REGION Network 28: ABFV 103 MULTIGRADE FILTER VALVE
   RUNG wire#powerrail
      Contact( "AlwaysTRUE" )
      { S7_Templates := "SrcType := Int" } GE_Contact(in1 := "MODE SELECTION DB".MGF."PROCESS BUFF", in2 := 30)
      { S7_Templates := "SrcType := Int" } LT_Contact(in1 := "MODE SELECTION DB".MGF."PROCESS BUFF", in2 := 55)
      { S7_Templates := "time_type := Time" } "IEC_Timer_0_DB_143".TOF(pt := T#3S, et =>)
      Coil( "AUTO_SUBOUTPUT DB"."ABFV 103 MULTIGRADE FILTER VALVE" )
   END_RUNG
   // the same network as SCL:
   "IEC_Timer_0_DB_143".TOF(IN := "AlwaysTRUE" AND ("MODE SELECTION DB".MGF."PROCESS BUFF" >= 30) AND ("MODE SELECTION DB".MGF."PROCESS BUFF" < 55),
                           PT := T#3S);
   "AUTO_SUBOUTPUT DB"."ABFV 103 MULTIGRADE FILTER VALVE" := "IEC_Timer_0_DB_143".Q;
END_REGION

REGION Network 29: ABFV 104 MULTIGRADE FILTER VALVE
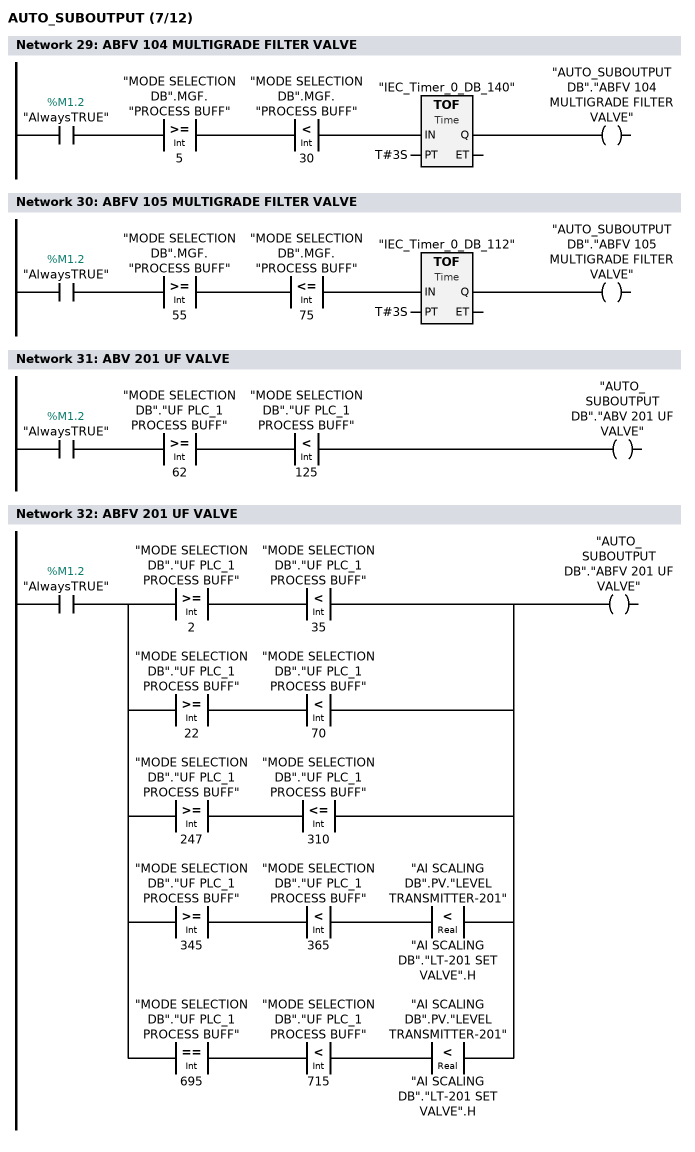
   RUNG wire#powerrail
      Contact( "AlwaysTRUE" )
      { S7_Templates := "SrcType := Int" } GE_Contact(in1 := "MODE SELECTION DB".MGF."PROCESS BUFF", in2 := 5)
      { S7_Templates := "SrcType := Int" } LT_Contact(in1 := "MODE SELECTION DB".MGF."PROCESS BUFF", in2 := 30)
      { S7_Templates := "time_type := Time" } "IEC_Timer_0_DB_140".TOF(pt := T#3S, et =>)
      Coil( "AUTO_SUBOUTPUT DB"."ABFV 104 MULTIGRADE FILTER VALVE" )
   END_RUNG
   // the same network as SCL:
   "IEC_Timer_0_DB_140".TOF(IN := "AlwaysTRUE" AND ("MODE SELECTION DB".MGF."PROCESS BUFF" >= 5) AND ("MODE SELECTION DB".MGF."PROCESS BUFF" < 30),
                           PT := T#3S);
   "AUTO_SUBOUTPUT DB"."ABFV 104 MULTIGRADE FILTER VALVE" := "IEC_Timer_0_DB_140".Q;
END_REGION

REGION Network 30: ABFV 105 MULTIGRADE FILTER VALVE
   RUNG wire#powerrail
      Contact( "AlwaysTRUE" )
      { S7_Templates := "SrcType := Int" } GE_Contact(in1 := "MODE SELECTION DB".MGF."PROCESS BUFF", in2 := 55)
      { S7_Templates := "SrcType := Int" } LE_Contact(in1 := "MODE SELECTION DB".MGF."PROCESS BUFF", in2 := 75)
      { S7_Templates := "time_type := Time" } "IEC_Timer_0_DB_112".TOF(pt := T#3S, et =>)
      Coil( "AUTO_SUBOUTPUT DB"."ABFV 105 MULTIGRADE FILTER VALVE" )
   END_RUNG
   // the same network as SCL:
   "IEC_Timer_0_DB_112".TOF(IN := "AlwaysTRUE" AND ("MODE SELECTION DB".MGF."PROCESS BUFF" >= 55) AND ("MODE SELECTION DB".MGF."PROCESS BUFF" <= 75),
                           PT := T#3S);
   "AUTO_SUBOUTPUT DB"."ABFV 105 MULTIGRADE FILTER VALVE" := "IEC_Timer_0_DB_112".Q;
END_REGION

REGION Network 31: ABV 201 UF VALVE
   RUNG wire#powerrail
      Contact( "AlwaysTRUE" )
      { S7_Templates := "SrcType := Int" } GE_Contact(in1 := "MODE SELECTION DB"."UF PLC_1 PROCESS BUFF", in2 := 62)
      { S7_Templates := "SrcType := Int" } LT_Contact(in1 := "MODE SELECTION DB"."UF PLC_1 PROCESS BUFF", in2 := 125)
      Coil( "AUTO_SUBOUTPUT DB"."ABV 201 UF VALVE" )
   END_RUNG
   // the same network as SCL:
   "AUTO_SUBOUTPUT DB"."ABV 201 UF VALVE" := "AlwaysTRUE" AND ("MODE SELECTION DB"."UF PLC_1 PROCESS BUFF" >= 62) AND ("MODE SELECTION DB"."UF PLC_1 PROCESS BUFF" < 125);
END_REGION

REGION Network 32: ABFV 201 UF VALVE
   RUNG wire#powerrail
      Contact( "AlwaysTRUE" )
      wire#w1
      { S7_Templates := "SrcType := Int" } GE_Contact(in1 := "MODE SELECTION DB"."UF PLC_1 PROCESS BUFF", in2 := 2)
      { S7_Templates := "SrcType := Int" } LT_Contact(in1 := "MODE SELECTION DB"."UF PLC_1 PROCESS BUFF", in2 := 35)
      wire#w2
      Coil( "AUTO_SUBOUTPUT DB"."ABFV 201 UF VALVE" )
   END_RUNG
   RUNG wire#w1
      { S7_Templates := "SrcType := Int" } GE_Contact(in1 := "MODE SELECTION DB"."UF PLC_1 PROCESS BUFF", in2 := 22)
      { S7_Templates := "SrcType := Int" } LT_Contact(in1 := "MODE SELECTION DB"."UF PLC_1 PROCESS BUFF", in2 := 70)
   END_RUNG wire#w2
   RUNG wire#w1
      { S7_Templates := "SrcType := Int" } GE_Contact(in1 := "MODE SELECTION DB"."UF PLC_1 PROCESS BUFF", in2 := 247)
      { S7_Templates := "SrcType := Int" } LE_Contact(in1 := "MODE SELECTION DB"."UF PLC_1 PROCESS BUFF", in2 := 310)
   END_RUNG wire#w2
   RUNG wire#w1
      { S7_Templates := "SrcType := Int" } GE_Contact(in1 := "MODE SELECTION DB"."UF PLC_1 PROCESS BUFF", in2 := 345)
      { S7_Templates := "SrcType := Int" } LT_Contact(in1 := "MODE SELECTION DB"."UF PLC_1 PROCESS BUFF", in2 := 365)
      { S7_Templates := "SrcType := Real" } LT_Contact(in1 := "AI SCALING DB".PV."LEVEL TRANSMITTER-201", in2 := "AI SCALING DB"."LT-201 SET VALVE".H)
   END_RUNG wire#w2
   RUNG wire#w1
      { S7_Templates := "SrcType := Int" } EQ_Contact(in1 := "MODE SELECTION DB"."UF PLC_1 PROCESS BUFF", in2 := 695)
      { S7_Templates := "SrcType := Int" } LT_Contact(in1 := "MODE SELECTION DB"."UF PLC_1 PROCESS BUFF", in2 := 715)
      { S7_Templates := "SrcType := Real" } LT_Contact(in1 := "AI SCALING DB".PV."LEVEL TRANSMITTER-201", in2 := "AI SCALING DB"."LT-201 SET VALVE".H)
   END_RUNG wire#w2
   // the same network as SCL:
   "AUTO_SUBOUTPUT DB"."ABFV 201 UF VALVE" := "AlwaysTRUE" AND ((("MODE SELECTION DB"."UF PLC_1 PROCESS BUFF" >= 2) AND ("MODE SELECTION DB"."UF PLC_1 PROCESS BUFF" < 35)) OR (("MODE SELECTION DB"."UF PLC_1 PROCESS BUFF" >= 22) AND ("MODE SELECTION DB"."UF PLC_1 PROCESS BUFF" < 70)) OR (("MODE SELECTION DB"."UF PLC_1 PROCESS BUFF" >= 247) AND ("MODE SELECTION DB"."UF PLC_1 PROCESS BUFF" <= 310)) OR (("MODE SELECTION DB"."UF PLC_1 PROCESS BUFF" >= 345) AND ("MODE SELECTION DB"."UF PLC_1 PROCESS BUFF" < 365) AND ("AI SCALING DB".PV."LEVEL TRANSMITTER-201" < "AI SCALING DB"."LT-201 SET VALVE".H)) OR (("MODE SELECTION DB"."UF PLC_1 PROCESS BUFF" = 695) AND ("MODE SELECTION DB"."UF PLC_1 PROCESS BUFF" < 715) AND ("AI SCALING DB".PV."LEVEL TRANSMITTER-201" < "AI SCALING DB"."LT-201 SET VALVE".H)));
END_REGION

REGION Network 33: ABFV 202 UF VALVE
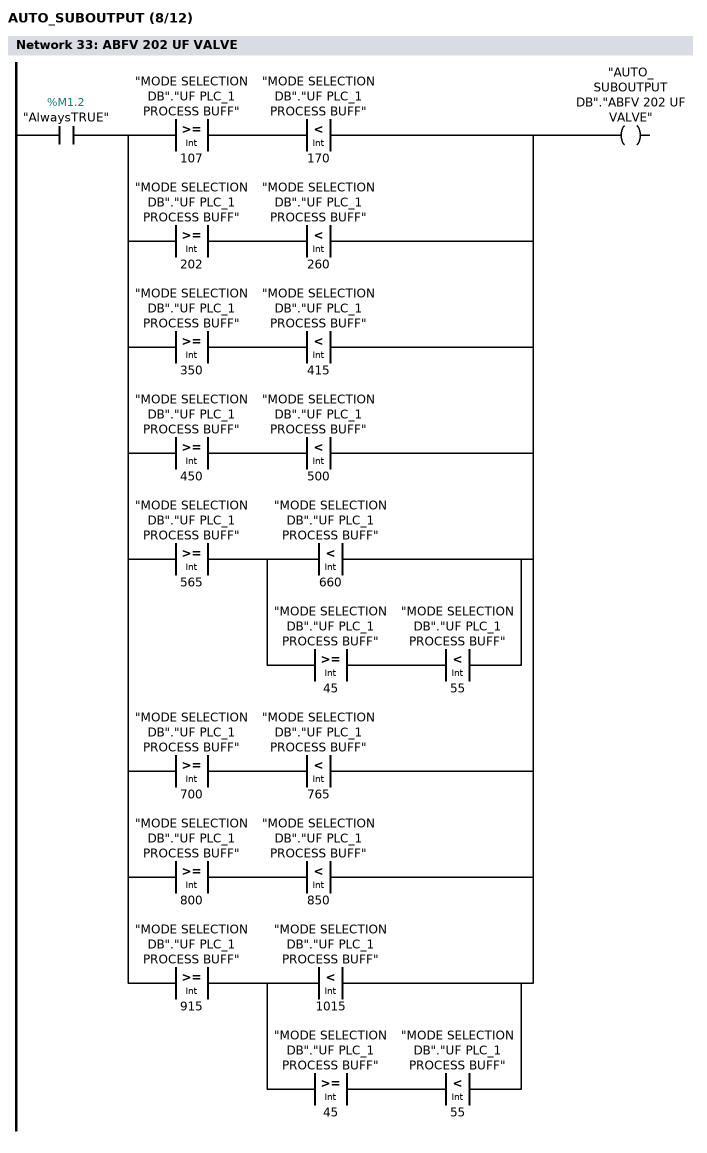
   RUNG wire#powerrail
      Contact( "AlwaysTRUE" )
      wire#w1
      { S7_Templates := "SrcType := Int" } GE_Contact(in1 := "MODE SELECTION DB"."UF PLC_1 PROCESS BUFF", in2 := 107)
      { S7_Templates := "SrcType := Int" } LT_Contact(in1 := "MODE SELECTION DB"."UF PLC_1 PROCESS BUFF", in2 := 170)
      wire#w2
      Coil( "AUTO_SUBOUTPUT DB"."ABFV 202 UF VALVE" )
   END_RUNG
   RUNG wire#w1
      { S7_Templates := "SrcType := Int" } GE_Contact(in1 := "MODE SELECTION DB"."UF PLC_1 PROCESS BUFF", in2 := 202)
      { S7_Templates := "SrcType := Int" } LT_Contact(in1 := "MODE SELECTION DB"."UF PLC_1 PROCESS BUFF", in2 := 260)
   END_RUNG wire#w2
   RUNG wire#w1
      { S7_Templates := "SrcType := Int" } GE_Contact(in1 := "MODE SELECTION DB"."UF PLC_1 PROCESS BUFF", in2 := 350)
      { S7_Templates := "SrcType := Int" } LT_Contact(in1 := "MODE SELECTION DB"."UF PLC_1 PROCESS BUFF", in2 := 415)
   END_RUNG wire#w2
   RUNG wire#w1
      { S7_Templates := "SrcType := Int" } GE_Contact(in1 := "MODE SELECTION DB"."UF PLC_1 PROCESS BUFF", in2 := 450)
      { S7_Templates := "SrcType := Int" } LT_Contact(in1 := "MODE SELECTION DB"."UF PLC_1 PROCESS BUFF", in2 := 500)
   END_RUNG wire#w2
   RUNG wire#w1
      { S7_Templates := "SrcType := Int" } GE_Contact(in1 := "MODE SELECTION DB"."UF PLC_1 PROCESS BUFF", in2 := 565)
      wire#w3
      { S7_Templates := "SrcType := Int" } LT_Contact(in1 := "MODE SELECTION DB"."UF PLC_1 PROCESS BUFF", in2 := 660)
   END_RUNG wire#w2
   RUNG wire#w3
      { S7_Templates := "SrcType := Int" } GE_Contact(in1 := "MODE SELECTION DB"."UF PLC_1 PROCESS BUFF", in2 := 45)
      { S7_Templates := "SrcType := Int" } LT_Contact(in1 := "MODE SELECTION DB"."UF PLC_1 PROCESS BUFF", in2 := 55)
   END_RUNG wire#w2
   RUNG wire#w1
      { S7_Templates := "SrcType := Int" } GE_Contact(in1 := "MODE SELECTION DB"."UF PLC_1 PROCESS BUFF", in2 := 700)
      { S7_Templates := "SrcType := Int" } LT_Contact(in1 := "MODE SELECTION DB"."UF PLC_1 PROCESS BUFF", in2 := 765)
   END_RUNG wire#w2
   RUNG wire#w1
      { S7_Templates := "SrcType := Int" } GE_Contact(in1 := "MODE SELECTION DB"."UF PLC_1 PROCESS BUFF", in2 := 800)
      { S7_Templates := "SrcType := Int" } LT_Contact(in1 := "MODE SELECTION DB"."UF PLC_1 PROCESS BUFF", in2 := 850)
   END_RUNG wire#w2
   RUNG wire#w1
      { S7_Templates := "SrcType := Int" } GE_Contact(in1 := "MODE SELECTION DB"."UF PLC_1 PROCESS BUFF", in2 := 915)
      wire#w4
      { S7_Templates := "SrcType := Int" } LT_Contact(in1 := "MODE SELECTION DB"."UF PLC_1 PROCESS BUFF", in2 := 1015)
   END_RUNG wire#w2
   RUNG wire#w4
      { S7_Templates := "SrcType := Int" } GE_Contact(in1 := "MODE SELECTION DB"."UF PLC_1 PROCESS BUFF", in2 := 45)
      { S7_Templates := "SrcType := Int" } LT_Contact(in1 := "MODE SELECTION DB"."UF PLC_1 PROCESS BUFF", in2 := 55)
   END_RUNG wire#w2
   // the same network as SCL:
   "AUTO_SUBOUTPUT DB"."ABFV 202 UF VALVE" := "AlwaysTRUE" AND ((("MODE SELECTION DB"."UF PLC_1 PROCESS BUFF" >= 107) AND ("MODE SELECTION DB"."UF PLC_1 PROCESS BUFF" < 170)) OR (("MODE SELECTION DB"."UF PLC_1 PROCESS BUFF" >= 202) AND ("MODE SELECTION DB"."UF PLC_1 PROCESS BUFF" < 260)) OR (("MODE SELECTION DB"."UF PLC_1 PROCESS BUFF" >= 350) AND ("MODE SELECTION DB"."UF PLC_1 PROCESS BUFF" < 415)) OR (("MODE SELECTION DB"."UF PLC_1 PROCESS BUFF" >= 450) AND ("MODE SELECTION DB"."UF PLC_1 PROCESS BUFF" < 500)) OR (("MODE SELECTION DB"."UF PLC_1 PROCESS BUFF" >= 565) AND (("MODE SELECTION DB"."UF PLC_1 PROCESS BUFF" < 660) OR (("MODE SELECTION DB"."UF PLC_1 PROCESS BUFF" >= 45) AND ("MODE SELECTION DB"."UF PLC_1 PROCESS BUFF" < 55)))) OR (("MODE SELECTION DB"."UF PLC_1 PROCESS BUFF" >= 700) AND ("MODE SELECTION DB"."UF PLC_1 PROCESS BUFF" < 765)) OR (("MODE SELECTION DB"."UF PLC_1 PROCESS BUFF" >= 800) AND ("MODE SELECTION DB"."UF PLC_1 PROCESS BUFF" < 850)) OR (("MODE SELECTION DB"."UF PLC_1 PROCESS BUFF" >= 915) AND (("MODE SELECTION DB"."UF PLC_1 PROCESS BUFF" < 1015) OR (("MODE SELECTION DB"."UF PLC_1 PROCESS BUFF" >= 45) AND ("MODE SELECTION DB"."UF PLC_1 PROCESS BUFF" < 55)))));
END_REGION

REGION Network 34: ABFV 203 UF VALVE
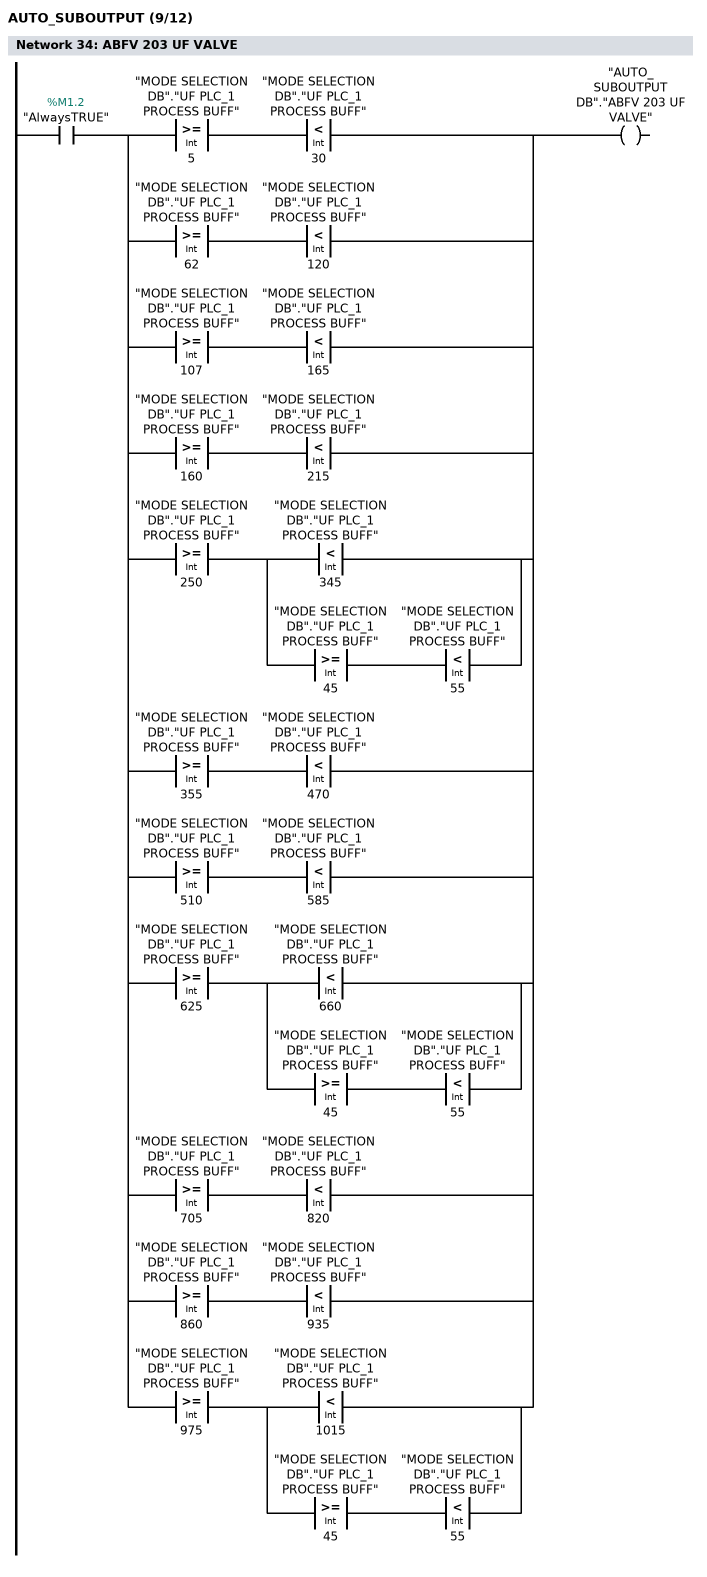
   RUNG wire#powerrail
      Contact( "AlwaysTRUE" )
      wire#w1
      { S7_Templates := "SrcType := Int" } GE_Contact(in1 := "MODE SELECTION DB"."UF PLC_1 PROCESS BUFF", in2 := 5)
      { S7_Templates := "SrcType := Int" } LT_Contact(in1 := "MODE SELECTION DB"."UF PLC_1 PROCESS BUFF", in2 := 30)
      wire#w2
      Coil( "AUTO_SUBOUTPUT DB"."ABFV 203 UF VALVE" )
   END_RUNG
   RUNG wire#w1
      { S7_Templates := "SrcType := Int" } GE_Contact(in1 := "MODE SELECTION DB"."UF PLC_1 PROCESS BUFF", in2 := 62)
      { S7_Templates := "SrcType := Int" } LT_Contact(in1 := "MODE SELECTION DB"."UF PLC_1 PROCESS BUFF", in2 := 120)
   END_RUNG wire#w2
   RUNG wire#w1
      { S7_Templates := "SrcType := Int" } GE_Contact(in1 := "MODE SELECTION DB"."UF PLC_1 PROCESS BUFF", in2 := 107)
      { S7_Templates := "SrcType := Int" } LT_Contact(in1 := "MODE SELECTION DB"."UF PLC_1 PROCESS BUFF", in2 := 165)
   END_RUNG wire#w2
   RUNG wire#w1
      { S7_Templates := "SrcType := Int" } GE_Contact(in1 := "MODE SELECTION DB"."UF PLC_1 PROCESS BUFF", in2 := 160)
      { S7_Templates := "SrcType := Int" } LT_Contact(in1 := "MODE SELECTION DB"."UF PLC_1 PROCESS BUFF", in2 := 215)
   END_RUNG wire#w2
   RUNG wire#w1
      { S7_Templates := "SrcType := Int" } GE_Contact(in1 := "MODE SELECTION DB"."UF PLC_1 PROCESS BUFF", in2 := 250)
      wire#w3
      { S7_Templates := "SrcType := Int" } LT_Contact(in1 := "MODE SELECTION DB"."UF PLC_1 PROCESS BUFF", in2 := 345)
   END_RUNG wire#w2
   RUNG wire#w3
      { S7_Templates := "SrcType := Int" } GE_Contact(in1 := "MODE SELECTION DB"."UF PLC_1 PROCESS BUFF", in2 := 45)
      { S7_Templates := "SrcType := Int" } LT_Contact(in1 := "MODE SELECTION DB"."UF PLC_1 PROCESS BUFF", in2 := 55)
   END_RUNG wire#w2
   RUNG wire#w1
      { S7_Templates := "SrcType := Int" } GE_Contact(in1 := "MODE SELECTION DB"."UF PLC_1 PROCESS BUFF", in2 := 355)
      { S7_Templates := "SrcType := Int" } LT_Contact(in1 := "MODE SELECTION DB"."UF PLC_1 PROCESS BUFF", in2 := 470)
   END_RUNG wire#w2
   RUNG wire#w1
      { S7_Templates := "SrcType := Int" } GE_Contact(in1 := "MODE SELECTION DB"."UF PLC_1 PROCESS BUFF", in2 := 510)
      { S7_Templates := "SrcType := Int" } LT_Contact(in1 := "MODE SELECTION DB"."UF PLC_1 PROCESS BUFF", in2 := 585)
   END_RUNG wire#w2
   RUNG wire#w1
      { S7_Templates := "SrcType := Int" } GE_Contact(in1 := "MODE SELECTION DB"."UF PLC_1 PROCESS BUFF", in2 := 625)
      wire#w4
      { S7_Templates := "SrcType := Int" } LT_Contact(in1 := "MODE SELECTION DB"."UF PLC_1 PROCESS BUFF", in2 := 660)
   END_RUNG wire#w2
   RUNG wire#w4
      { S7_Templates := "SrcType := Int" } GE_Contact(in1 := "MODE SELECTION DB"."UF PLC_1 PROCESS BUFF", in2 := 45)
      { S7_Templates := "SrcType := Int" } LT_Contact(in1 := "MODE SELECTION DB"."UF PLC_1 PROCESS BUFF", in2 := 55)
   END_RUNG wire#w2
   RUNG wire#w1
      { S7_Templates := "SrcType := Int" } GE_Contact(in1 := "MODE SELECTION DB"."UF PLC_1 PROCESS BUFF", in2 := 705)
      { S7_Templates := "SrcType := Int" } LT_Contact(in1 := "MODE SELECTION DB"."UF PLC_1 PROCESS BUFF", in2 := 820)
   END_RUNG wire#w2
   RUNG wire#w1
      { S7_Templates := "SrcType := Int" } GE_Contact(in1 := "MODE SELECTION DB"."UF PLC_1 PROCESS BUFF", in2 := 860)
      { S7_Templates := "SrcType := Int" } LT_Contact(in1 := "MODE SELECTION DB"."UF PLC_1 PROCESS BUFF", in2 := 935)
   END_RUNG wire#w2
   RUNG wire#w1
      { S7_Templates := "SrcType := Int" } GE_Contact(in1 := "MODE SELECTION DB"."UF PLC_1 PROCESS BUFF", in2 := 975)
      wire#w5
      { S7_Templates := "SrcType := Int" } LT_Contact(in1 := "MODE SELECTION DB"."UF PLC_1 PROCESS BUFF", in2 := 1015)
   END_RUNG wire#w2
   RUNG wire#w5
      { S7_Templates := "SrcType := Int" } GE_Contact(in1 := "MODE SELECTION DB"."UF PLC_1 PROCESS BUFF", in2 := 45)
      { S7_Templates := "SrcType := Int" } LT_Contact(in1 := "MODE SELECTION DB"."UF PLC_1 PROCESS BUFF", in2 := 55)
   END_RUNG wire#w2
   // the same network as SCL:
   "AUTO_SUBOUTPUT DB"."ABFV 203 UF VALVE" := "AlwaysTRUE" AND ((("MODE SELECTION DB"."UF PLC_1 PROCESS BUFF" >= 5) AND ("MODE SELECTION DB"."UF PLC_1 PROCESS BUFF" < 30)) OR (("MODE SELECTION DB"."UF PLC_1 PROCESS BUFF" >= 62) AND ("MODE SELECTION DB"."UF PLC_1 PROCESS BUFF" < 120)) OR (("MODE SELECTION DB"."UF PLC_1 PROCESS BUFF" >= 107) AND ("MODE SELECTION DB"."UF PLC_1 PROCESS BUFF" < 165)) OR (("MODE SELECTION DB"."UF PLC_1 PROCESS BUFF" >= 160) AND ("MODE SELECTION DB"."UF PLC_1 PROCESS BUFF" < 215)) OR (("MODE SELECTION DB"."UF PLC_1 PROCESS BUFF" >= 250) AND (("MODE SELECTION DB"."UF PLC_1 PROCESS BUFF" < 345) OR (("MODE SELECTION DB"."UF PLC_1 PROCESS BUFF" >= 45) AND ("MODE SELECTION DB"."UF PLC_1 PROCESS BUFF" < 55)))) OR (("MODE SELECTION DB"."UF PLC_1 PROCESS BUFF" >= 355) AND ("MODE SELECTION DB"."UF PLC_1 PROCESS BUFF" < 470)) OR (("MODE SELECTION DB"."UF PLC_1 PROCESS BUFF" >= 510) AND ("MODE SELECTION DB"."UF PLC_1 PROCESS BUFF" < 585)) OR (("MODE SELECTION DB"."UF PLC_1 PROCESS BUFF" >= 625) AND (("MODE SELECTION DB"."UF PLC_1 PROCESS BUFF" < 660) OR (("MODE SELECTION DB"."UF PLC_1 PROCESS BUFF" >= 45) AND ("MODE SELECTION DB"."UF PLC_1 PROCESS BUFF" < 55)))) OR (("MODE SELECTION DB"."UF PLC_1 PROCESS BUFF" >= 705) AND ("MODE SELECTION DB"."UF PLC_1 PROCESS BUFF" < 820)) OR (("MODE SELECTION DB"."UF PLC_1 PROCESS BUFF" >= 860) AND ("MODE SELECTION DB"."UF PLC_1 PROCESS BUFF" < 935)) OR (("MODE SELECTION DB"."UF PLC_1 PROCESS BUFF" >= 975) AND (("MODE SELECTION DB"."UF PLC_1 PROCESS BUFF" < 1015) OR (("MODE SELECTION DB"."UF PLC_1 PROCESS BUFF" >= 45) AND ("MODE SELECTION DB"."UF PLC_1 PROCESS BUFF" < 55)))));
END_REGION

REGION Network 35: ABFV 204 UF VALVE
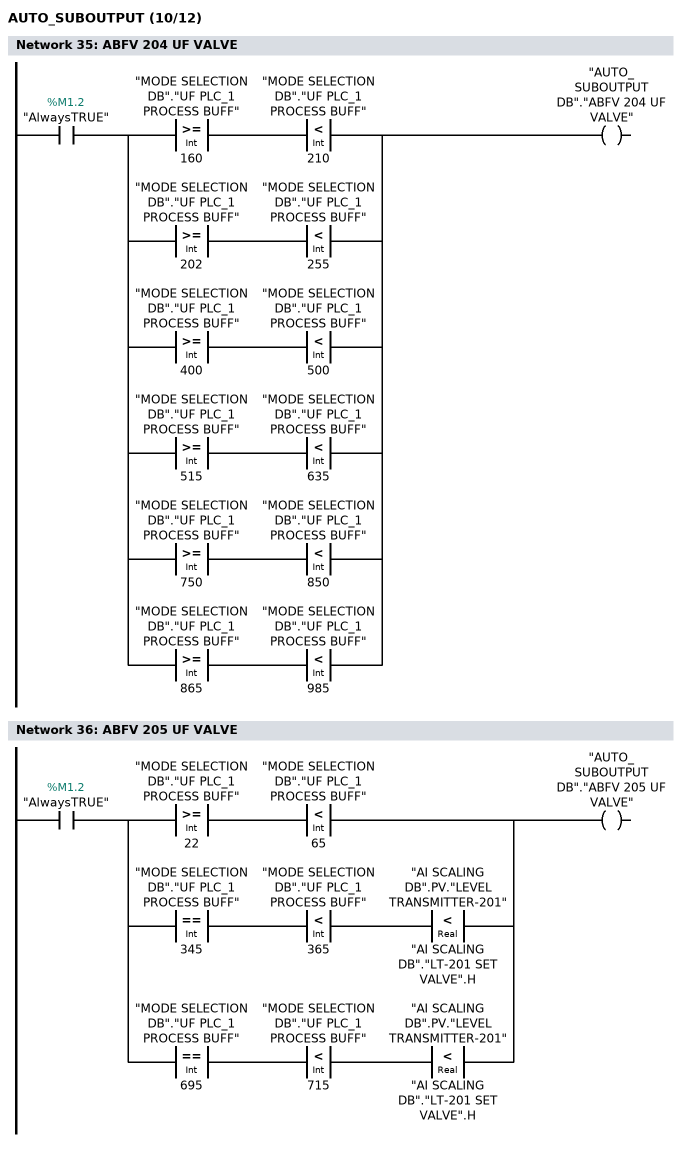
   RUNG wire#powerrail
      Contact( "AlwaysTRUE" )
      wire#w1
      { S7_Templates := "SrcType := Int" } GE_Contact(in1 := "MODE SELECTION DB"."UF PLC_1 PROCESS BUFF", in2 := 160)
      { S7_Templates := "SrcType := Int" } LT_Contact(in1 := "MODE SELECTION DB"."UF PLC_1 PROCESS BUFF", in2 := 210)
      wire#w2
      Coil( "AUTO_SUBOUTPUT DB"."ABFV 204 UF VALVE" )
   END_RUNG
   RUNG wire#w1
      { S7_Templates := "SrcType := Int" } GE_Contact(in1 := "MODE SELECTION DB"."UF PLC_1 PROCESS BUFF", in2 := 202)
      { S7_Templates := "SrcType := Int" } LT_Contact(in1 := "MODE SELECTION DB"."UF PLC_1 PROCESS BUFF", in2 := 255)
   END_RUNG wire#w2
   RUNG wire#w1
      { S7_Templates := "SrcType := Int" } GE_Contact(in1 := "MODE SELECTION DB"."UF PLC_1 PROCESS BUFF", in2 := 400)
      { S7_Templates := "SrcType := Int" } LT_Contact(in1 := "MODE SELECTION DB"."UF PLC_1 PROCESS BUFF", in2 := 500)
   END_RUNG wire#w2
   RUNG wire#w1
      { S7_Templates := "SrcType := Int" } GE_Contact(in1 := "MODE SELECTION DB"."UF PLC_1 PROCESS BUFF", in2 := 515)
      { S7_Templates := "SrcType := Int" } LT_Contact(in1 := "MODE SELECTION DB"."UF PLC_1 PROCESS BUFF", in2 := 635)
   END_RUNG wire#w2
   RUNG wire#w1
      { S7_Templates := "SrcType := Int" } GE_Contact(in1 := "MODE SELECTION DB"."UF PLC_1 PROCESS BUFF", in2 := 750)
      { S7_Templates := "SrcType := Int" } LT_Contact(in1 := "MODE SELECTION DB"."UF PLC_1 PROCESS BUFF", in2 := 850)
   END_RUNG wire#w2
   RUNG wire#w1
      { S7_Templates := "SrcType := Int" } GE_Contact(in1 := "MODE SELECTION DB"."UF PLC_1 PROCESS BUFF", in2 := 865)
      { S7_Templates := "SrcType := Int" } LT_Contact(in1 := "MODE SELECTION DB"."UF PLC_1 PROCESS BUFF", in2 := 985)
   END_RUNG wire#w2
   // the same network as SCL:
   "AUTO_SUBOUTPUT DB"."ABFV 204 UF VALVE" := "AlwaysTRUE" AND ((("MODE SELECTION DB"."UF PLC_1 PROCESS BUFF" >= 160) AND ("MODE SELECTION DB"."UF PLC_1 PROCESS BUFF" < 210)) OR (("MODE SELECTION DB"."UF PLC_1 PROCESS BUFF" >= 202) AND ("MODE SELECTION DB"."UF PLC_1 PROCESS BUFF" < 255)) OR (("MODE SELECTION DB"."UF PLC_1 PROCESS BUFF" >= 400) AND ("MODE SELECTION DB"."UF PLC_1 PROCESS BUFF" < 500)) OR (("MODE SELECTION DB"."UF PLC_1 PROCESS BUFF" >= 515) AND ("MODE SELECTION DB"."UF PLC_1 PROCESS BUFF" < 635)) OR (("MODE SELECTION DB"."UF PLC_1 PROCESS BUFF" >= 750) AND ("MODE SELECTION DB"."UF PLC_1 PROCESS BUFF" < 850)) OR (("MODE SELECTION DB"."UF PLC_1 PROCESS BUFF" >= 865) AND ("MODE SELECTION DB"."UF PLC_1 PROCESS BUFF" < 985)));
END_REGION

REGION Network 36: ABFV 205 UF VALVE
   RUNG wire#powerrail
      Contact( "AlwaysTRUE" )
      wire#w1
      { S7_Templates := "SrcType := Int" } GE_Contact(in1 := "MODE SELECTION DB"."UF PLC_1 PROCESS BUFF", in2 := 22)
      { S7_Templates := "SrcType := Int" } LT_Contact(in1 := "MODE SELECTION DB"."UF PLC_1 PROCESS BUFF", in2 := 65)
      wire#w2
      Coil( "AUTO_SUBOUTPUT DB"."ABFV 205 UF VALVE" )
   END_RUNG
   RUNG wire#w1
      { S7_Templates := "SrcType := Int" } EQ_Contact(in1 := "MODE SELECTION DB"."UF PLC_1 PROCESS BUFF", in2 := 345)
      { S7_Templates := "SrcType := Int" } LT_Contact(in1 := "MODE SELECTION DB"."UF PLC_1 PROCESS BUFF", in2 := 365)
      { S7_Templates := "SrcType := Real" } LT_Contact(in1 := "AI SCALING DB".PV."LEVEL TRANSMITTER-201", in2 := "AI SCALING DB"."LT-201 SET VALVE".H)
   END_RUNG wire#w2
   RUNG wire#w1
      { S7_Templates := "SrcType := Int" } EQ_Contact(in1 := "MODE SELECTION DB"."UF PLC_1 PROCESS BUFF", in2 := 695)
      { S7_Templates := "SrcType := Int" } LT_Contact(in1 := "MODE SELECTION DB"."UF PLC_1 PROCESS BUFF", in2 := 715)
      { S7_Templates := "SrcType := Real" } LT_Contact(in1 := "AI SCALING DB".PV."LEVEL TRANSMITTER-201", in2 := "AI SCALING DB"."LT-201 SET VALVE".H)
   END_RUNG wire#w2
   // the same network as SCL:
   "AUTO_SUBOUTPUT DB"."ABFV 205 UF VALVE" := "AlwaysTRUE" AND ((("MODE SELECTION DB"."UF PLC_1 PROCESS BUFF" >= 22) AND ("MODE SELECTION DB"."UF PLC_1 PROCESS BUFF" < 65)) OR (("MODE SELECTION DB"."UF PLC_1 PROCESS BUFF" = 345) AND ("MODE SELECTION DB"."UF PLC_1 PROCESS BUFF" < 365) AND ("AI SCALING DB".PV."LEVEL TRANSMITTER-201" < "AI SCALING DB"."LT-201 SET VALVE".H)) OR (("MODE SELECTION DB"."UF PLC_1 PROCESS BUFF" = 695) AND ("MODE SELECTION DB"."UF PLC_1 PROCESS BUFF" < 715) AND ("AI SCALING DB".PV."LEVEL TRANSMITTER-201" < "AI SCALING DB"."LT-201 SET VALVE".H)));
END_REGION

REGION Network 37: ABFV 206 UF VALVE
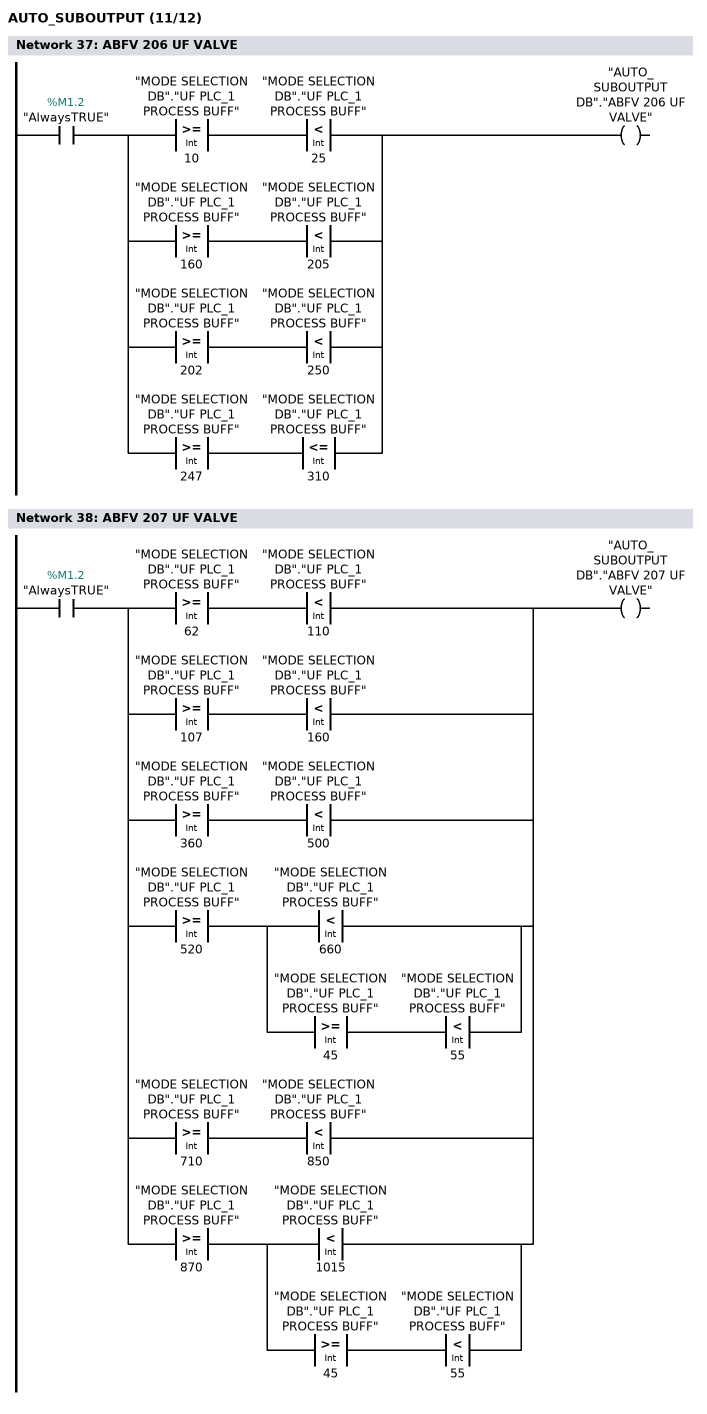
   RUNG wire#powerrail
      Contact( "AlwaysTRUE" )
      wire#w1
      { S7_Templates := "SrcType := Int" } GE_Contact(in1 := "MODE SELECTION DB"."UF PLC_1 PROCESS BUFF", in2 := 10)
      { S7_Templates := "SrcType := Int" } LT_Contact(in1 := "MODE SELECTION DB"."UF PLC_1 PROCESS BUFF", in2 := 25)
      wire#w2
      Coil( "AUTO_SUBOUTPUT DB"."ABFV 206 UF VALVE" )
   END_RUNG
   RUNG wire#w1
      { S7_Templates := "SrcType := Int" } GE_Contact(in1 := "MODE SELECTION DB"."UF PLC_1 PROCESS BUFF", in2 := 160)
      { S7_Templates := "SrcType := Int" } LT_Contact(in1 := "MODE SELECTION DB"."UF PLC_1 PROCESS BUFF", in2 := 205)
   END_RUNG wire#w2
   RUNG wire#w1
      { S7_Templates := "SrcType := Int" } GE_Contact(in1 := "MODE SELECTION DB"."UF PLC_1 PROCESS BUFF", in2 := 202)
      { S7_Templates := "SrcType := Int" } LT_Contact(in1 := "MODE SELECTION DB"."UF PLC_1 PROCESS BUFF", in2 := 250)
   END_RUNG wire#w2
   RUNG wire#w1
      { S7_Templates := "SrcType := Int" } GE_Contact(in1 := "MODE SELECTION DB"."UF PLC_1 PROCESS BUFF", in2 := 247)
      { S7_Templates := "SrcType := Int" } LE_Contact(in1 := "MODE SELECTION DB"."UF PLC_1 PROCESS BUFF", in2 := 310)
   END_RUNG wire#w2
   // the same network as SCL:
   "AUTO_SUBOUTPUT DB"."ABFV 206 UF VALVE" := "AlwaysTRUE" AND ((("MODE SELECTION DB"."UF PLC_1 PROCESS BUFF" >= 10) AND ("MODE SELECTION DB"."UF PLC_1 PROCESS BUFF" < 25)) OR (("MODE SELECTION DB"."UF PLC_1 PROCESS BUFF" >= 160) AND ("MODE SELECTION DB"."UF PLC_1 PROCESS BUFF" < 205)) OR (("MODE SELECTION DB"."UF PLC_1 PROCESS BUFF" >= 202) AND ("MODE SELECTION DB"."UF PLC_1 PROCESS BUFF" < 250)) OR (("MODE SELECTION DB"."UF PLC_1 PROCESS BUFF" >= 247) AND ("MODE SELECTION DB"."UF PLC_1 PROCESS BUFF" <= 310)));
END_REGION

REGION Network 38: ABFV 207 UF VALVE
   RUNG wire#powerrail
      Contact( "AlwaysTRUE" )
      wire#w1
      { S7_Templates := "SrcType := Int" } GE_Contact(in1 := "MODE SELECTION DB"."UF PLC_1 PROCESS BUFF", in2 := 62)
      { S7_Templates := "SrcType := Int" } LT_Contact(in1 := "MODE SELECTION DB"."UF PLC_1 PROCESS BUFF", in2 := 110)
      wire#w2
      Coil( "AUTO_SUBOUTPUT DB"."ABFV 207 UF VALVE" )
   END_RUNG
   RUNG wire#w1
      { S7_Templates := "SrcType := Int" } GE_Contact(in1 := "MODE SELECTION DB"."UF PLC_1 PROCESS BUFF", in2 := 107)
      { S7_Templates := "SrcType := Int" } LT_Contact(in1 := "MODE SELECTION DB"."UF PLC_1 PROCESS BUFF", in2 := 160)
   END_RUNG wire#w2
   RUNG wire#w1
      { S7_Templates := "SrcType := Int" } GE_Contact(in1 := "MODE SELECTION DB"."UF PLC_1 PROCESS BUFF", in2 := 360)
      { S7_Templates := "SrcType := Int" } LT_Contact(in1 := "MODE SELECTION DB"."UF PLC_1 PROCESS BUFF", in2 := 500)
   END_RUNG wire#w2
   RUNG wire#w1
      { S7_Templates := "SrcType := Int" } GE_Contact(in1 := "MODE SELECTION DB"."UF PLC_1 PROCESS BUFF", in2 := 520)
      wire#w3
      { S7_Templates := "SrcType := Int" } LT_Contact(in1 := "MODE SELECTION DB"."UF PLC_1 PROCESS BUFF", in2 := 660)
   END_RUNG wire#w2
   RUNG wire#w3
      { S7_Templates := "SrcType := Int" } GE_Contact(in1 := "MODE SELECTION DB"."UF PLC_1 PROCESS BUFF", in2 := 45)
      { S7_Templates := "SrcType := Int" } LT_Contact(in1 := "MODE SELECTION DB"."UF PLC_1 PROCESS BUFF", in2 := 55)
   END_RUNG wire#w2
   RUNG wire#w1
      { S7_Templates := "SrcType := Int" } GE_Contact(in1 := "MODE SELECTION DB"."UF PLC_1 PROCESS BUFF", in2 := 710)
      { S7_Templates := "SrcType := Int" } LT_Contact(in1 := "MODE SELECTION DB"."UF PLC_1 PROCESS BUFF", in2 := 850)
   END_RUNG wire#w2
   RUNG wire#w1
      { S7_Templates := "SrcType := Int" } GE_Contact(in1 := "MODE SELECTION DB"."UF PLC_1 PROCESS BUFF", in2 := 870)
      wire#w4
      { S7_Templates := "SrcType := Int" } LT_Contact(in1 := "MODE SELECTION DB"."UF PLC_1 PROCESS BUFF", in2 := 1015)
   END_RUNG wire#w2
   RUNG wire#w4
      { S7_Templates := "SrcType := Int" } GE_Contact(in1 := "MODE SELECTION DB"."UF PLC_1 PROCESS BUFF", in2 := 45)
      { S7_Templates := "SrcType := Int" } LT_Contact(in1 := "MODE SELECTION DB"."UF PLC_1 PROCESS BUFF", in2 := 55)
   END_RUNG wire#w2
   // the same network as SCL:
   "AUTO_SUBOUTPUT DB"."ABFV 207 UF VALVE" := "AlwaysTRUE" AND ((("MODE SELECTION DB"."UF PLC_1 PROCESS BUFF" >= 62) AND ("MODE SELECTION DB"."UF PLC_1 PROCESS BUFF" < 110)) OR (("MODE SELECTION DB"."UF PLC_1 PROCESS BUFF" >= 107) AND ("MODE SELECTION DB"."UF PLC_1 PROCESS BUFF" < 160)) OR (("MODE SELECTION DB"."UF PLC_1 PROCESS BUFF" >= 360) AND ("MODE SELECTION DB"."UF PLC_1 PROCESS BUFF" < 500)) OR (("MODE SELECTION DB"."UF PLC_1 PROCESS BUFF" >= 520) AND (("MODE SELECTION DB"."UF PLC_1 PROCESS BUFF" < 660) OR (("MODE SELECTION DB"."UF PLC_1 PROCESS BUFF" >= 45) AND ("MODE SELECTION DB"."UF PLC_1 PROCESS BUFF" < 55)))) OR (("MODE SELECTION DB"."UF PLC_1 PROCESS BUFF" >= 710) AND ("MODE SELECTION DB"."UF PLC_1 PROCESS BUFF" < 850)) OR (("MODE SELECTION DB"."UF PLC_1 PROCESS BUFF" >= 870) AND (("MODE SELECTION DB"."UF PLC_1 PROCESS BUFF" < 1015) OR (("MODE SELECTION DB"."UF PLC_1 PROCESS BUFF" >= 45) AND ("MODE SELECTION DB"."UF PLC_1 PROCESS BUFF" < 55)))));
END_REGION

REGION Network 39: ABFV 208 UF VALVE
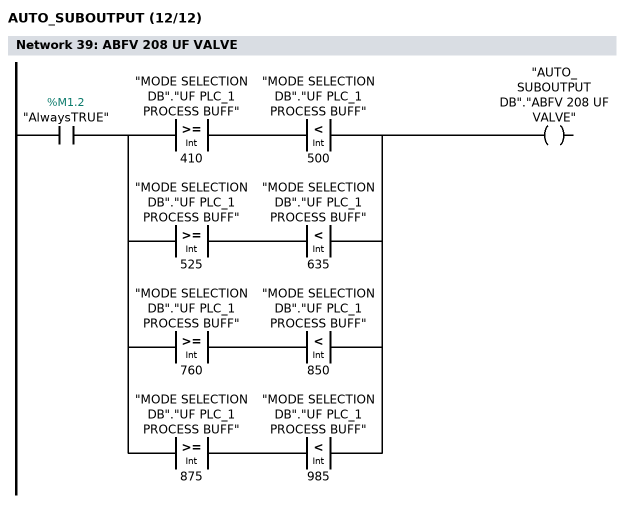
   RUNG wire#powerrail
      Contact( "AlwaysTRUE" )
      wire#w1
      { S7_Templates := "SrcType := Int" } GE_Contact(in1 := "MODE SELECTION DB"."UF PLC_1 PROCESS BUFF", in2 := 410)
      { S7_Templates := "SrcType := Int" } LT_Contact(in1 := "MODE SELECTION DB"."UF PLC_1 PROCESS BUFF", in2 := 500)
      wire#w2
      Coil( "AUTO_SUBOUTPUT DB"."ABFV 208 UF VALVE" )
   END_RUNG
   RUNG wire#w1
      { S7_Templates := "SrcType := Int" } GE_Contact(in1 := "MODE SELECTION DB"."UF PLC_1 PROCESS BUFF", in2 := 525)
      { S7_Templates := "SrcType := Int" } LT_Contact(in1 := "MODE SELECTION DB"."UF PLC_1 PROCESS BUFF", in2 := 635)
   END_RUNG wire#w2
   RUNG wire#w1
      { S7_Templates := "SrcType := Int" } GE_Contact(in1 := "MODE SELECTION DB"."UF PLC_1 PROCESS BUFF", in2 := 760)
      { S7_Templates := "SrcType := Int" } LT_Contact(in1 := "MODE SELECTION DB"."UF PLC_1 PROCESS BUFF", in2 := 850)
   END_RUNG wire#w2
   RUNG wire#w1
      { S7_Templates := "SrcType := Int" } GE_Contact(in1 := "MODE SELECTION DB"."UF PLC_1 PROCESS BUFF", in2 := 875)
      { S7_Templates := "SrcType := Int" } LT_Contact(in1 := "MODE SELECTION DB"."UF PLC_1 PROCESS BUFF", in2 := 985)
   END_RUNG wire#w2
   // the same network as SCL:
   "AUTO_SUBOUTPUT DB"."ABFV 208 UF VALVE" := "AlwaysTRUE" AND ((("MODE SELECTION DB"."UF PLC_1 PROCESS BUFF" >= 410) AND ("MODE SELECTION DB"."UF PLC_1 PROCESS BUFF" < 500)) OR (("MODE SELECTION DB"."UF PLC_1 PROCESS BUFF" >= 525) AND ("MODE SELECTION DB"."UF PLC_1 PROCESS BUFF" < 635)) OR (("MODE SELECTION DB"."UF PLC_1 PROCESS BUFF" >= 760) AND ("MODE SELECTION DB"."UF PLC_1 PROCESS BUFF" < 850)) OR (("MODE SELECTION DB"."UF PLC_1 PROCESS BUFF" >= 875) AND ("MODE SELECTION DB"."UF PLC_1 PROCESS BUFF" < 985)));
END_REGION
END_FUNCTION

FUNCTION "BACKWASH" : Void   // FC13, LAD
{ S7_Optimized_Access := 'TRUE' }
// stored: SetENOAutomatically false
BEGIN

REGION Network 1: BACKWASH_TIMER
END_REGION

REGION Network 2: VALVE OPEN
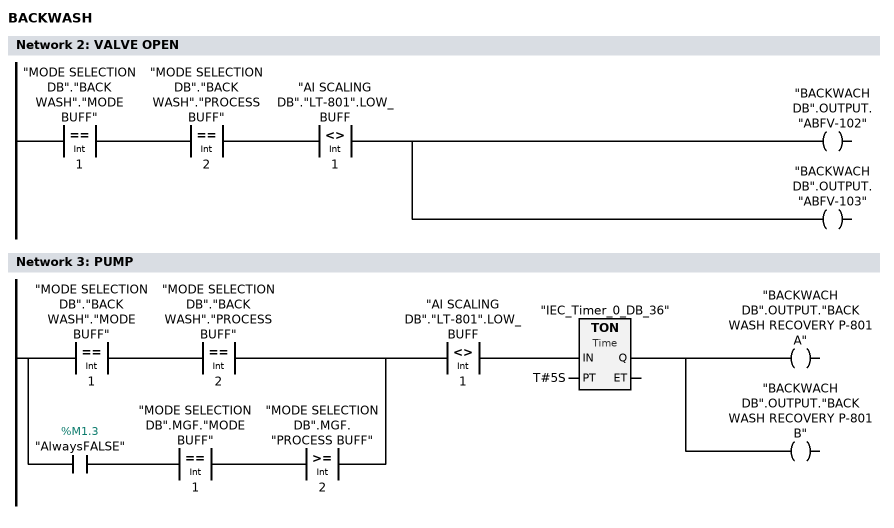
   RUNG wire#powerrail
      { S7_Templates := "SrcType := Int" } EQ_Contact(in1 := "MODE SELECTION DB"."BACK WASH"."MODE BUFF", in2 := 1)
      { S7_Templates := "SrcType := Int" } EQ_Contact(in1 := "MODE SELECTION DB"."BACK WASH"."PROCESS BUFF", in2 := 2)
      { S7_Templates := "SrcType := Int" } NE_Contact(in1 := "AI SCALING DB"."LT-801".LOW_BUFF, in2 := 1)
      wire#w1
      Coil( "BACKWACH DB".OUTPUT."ABFV-102" )
   END_RUNG
   RUNG wire#w1
      Coil( "BACKWACH DB".OUTPUT."ABFV-103" )
   END_RUNG
   // the same network as SCL:
   "BACKWACH DB".OUTPUT."ABFV-102" := ("MODE SELECTION DB"."BACK WASH"."MODE BUFF" = 1) AND ("MODE SELECTION DB"."BACK WASH"."PROCESS BUFF" = 2) AND ("AI SCALING DB"."LT-801".LOW_BUFF <> 1);
   "BACKWACH DB".OUTPUT."ABFV-103" := "BACKWACH DB".OUTPUT."ABFV-102";
END_REGION

REGION Network 3: PUMP
   RUNG wire#powerrail
      { S7_Templates := "SrcType := Int" } EQ_Contact(in1 := "MODE SELECTION DB"."BACK WASH"."MODE BUFF", in2 := 1)
      { S7_Templates := "SrcType := Int" } EQ_Contact(in1 := "MODE SELECTION DB"."BACK WASH"."PROCESS BUFF", in2 := 2)
      wire#w1
      { S7_Templates := "SrcType := Int" } NE_Contact(in1 := "AI SCALING DB"."LT-801".LOW_BUFF, in2 := 1)
      { S7_Templates := "time_type := Time" } "IEC_Timer_0_DB_36".TON(pt := T#5S, et =>)
      wire#w2
      Coil( "BACKWACH DB".OUTPUT."BACK WASH RECOVERY P-801 A" )
   END_RUNG
   RUNG wire#powerrail
      Contact( "AlwaysFALSE" )
      { S7_Templates := "SrcType := Int" } EQ_Contact(in1 := "MODE SELECTION DB".MGF."MODE BUFF", in2 := 1)
      { S7_Templates := "SrcType := Int" } GE_Contact(in1 := "MODE SELECTION DB".MGF."PROCESS BUFF", in2 := 2)
   END_RUNG wire#w1
   RUNG wire#w2
      Coil( "BACKWACH DB".OUTPUT."BACK WASH RECOVERY P-801 B" )
   END_RUNG
   // the same network as SCL:
   "IEC_Timer_0_DB_36".TON(IN := ((("MODE SELECTION DB"."BACK WASH"."MODE BUFF" = 1) AND ("MODE SELECTION DB"."BACK WASH"."PROCESS BUFF" = 2)) OR ("AlwaysFALSE" AND ("MODE SELECTION DB".MGF."MODE BUFF" = 1) AND ("MODE SELECTION DB".MGF."PROCESS BUFF" >= 2))) AND ("AI SCALING DB"."LT-801".LOW_BUFF <> 1),
                           PT := T#5S);
   "BACKWACH DB".OUTPUT."BACK WASH RECOVERY P-801 A" := "IEC_Timer_0_DB_36".Q;
   "BACKWACH DB".OUTPUT."BACK WASH RECOVERY P-801 B" := "IEC_Timer_0_DB_36".Q;
END_REGION
END_FUNCTION

FUNCTION "MGF AUTO" : Void   // FC10, LAD
{ S7_Optimized_Access := 'TRUE' }
// stored: SetENOAutomatically false
BEGIN

REGION Network 1
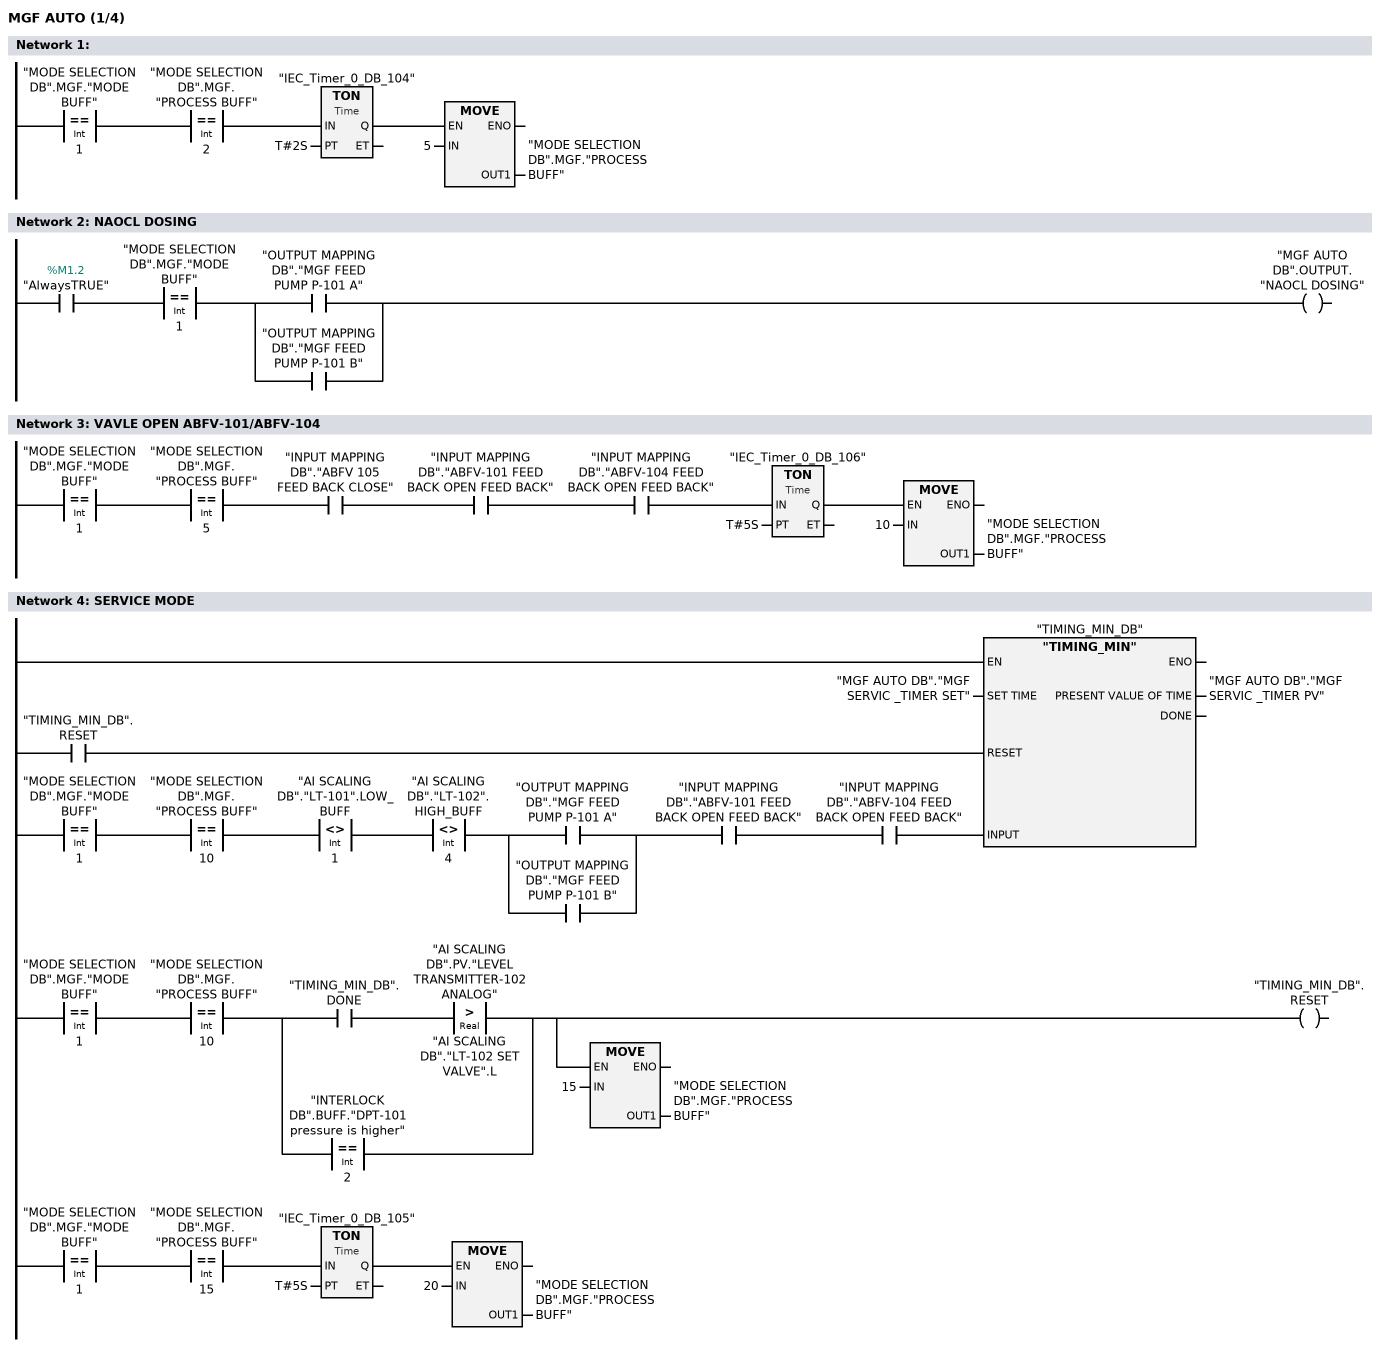
   RUNG wire#powerrail
      { S7_Templates := "SrcType := Int" } EQ_Contact(in1 := "MODE SELECTION DB".MGF."MODE BUFF", in2 := 1)
      { S7_Templates := "SrcType := Int" } EQ_Contact(in1 := "MODE SELECTION DB".MGF."PROCESS BUFF", in2 := 2)
      { S7_Templates := "time_type := Time" } "IEC_Timer_0_DB_104".TON(pt := T#2S, et =>)
      Move(in := 5, out1 => "MODE SELECTION DB".MGF."PROCESS BUFF")
   END_RUNG
   // the same network as SCL:
   "IEC_Timer_0_DB_104".TON(IN := ("MODE SELECTION DB".MGF."MODE BUFF" = 1) AND ("MODE SELECTION DB".MGF."PROCESS BUFF" = 2),
                           PT := T#2S);
   IF "IEC_Timer_0_DB_104".Q THEN "MODE SELECTION DB".MGF."PROCESS BUFF" := 5; END_IF;
END_REGION

REGION Network 2: NAOCL DOSING
   RUNG wire#powerrail
      Contact( "AlwaysTRUE" )
      { S7_Templates := "SrcType := Int" } EQ_Contact(in1 := "MODE SELECTION DB".MGF."MODE BUFF", in2 := 1)
      wire#w1
      Contact( "OUTPUT MAPPING DB"."MGF FEED PUMP P-101 A" )
      wire#w2
      Coil( "MGF AUTO DB".OUTPUT."NAOCL DOSING" )
   END_RUNG
   RUNG wire#w1
      Contact( "OUTPUT MAPPING DB"."MGF FEED PUMP P-101 B" )
   END_RUNG wire#w2
   // the same network as SCL:
   "MGF AUTO DB".OUTPUT."NAOCL DOSING" := "AlwaysTRUE" AND ("MODE SELECTION DB".MGF."MODE BUFF" = 1) AND ("OUTPUT MAPPING DB"."MGF FEED PUMP P-101 A" OR "OUTPUT MAPPING DB"."MGF FEED PUMP P-101 B");
END_REGION

REGION Network 3: VAVLE OPEN ABFV-101/ABFV-104
   RUNG wire#powerrail
      { S7_Templates := "SrcType := Int" } EQ_Contact(in1 := "MODE SELECTION DB".MGF."MODE BUFF", in2 := 1)
      { S7_Templates := "SrcType := Int" } EQ_Contact(in1 := "MODE SELECTION DB".MGF."PROCESS BUFF", in2 := 5)
      Contact( "INPUT MAPPING DB"."ABFV 105 FEED BACK CLOSE" )
      Contact( "INPUT MAPPING DB"."ABFV-101 FEED BACK OPEN FEED BACK" )
      Contact( "INPUT MAPPING DB"."ABFV-104 FEED BACK OPEN FEED BACK" )
      { S7_Templates := "time_type := Time" } "IEC_Timer_0_DB_106".TON(pt := T#5S, et =>)
      Move(in := 10, out1 => "MODE SELECTION DB".MGF."PROCESS BUFF")
   END_RUNG
   // the same network as SCL:
   "IEC_Timer_0_DB_106".TON(IN := ("MODE SELECTION DB".MGF."MODE BUFF" = 1) AND ("MODE SELECTION DB".MGF."PROCESS BUFF" = 5) AND "INPUT MAPPING DB"."ABFV 105 FEED BACK CLOSE" AND "INPUT MAPPING DB"."ABFV-101 FEED BACK OPEN FEED BACK" AND "INPUT MAPPING DB"."ABFV-104 FEED BACK OPEN FEED BACK",
                           PT := T#5S);
   IF "IEC_Timer_0_DB_106".Q THEN "MODE SELECTION DB".MGF."PROCESS BUFF" := 10; END_IF;
END_REGION

REGION Network 4: SERVICE MODE
   RUNG wire#powerrail
      "TIMING_MIN_DB"(RESET := wire#w1, INPUT := wire#w4, "SET TIME" := "MGF AUTO DB"."MGF SERVIC _TIMER SET", "PRESENT VALUE OF TIME" => "MGF AUTO DB"."MGF SERVIC _TIMER PV", DONE =>)
   END_RUNG
   RUNG wire#powerrail
      Contact( "TIMING_MIN_DB".RESET )
   END_RUNG wire#w1
   RUNG wire#powerrail
      { S7_Templates := "SrcType := Int" } EQ_Contact(in1 := "MODE SELECTION DB".MGF."MODE BUFF", in2 := 1)
      { S7_Templates := "SrcType := Int" } EQ_Contact(in1 := "MODE SELECTION DB".MGF."PROCESS BUFF", in2 := 10)
      { S7_Templates := "SrcType := Int" } NE_Contact(in1 := "AI SCALING DB"."LT-101".LOW_BUFF, in2 := 1)
      { S7_Templates := "SrcType := Int" } NE_Contact(in1 := "AI SCALING DB"."LT-102".HIGH_BUFF, in2 := 4)
      wire#w2
      Contact( "OUTPUT MAPPING DB"."MGF FEED PUMP P-101 A" )
      wire#w3
      Contact( "INPUT MAPPING DB"."ABFV-101 FEED BACK OPEN FEED BACK" )
      Contact( "INPUT MAPPING DB"."ABFV-104 FEED BACK OPEN FEED BACK" )
   END_RUNG wire#w4
   RUNG wire#w2
      Contact( "OUTPUT MAPPING DB"."MGF FEED PUMP P-101 B" )
   END_RUNG wire#w3
   RUNG wire#powerrail
      { S7_Templates := "SrcType := Int" } EQ_Contact(in1 := "MODE SELECTION DB".MGF."MODE BUFF", in2 := 1)
      { S7_Templates := "SrcType := Int" } EQ_Contact(in1 := "MODE SELECTION DB".MGF."PROCESS BUFF", in2 := 10)
      wire#w5
      Contact( "TIMING_MIN_DB".DONE )
      { S7_Templates := "SrcType := Real" } GT_Contact(in1 := "AI SCALING DB".PV."LEVEL TRANSMITTER-102 ANALOG", in2 := "AI SCALING DB"."LT-102 SET VALVE".L)
      wire#w6
      Coil( "TIMING_MIN_DB".RESET )
   END_RUNG
   RUNG wire#w5
      { S7_Templates := "SrcType := Int" } EQ_Contact(in1 := "INTERLOCK DB".BUFF."DPT-101 pressure is higher", in2 := 2)
   END_RUNG wire#w6
   RUNG wire#w6
      Move(in := 15, out1 => "MODE SELECTION DB".MGF."PROCESS BUFF")
   END_RUNG
   RUNG wire#powerrail
      { S7_Templates := "SrcType := Int" } EQ_Contact(in1 := "MODE SELECTION DB".MGF."MODE BUFF", in2 := 1)
      { S7_Templates := "SrcType := Int" } EQ_Contact(in1 := "MODE SELECTION DB".MGF."PROCESS BUFF", in2 := 15)
      { S7_Templates := "time_type := Time" } "IEC_Timer_0_DB_105".TON(pt := T#5S, et =>)
      Move(in := 20, out1 => "MODE SELECTION DB".MGF."PROCESS BUFF")
   END_RUNG
   // the same network as SCL:
   "TIMING_MIN_DB"("SET TIME" := "MGF AUTO DB"."MGF SERVIC _TIMER SET",   // "TIMING_MIN"
                   RESET := "TIMING_MIN_DB".RESET,
                   INPUT := ("MODE SELECTION DB".MGF."MODE BUFF" = 1) AND ("MODE SELECTION DB".MGF."PROCESS BUFF" = 10) AND ("AI SCALING DB"."LT-101".LOW_BUFF <> 1) AND ("AI SCALING DB"."LT-102".HIGH_BUFF <> 4) AND ("OUTPUT MAPPING DB"."MGF FEED PUMP P-101 A" OR "OUTPUT MAPPING DB"."MGF FEED PUMP P-101 B") AND "INPUT MAPPING DB"."ABFV-101 FEED BACK OPEN FEED BACK" AND "INPUT MAPPING DB"."ABFV-104 FEED BACK OPEN FEED BACK",
                   "PRESENT VALUE OF TIME" => "MGF AUTO DB"."MGF SERVIC _TIMER PV");
   "TIMING_MIN_DB".RESET := ("MODE SELECTION DB".MGF."MODE BUFF" = 1) AND ("MODE SELECTION DB".MGF."PROCESS BUFF" = 10) AND (("TIMING_MIN_DB".DONE AND ("AI SCALING DB".PV."LEVEL TRANSMITTER-102 ANALOG" > "AI SCALING DB"."LT-102 SET VALVE".L)) OR ("INTERLOCK DB".BUFF."DPT-101 pressure is higher" = 2));
   IF "TIMING_MIN_DB".RESET THEN "MODE SELECTION DB".MGF."PROCESS BUFF" := 15; END_IF;
   "IEC_Timer_0_DB_105".TON(IN := ("MODE SELECTION DB".MGF."MODE BUFF" = 1) AND ("MODE SELECTION DB".MGF."PROCESS BUFF" = 15),
                           PT := T#5S);
   IF "IEC_Timer_0_DB_105".Q THEN "MODE SELECTION DB".MGF."PROCESS BUFF" := 20; END_IF;
END_REGION

REGION Network 5: VAVLE CLOSE ABFV-101/ABFV-104
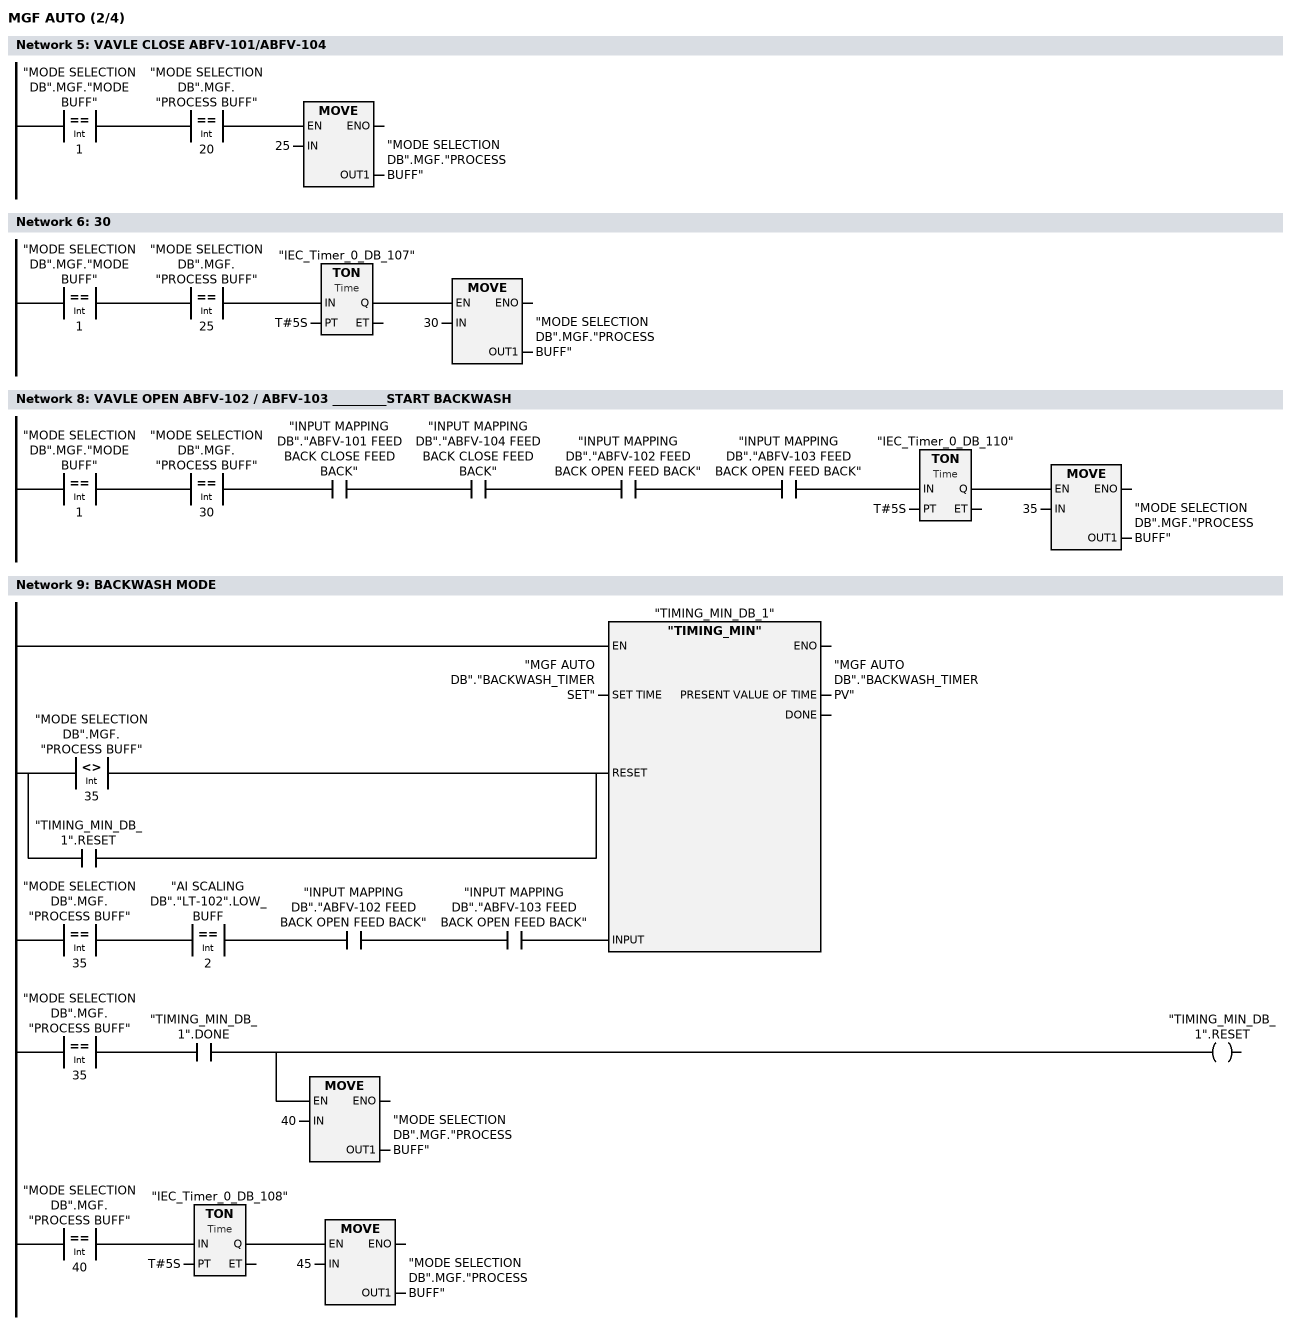
   RUNG wire#powerrail
      { S7_Templates := "SrcType := Int" } EQ_Contact(in1 := "MODE SELECTION DB".MGF."MODE BUFF", in2 := 1)
      { S7_Templates := "SrcType := Int" } EQ_Contact(in1 := "MODE SELECTION DB".MGF."PROCESS BUFF", in2 := 20)
      Move(in := 25, out1 => "MODE SELECTION DB".MGF."PROCESS BUFF")
   END_RUNG
   // the same network as SCL:
   IF ("MODE SELECTION DB".MGF."MODE BUFF" = 1) AND ("MODE SELECTION DB".MGF."PROCESS BUFF" = 20) THEN
       "MODE SELECTION DB".MGF."PROCESS BUFF" := 25;
   END_IF;
END_REGION

REGION Network 6: 30
   RUNG wire#powerrail
      { S7_Templates := "SrcType := Int" } EQ_Contact(in1 := "MODE SELECTION DB".MGF."MODE BUFF", in2 := 1)
      { S7_Templates := "SrcType := Int" } EQ_Contact(in1 := "MODE SELECTION DB".MGF."PROCESS BUFF", in2 := 25)
      { S7_Templates := "time_type := Time" } "IEC_Timer_0_DB_107".TON(pt := T#5S, et =>)
      Move(in := 30, out1 => "MODE SELECTION DB".MGF."PROCESS BUFF")
   END_RUNG
   // the same network as SCL:
   "IEC_Timer_0_DB_107".TON(IN := ("MODE SELECTION DB".MGF."MODE BUFF" = 1) AND ("MODE SELECTION DB".MGF."PROCESS BUFF" = 25),
                           PT := T#5S);
   IF "IEC_Timer_0_DB_107".Q THEN "MODE SELECTION DB".MGF."PROCESS BUFF" := 30; END_IF;
END_REGION

REGION Network 8: VAVLE OPEN ABFV-102 / ABFV-103 _________START BACKWASH
   RUNG wire#powerrail
      { S7_Templates := "SrcType := Int" } EQ_Contact(in1 := "MODE SELECTION DB".MGF."MODE BUFF", in2 := 1)
      { S7_Templates := "SrcType := Int" } EQ_Contact(in1 := "MODE SELECTION DB".MGF."PROCESS BUFF", in2 := 30)
      Contact( "INPUT MAPPING DB"."ABFV-101 FEED BACK CLOSE FEED BACK" )
      Contact( "INPUT MAPPING DB"."ABFV-104 FEED BACK CLOSE FEED BACK" )
      Contact( "INPUT MAPPING DB"."ABFV-102 FEED BACK OPEN FEED BACK" )
      Contact( "INPUT MAPPING DB"."ABFV-103 FEED BACK OPEN FEED BACK" )
      { S7_Templates := "time_type := Time" } "IEC_Timer_0_DB_110".TON(pt := T#5S, et =>)
      Move(in := 35, out1 => "MODE SELECTION DB".MGF."PROCESS BUFF")
   END_RUNG
   // the same network as SCL:
   "IEC_Timer_0_DB_110".TON(IN := ("MODE SELECTION DB".MGF."MODE BUFF" = 1) AND ("MODE SELECTION DB".MGF."PROCESS BUFF" = 30) AND "INPUT MAPPING DB"."ABFV-101 FEED BACK CLOSE FEED BACK" AND "INPUT MAPPING DB"."ABFV-104 FEED BACK CLOSE FEED BACK" AND "INPUT MAPPING DB"."ABFV-102 FEED BACK OPEN FEED BACK" AND "INPUT MAPPING DB"."ABFV-103 FEED BACK OPEN FEED BACK",
                           PT := T#5S);
   IF "IEC_Timer_0_DB_110".Q THEN "MODE SELECTION DB".MGF."PROCESS BUFF" := 35; END_IF;
END_REGION

REGION Network 9: BACKWASH MODE
   RUNG wire#powerrail
      "TIMING_MIN_DB_1"(RESET := wire#w1, INPUT := wire#w2, "SET TIME" := "MGF AUTO DB"."BACKWASH_TIMER SET", "PRESENT VALUE OF TIME" => "MGF AUTO DB"."BACKWASH_TIMER PV", DONE =>)
   END_RUNG
   RUNG wire#powerrail
      { S7_Templates := "SrcType := Int" } NE_Contact(in1 := "MODE SELECTION DB".MGF."PROCESS BUFF", in2 := 35)
   END_RUNG wire#w1
   RUNG wire#powerrail
      Contact( "TIMING_MIN_DB_1".RESET )
   END_RUNG wire#w1
   RUNG wire#powerrail
      { S7_Templates := "SrcType := Int" } EQ_Contact(in1 := "MODE SELECTION DB".MGF."PROCESS BUFF", in2 := 35)
      { S7_Templates := "SrcType := Int" } EQ_Contact(in1 := "AI SCALING DB"."LT-102".LOW_BUFF, in2 := 2)
      Contact( "INPUT MAPPING DB"."ABFV-102 FEED BACK OPEN FEED BACK" )
      Contact( "INPUT MAPPING DB"."ABFV-103 FEED BACK OPEN FEED BACK" )
   END_RUNG wire#w2
   RUNG wire#powerrail
      { S7_Templates := "SrcType := Int" } EQ_Contact(in1 := "MODE SELECTION DB".MGF."PROCESS BUFF", in2 := 35)
      Contact( "TIMING_MIN_DB_1".DONE )
      wire#w3
      Coil( "TIMING_MIN_DB_1".RESET )
   END_RUNG
   RUNG wire#w3
      Move(in := 40, out1 => "MODE SELECTION DB".MGF."PROCESS BUFF")
   END_RUNG
   RUNG wire#powerrail
      { S7_Templates := "SrcType := Int" } EQ_Contact(in1 := "MODE SELECTION DB".MGF."PROCESS BUFF", in2 := 40)
      { S7_Templates := "time_type := Time" } "IEC_Timer_0_DB_108".TON(pt := T#5S, et =>)
      Move(in := 45, out1 => "MODE SELECTION DB".MGF."PROCESS BUFF")
   END_RUNG
   // the same network as SCL:
   "TIMING_MIN_DB_1"("SET TIME" := "MGF AUTO DB"."BACKWASH_TIMER SET",   // "TIMING_MIN"
                     RESET := ("MODE SELECTION DB".MGF."PROCESS BUFF" <> 35) OR "TIMING_MIN_DB_1".RESET,
                     INPUT := ("MODE SELECTION DB".MGF."PROCESS BUFF" = 35) AND ("AI SCALING DB"."LT-102".LOW_BUFF = 2) AND "INPUT MAPPING DB"."ABFV-102 FEED BACK OPEN FEED BACK" AND "INPUT MAPPING DB"."ABFV-103 FEED BACK OPEN FEED BACK",
                     "PRESENT VALUE OF TIME" => "MGF AUTO DB"."BACKWASH_TIMER PV");
   "TIMING_MIN_DB_1".RESET := ("MODE SELECTION DB".MGF."PROCESS BUFF" = 35) AND "TIMING_MIN_DB_1".DONE;
   IF "TIMING_MIN_DB_1".RESET THEN "MODE SELECTION DB".MGF."PROCESS BUFF" := 40; END_IF;
   "IEC_Timer_0_DB_108".TON(IN := "MODE SELECTION DB".MGF."PROCESS BUFF" = 40, PT := T#5S);
   IF "IEC_Timer_0_DB_108".Q THEN "MODE SELECTION DB".MGF."PROCESS BUFF" := 45; END_IF;
END_REGION

REGION Network 10: VALVE CLOSE
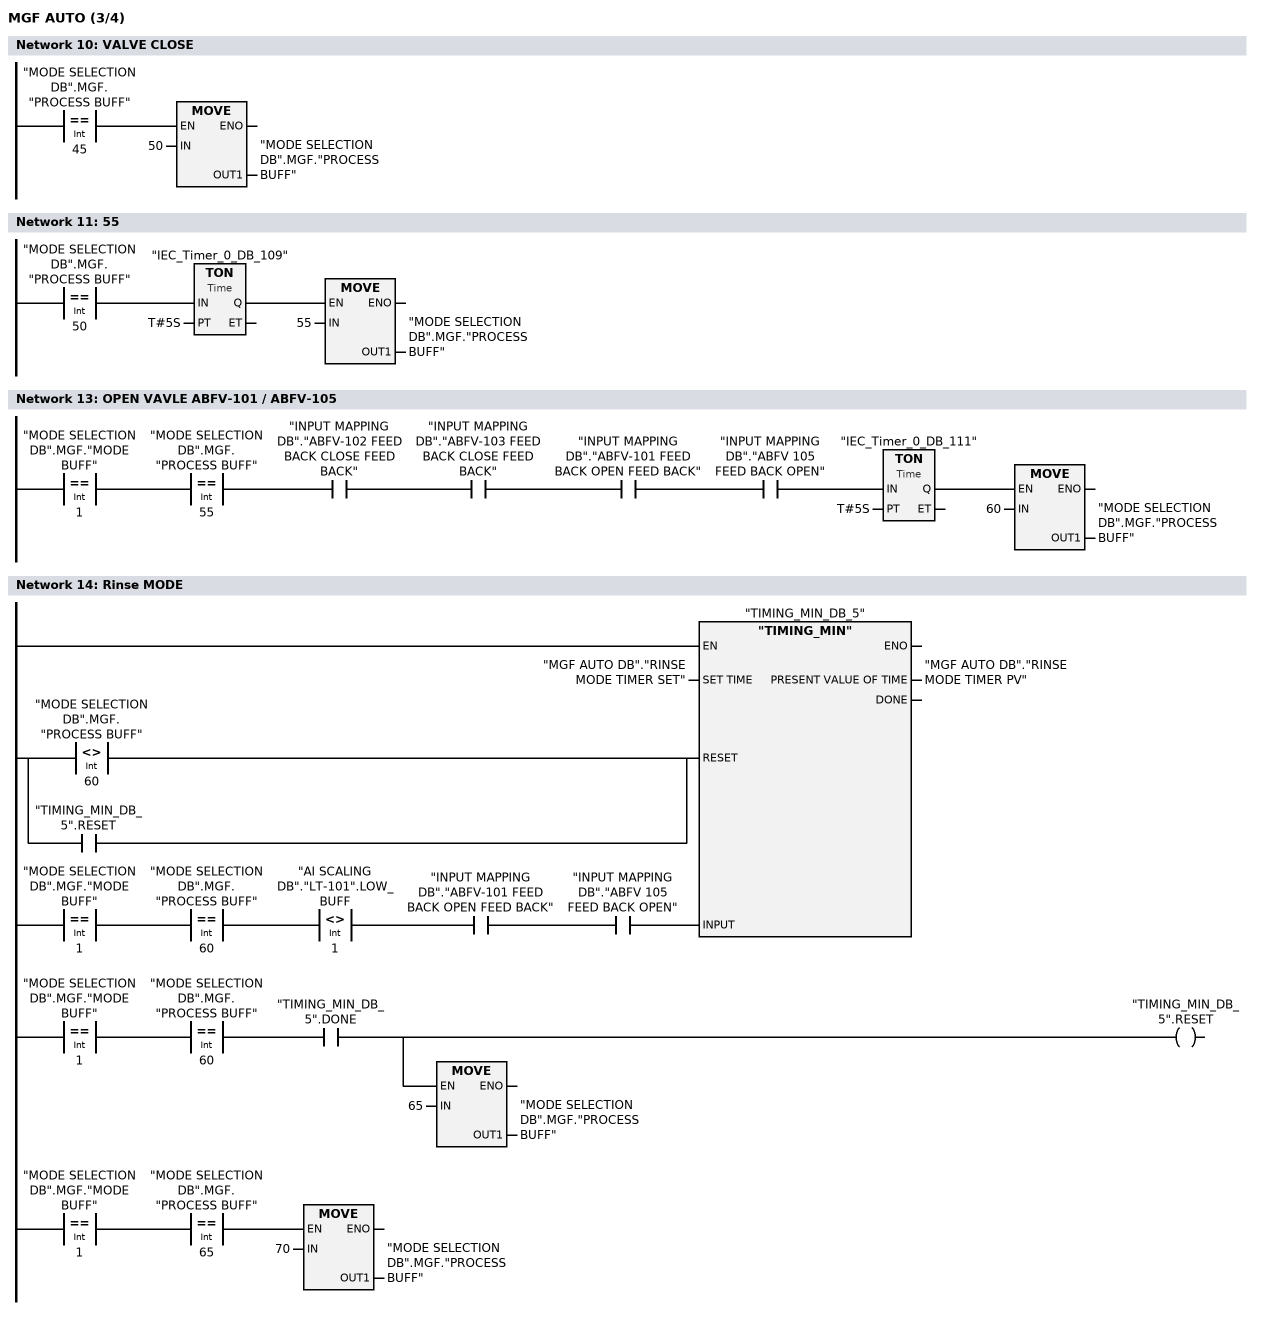
   RUNG wire#powerrail
      { S7_Templates := "SrcType := Int" } EQ_Contact(in1 := "MODE SELECTION DB".MGF."PROCESS BUFF", in2 := 45)
      Move(in := 50, out1 => "MODE SELECTION DB".MGF."PROCESS BUFF")
   END_RUNG
   // the same network as SCL:
   IF "MODE SELECTION DB".MGF."PROCESS BUFF" = 45 THEN "MODE SELECTION DB".MGF."PROCESS BUFF" := 50; END_IF;
END_REGION

REGION Network 11: 55
   RUNG wire#powerrail
      { S7_Templates := "SrcType := Int" } EQ_Contact(in1 := "MODE SELECTION DB".MGF."PROCESS BUFF", in2 := 50)
      { S7_Templates := "time_type := Time" } "IEC_Timer_0_DB_109".TON(pt := T#5S, et =>)
      Move(in := 55, out1 => "MODE SELECTION DB".MGF."PROCESS BUFF")
   END_RUNG
   // the same network as SCL:
   "IEC_Timer_0_DB_109".TON(IN := "MODE SELECTION DB".MGF."PROCESS BUFF" = 50, PT := T#5S);
   IF "IEC_Timer_0_DB_109".Q THEN "MODE SELECTION DB".MGF."PROCESS BUFF" := 55; END_IF;
END_REGION

REGION Network 13: OPEN VAVLE ABFV-101 / ABFV-105
   RUNG wire#powerrail
      { S7_Templates := "SrcType := Int" } EQ_Contact(in1 := "MODE SELECTION DB".MGF."MODE BUFF", in2 := 1)
      { S7_Templates := "SrcType := Int" } EQ_Contact(in1 := "MODE SELECTION DB".MGF."PROCESS BUFF", in2 := 55)
      Contact( "INPUT MAPPING DB"."ABFV-102 FEED BACK CLOSE FEED BACK" )
      Contact( "INPUT MAPPING DB"."ABFV-103 FEED BACK CLOSE FEED BACK" )
      Contact( "INPUT MAPPING DB"."ABFV-101 FEED BACK OPEN FEED BACK" )
      Contact( "INPUT MAPPING DB"."ABFV 105 FEED BACK OPEN" )
      { S7_Templates := "time_type := Time" } "IEC_Timer_0_DB_111".TON(pt := T#5S, et =>)
      Move(in := 60, out1 => "MODE SELECTION DB".MGF."PROCESS BUFF")
   END_RUNG
   // the same network as SCL:
   "IEC_Timer_0_DB_111".TON(IN := ("MODE SELECTION DB".MGF."MODE BUFF" = 1) AND ("MODE SELECTION DB".MGF."PROCESS BUFF" = 55) AND "INPUT MAPPING DB"."ABFV-102 FEED BACK CLOSE FEED BACK" AND "INPUT MAPPING DB"."ABFV-103 FEED BACK CLOSE FEED BACK" AND "INPUT MAPPING DB"."ABFV-101 FEED BACK OPEN FEED BACK" AND "INPUT MAPPING DB"."ABFV 105 FEED BACK OPEN",
                           PT := T#5S);
   IF "IEC_Timer_0_DB_111".Q THEN "MODE SELECTION DB".MGF."PROCESS BUFF" := 60; END_IF;
END_REGION

REGION Network 14: Rinse MODE
   RUNG wire#powerrail
      "TIMING_MIN_DB_5"(RESET := wire#w1, INPUT := wire#w2, "SET TIME" := "MGF AUTO DB"."RINSE MODE TIMER SET", "PRESENT VALUE OF TIME" => "MGF AUTO DB"."RINSE MODE TIMER PV", DONE =>)
   END_RUNG
   RUNG wire#powerrail
      { S7_Templates := "SrcType := Int" } NE_Contact(in1 := "MODE SELECTION DB".MGF."PROCESS BUFF", in2 := 60)
   END_RUNG wire#w1
   RUNG wire#powerrail
      Contact( "TIMING_MIN_DB_5".RESET )
   END_RUNG wire#w1
   RUNG wire#powerrail
      { S7_Templates := "SrcType := Int" } EQ_Contact(in1 := "MODE SELECTION DB".MGF."MODE BUFF", in2 := 1)
      { S7_Templates := "SrcType := Int" } EQ_Contact(in1 := "MODE SELECTION DB".MGF."PROCESS BUFF", in2 := 60)
      { S7_Templates := "SrcType := Int" } NE_Contact(in1 := "AI SCALING DB"."LT-101".LOW_BUFF, in2 := 1)
      Contact( "INPUT MAPPING DB"."ABFV-101 FEED BACK OPEN FEED BACK" )
      Contact( "INPUT MAPPING DB"."ABFV 105 FEED BACK OPEN" )
   END_RUNG wire#w2
   RUNG wire#powerrail
      { S7_Templates := "SrcType := Int" } EQ_Contact(in1 := "MODE SELECTION DB".MGF."MODE BUFF", in2 := 1)
      { S7_Templates := "SrcType := Int" } EQ_Contact(in1 := "MODE SELECTION DB".MGF."PROCESS BUFF", in2 := 60)
      Contact( "TIMING_MIN_DB_5".DONE )
      wire#w3
      Coil( "TIMING_MIN_DB_5".RESET )
   END_RUNG
   RUNG wire#w3
      Move(in := 65, out1 => "MODE SELECTION DB".MGF."PROCESS BUFF")
   END_RUNG
   RUNG wire#powerrail
      { S7_Templates := "SrcType := Int" } EQ_Contact(in1 := "MODE SELECTION DB".MGF."MODE BUFF", in2 := 1)
      { S7_Templates := "SrcType := Int" } EQ_Contact(in1 := "MODE SELECTION DB".MGF."PROCESS BUFF", in2 := 65)
      Move(in := 70, out1 => "MODE SELECTION DB".MGF."PROCESS BUFF")
   END_RUNG
   // the same network as SCL:
   "TIMING_MIN_DB_5"("SET TIME" := "MGF AUTO DB"."RINSE MODE TIMER SET",   // "TIMING_MIN"
                     RESET := ("MODE SELECTION DB".MGF."PROCESS BUFF" <> 60) OR "TIMING_MIN_DB_5".RESET,
                     INPUT := ("MODE SELECTION DB".MGF."MODE BUFF" = 1) AND ("MODE SELECTION DB".MGF."PROCESS BUFF" = 60) AND ("AI SCALING DB"."LT-101".LOW_BUFF <> 1) AND "INPUT MAPPING DB"."ABFV-101 FEED BACK OPEN FEED BACK" AND "INPUT MAPPING DB"."ABFV 105 FEED BACK OPEN",
                     "PRESENT VALUE OF TIME" => "MGF AUTO DB"."RINSE MODE TIMER PV");
   "TIMING_MIN_DB_5".RESET := ("MODE SELECTION DB".MGF."MODE BUFF" = 1) AND ("MODE SELECTION DB".MGF."PROCESS BUFF" = 60) AND "TIMING_MIN_DB_5".DONE;
   IF "TIMING_MIN_DB_5".RESET THEN "MODE SELECTION DB".MGF."PROCESS BUFF" := 65; END_IF;
   IF ("MODE SELECTION DB".MGF."MODE BUFF" = 1) AND ("MODE SELECTION DB".MGF."PROCESS BUFF" = 65) THEN
       "MODE SELECTION DB".MGF."PROCESS BUFF" := 70;
   END_IF;
END_REGION

REGION Network 15: VALVE CLOSE
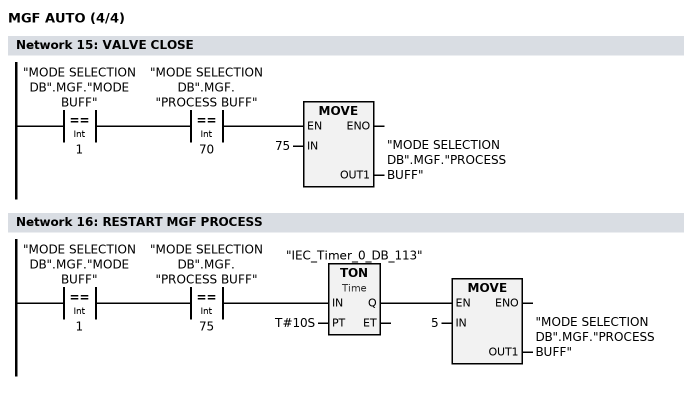
   RUNG wire#powerrail
      { S7_Templates := "SrcType := Int" } EQ_Contact(in1 := "MODE SELECTION DB".MGF."MODE BUFF", in2 := 1)
      { S7_Templates := "SrcType := Int" } EQ_Contact(in1 := "MODE SELECTION DB".MGF."PROCESS BUFF", in2 := 70)
      Move(in := 75, out1 => "MODE SELECTION DB".MGF."PROCESS BUFF")
   END_RUNG
   // the same network as SCL:
   IF ("MODE SELECTION DB".MGF."MODE BUFF" = 1) AND ("MODE SELECTION DB".MGF."PROCESS BUFF" = 70) THEN
       "MODE SELECTION DB".MGF."PROCESS BUFF" := 75;
   END_IF;
END_REGION

REGION Network 16: RESTART MGF PROCESS
   RUNG wire#powerrail
      { S7_Templates := "SrcType := Int" } EQ_Contact(in1 := "MODE SELECTION DB".MGF."MODE BUFF", in2 := 1)
      { S7_Templates := "SrcType := Int" } EQ_Contact(in1 := "MODE SELECTION DB".MGF."PROCESS BUFF", in2 := 75)
      { S7_Templates := "time_type := Time" } "IEC_Timer_0_DB_113".TON(pt := T#10S, et =>)
      Move(in := 5, out1 => "MODE SELECTION DB".MGF."PROCESS BUFF")
   END_RUNG
   // the same network as SCL:
   "IEC_Timer_0_DB_113".TON(IN := ("MODE SELECTION DB".MGF."MODE BUFF" = 1) AND ("MODE SELECTION DB".MGF."PROCESS BUFF" = 75),
                           PT := T#10S);
   IF "IEC_Timer_0_DB_113".Q THEN "MODE SELECTION DB".MGF."PROCESS BUFF" := 5; END_IF;
END_REGION
END_FUNCTION

FUNCTION "UF" : Void   // FC12, LAD
{ S7_Optimized_Access := 'TRUE' }
// stored: SetENOAutomatically false
   VAR_TEMP   // added for the SCL form of the ladder/FBD networks
      _w1 : Bool;
      _w2 : Bool;
   END_VAR
BEGIN

REGION Network 1: ABFV-201 OPEN F/B
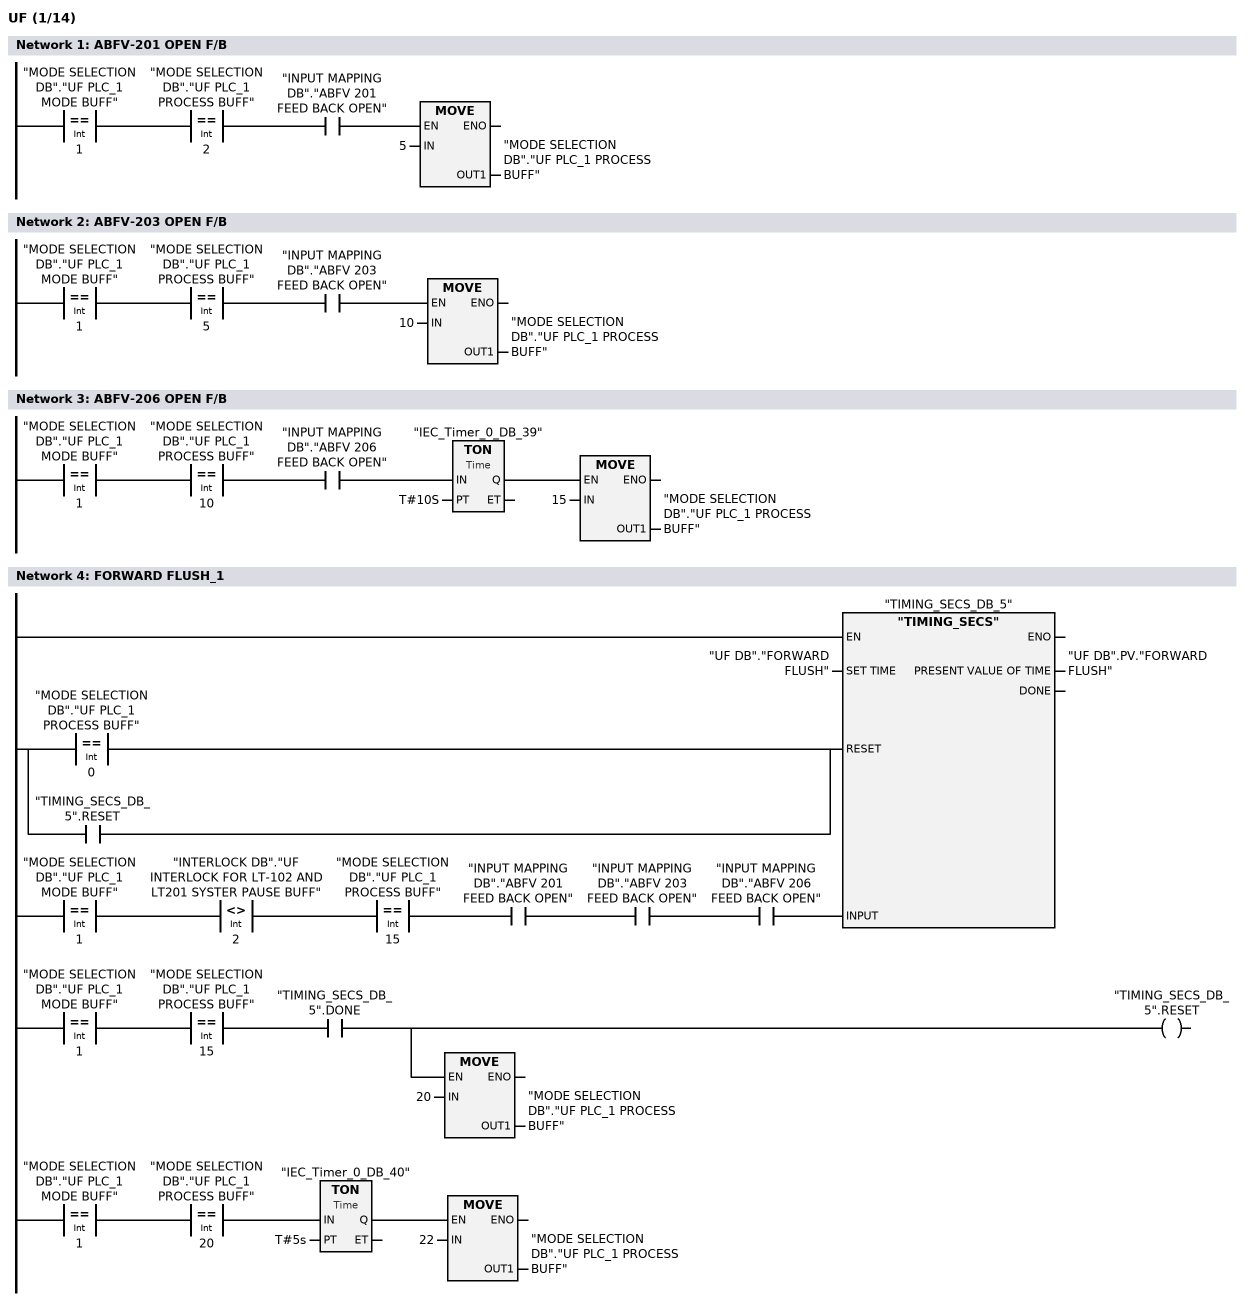
   RUNG wire#powerrail
      { S7_Templates := "SrcType := Int" } EQ_Contact(in1 := "MODE SELECTION DB"."UF PLC_1 MODE BUFF", in2 := 1)
      { S7_Templates := "SrcType := Int" } EQ_Contact(in1 := "MODE SELECTION DB"."UF PLC_1 PROCESS BUFF", in2 := 2)
      Contact( "INPUT MAPPING DB"."ABFV 201 FEED BACK OPEN" )
      Move(in := 5, out1 => "MODE SELECTION DB"."UF PLC_1 PROCESS BUFF")
   END_RUNG
   // the same network as SCL:
   IF ("MODE SELECTION DB"."UF PLC_1 MODE BUFF" = 1) AND ("MODE SELECTION DB"."UF PLC_1 PROCESS BUFF" = 2) AND "INPUT MAPPING DB"."ABFV 201 FEED BACK OPEN" THEN
       "MODE SELECTION DB"."UF PLC_1 PROCESS BUFF" := 5;
   END_IF;
END_REGION

REGION Network 2: ABFV-203 OPEN F/B
   RUNG wire#powerrail
      { S7_Templates := "SrcType := Int" } EQ_Contact(in1 := "MODE SELECTION DB"."UF PLC_1 MODE BUFF", in2 := 1)
      { S7_Templates := "SrcType := Int" } EQ_Contact(in1 := "MODE SELECTION DB"."UF PLC_1 PROCESS BUFF", in2 := 5)
      Contact( "INPUT MAPPING DB"."ABFV 203 FEED BACK OPEN" )
      Move(in := 10, out1 => "MODE SELECTION DB"."UF PLC_1 PROCESS BUFF")
   END_RUNG
   // the same network as SCL:
   IF ("MODE SELECTION DB"."UF PLC_1 MODE BUFF" = 1) AND ("MODE SELECTION DB"."UF PLC_1 PROCESS BUFF" = 5) AND "INPUT MAPPING DB"."ABFV 203 FEED BACK OPEN" THEN
       "MODE SELECTION DB"."UF PLC_1 PROCESS BUFF" := 10;
   END_IF;
END_REGION

REGION Network 3: ABFV-206 OPEN F/B
   RUNG wire#powerrail
      { S7_Templates := "SrcType := Int" } EQ_Contact(in1 := "MODE SELECTION DB"."UF PLC_1 MODE BUFF", in2 := 1)
      { S7_Templates := "SrcType := Int" } EQ_Contact(in1 := "MODE SELECTION DB"."UF PLC_1 PROCESS BUFF", in2 := 10)
      Contact( "INPUT MAPPING DB"."ABFV 206 FEED BACK OPEN" )
      { S7_Templates := "time_type := Time" } "IEC_Timer_0_DB_39".TON(pt := T#10S, et =>)
      Move(in := 15, out1 => "MODE SELECTION DB"."UF PLC_1 PROCESS BUFF")
   END_RUNG
   // the same network as SCL:
   "IEC_Timer_0_DB_39".TON(IN := ("MODE SELECTION DB"."UF PLC_1 MODE BUFF" = 1) AND ("MODE SELECTION DB"."UF PLC_1 PROCESS BUFF" = 10) AND "INPUT MAPPING DB"."ABFV 206 FEED BACK OPEN",
                           PT := T#10S);
   IF "IEC_Timer_0_DB_39".Q THEN "MODE SELECTION DB"."UF PLC_1 PROCESS BUFF" := 15; END_IF;
END_REGION

REGION Network 4: FORWARD FLUSH_1
   RUNG wire#powerrail
      "TIMING_SECS_DB_5"(RESET := wire#w1, INPUT := wire#w2, "SET TIME" := "UF DB"."FORWARD FLUSH", "PRESENT VALUE OF TIME" => "UF DB".PV."FORWARD FLUSH", DONE =>)
   END_RUNG
   RUNG wire#powerrail
      { S7_Templates := "SrcType := Int" } EQ_Contact(in1 := "MODE SELECTION DB"."UF PLC_1 PROCESS BUFF", in2 := 0)
   END_RUNG wire#w1
   RUNG wire#powerrail
      Contact( "TIMING_SECS_DB_5".RESET )
   END_RUNG wire#w1
   RUNG wire#powerrail
      { S7_Templates := "SrcType := Int" } EQ_Contact(in1 := "MODE SELECTION DB"."UF PLC_1 MODE BUFF", in2 := 1)
      { S7_Templates := "SrcType := Int" } NE_Contact(in1 := "INTERLOCK DB"."UF INTERLOCK FOR LT-102 AND LT201 SYSTER PAUSE BUFF", in2 := 2)
      { S7_Templates := "SrcType := Int" } EQ_Contact(in1 := "MODE SELECTION DB"."UF PLC_1 PROCESS BUFF", in2 := 15)
      Contact( "INPUT MAPPING DB"."ABFV 201 FEED BACK OPEN" )
      Contact( "INPUT MAPPING DB"."ABFV 203 FEED BACK OPEN" )
      Contact( "INPUT MAPPING DB"."ABFV 206 FEED BACK OPEN" )
   END_RUNG wire#w2
   RUNG wire#powerrail
      { S7_Templates := "SrcType := Int" } EQ_Contact(in1 := "MODE SELECTION DB"."UF PLC_1 MODE BUFF", in2 := 1)
      { S7_Templates := "SrcType := Int" } EQ_Contact(in1 := "MODE SELECTION DB"."UF PLC_1 PROCESS BUFF", in2 := 15)
      Contact( "TIMING_SECS_DB_5".DONE )
      wire#w3
      Coil( "TIMING_SECS_DB_5".RESET )
   END_RUNG
   RUNG wire#w3
      Move(in := 20, out1 => "MODE SELECTION DB"."UF PLC_1 PROCESS BUFF")
   END_RUNG
   RUNG wire#powerrail
      { S7_Templates := "SrcType := Int" } EQ_Contact(in1 := "MODE SELECTION DB"."UF PLC_1 MODE BUFF", in2 := 1)
      { S7_Templates := "SrcType := Int" } EQ_Contact(in1 := "MODE SELECTION DB"."UF PLC_1 PROCESS BUFF", in2 := 20)
      { S7_Templates := "time_type := Time" } "IEC_Timer_0_DB_40".TON(pt := T#5s, et =>)
      Move(in := 22, out1 => "MODE SELECTION DB"."UF PLC_1 PROCESS BUFF")
   END_RUNG
   // the same network as SCL:
   "TIMING_SECS_DB_5"("SET TIME" := "UF DB"."FORWARD FLUSH",   // "TIMING_SECS"
                      RESET := ("MODE SELECTION DB"."UF PLC_1 PROCESS BUFF" = 0) OR "TIMING_SECS_DB_5".RESET,
                      INPUT := ("MODE SELECTION DB"."UF PLC_1 MODE BUFF" = 1) AND ("INTERLOCK DB"."UF INTERLOCK FOR LT-102 AND LT201 SYSTER PAUSE BUFF" <> 2) AND ("MODE SELECTION DB"."UF PLC_1 PROCESS BUFF" = 15) AND "INPUT MAPPING DB"."ABFV 201 FEED BACK OPEN" AND "INPUT MAPPING DB"."ABFV 203 FEED BACK OPEN" AND "INPUT MAPPING DB"."ABFV 206 FEED BACK OPEN",
                      "PRESENT VALUE OF TIME" => "UF DB".PV."FORWARD FLUSH");
   "TIMING_SECS_DB_5".RESET := ("MODE SELECTION DB"."UF PLC_1 MODE BUFF" = 1) AND ("MODE SELECTION DB"."UF PLC_1 PROCESS BUFF" = 15) AND "TIMING_SECS_DB_5".DONE;
   IF "TIMING_SECS_DB_5".RESET THEN "MODE SELECTION DB"."UF PLC_1 PROCESS BUFF" := 20; END_IF;
   "IEC_Timer_0_DB_40".TON(IN := ("MODE SELECTION DB"."UF PLC_1 MODE BUFF" = 1) AND ("MODE SELECTION DB"."UF PLC_1 PROCESS BUFF" = 20),
                           PT := T#5s);
   IF "IEC_Timer_0_DB_40".Q THEN "MODE SELECTION DB"."UF PLC_1 PROCESS BUFF" := 22; END_IF;
END_REGION

REGION Network 5: OPEN ALL VALVE NEXT PROCESS
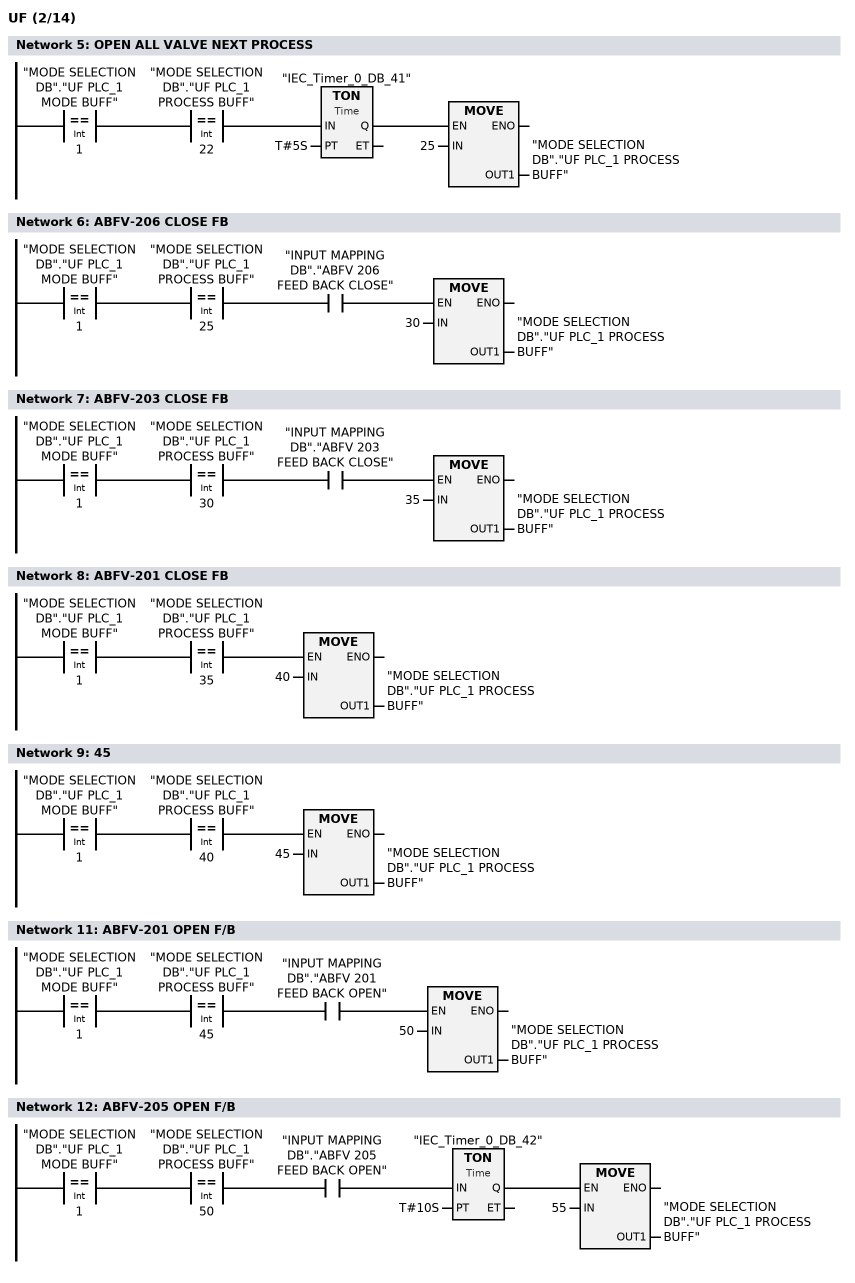
   RUNG wire#powerrail
      { S7_Templates := "SrcType := Int" } EQ_Contact(in1 := "MODE SELECTION DB"."UF PLC_1 MODE BUFF", in2 := 1)
      { S7_Templates := "SrcType := Int" } EQ_Contact(in1 := "MODE SELECTION DB"."UF PLC_1 PROCESS BUFF", in2 := 22)
      { S7_Templates := "time_type := Time" } "IEC_Timer_0_DB_41".TON(pt := T#5S, et =>)
      Move(in := 25, out1 => "MODE SELECTION DB"."UF PLC_1 PROCESS BUFF")
   END_RUNG
   // the same network as SCL:
   "IEC_Timer_0_DB_41".TON(IN := ("MODE SELECTION DB"."UF PLC_1 MODE BUFF" = 1) AND ("MODE SELECTION DB"."UF PLC_1 PROCESS BUFF" = 22),
                           PT := T#5S);
   IF "IEC_Timer_0_DB_41".Q THEN "MODE SELECTION DB"."UF PLC_1 PROCESS BUFF" := 25; END_IF;
END_REGION

REGION Network 6: ABFV-206 CLOSE FB
   RUNG wire#powerrail
      { S7_Templates := "SrcType := Int" } EQ_Contact(in1 := "MODE SELECTION DB"."UF PLC_1 MODE BUFF", in2 := 1)
      { S7_Templates := "SrcType := Int" } EQ_Contact(in1 := "MODE SELECTION DB"."UF PLC_1 PROCESS BUFF", in2 := 25)
      Contact( "INPUT MAPPING DB"."ABFV 206 FEED BACK CLOSE" )
      Move(in := 30, out1 => "MODE SELECTION DB"."UF PLC_1 PROCESS BUFF")
   END_RUNG
   // the same network as SCL:
   IF ("MODE SELECTION DB"."UF PLC_1 MODE BUFF" = 1) AND ("MODE SELECTION DB"."UF PLC_1 PROCESS BUFF" = 25) AND "INPUT MAPPING DB"."ABFV 206 FEED BACK CLOSE" THEN
       "MODE SELECTION DB"."UF PLC_1 PROCESS BUFF" := 30;
   END_IF;
END_REGION

REGION Network 7: ABFV-203 CLOSE FB
   RUNG wire#powerrail
      { S7_Templates := "SrcType := Int" } EQ_Contact(in1 := "MODE SELECTION DB"."UF PLC_1 MODE BUFF", in2 := 1)
      { S7_Templates := "SrcType := Int" } EQ_Contact(in1 := "MODE SELECTION DB"."UF PLC_1 PROCESS BUFF", in2 := 30)
      Contact( "INPUT MAPPING DB"."ABFV 203 FEED BACK CLOSE" )
      Move(in := 35, out1 => "MODE SELECTION DB"."UF PLC_1 PROCESS BUFF")
   END_RUNG
   // the same network as SCL:
   IF ("MODE SELECTION DB"."UF PLC_1 MODE BUFF" = 1) AND ("MODE SELECTION DB"."UF PLC_1 PROCESS BUFF" = 30) AND "INPUT MAPPING DB"."ABFV 203 FEED BACK CLOSE" THEN
       "MODE SELECTION DB"."UF PLC_1 PROCESS BUFF" := 35;
   END_IF;
END_REGION

REGION Network 8: ABFV-201 CLOSE FB
   RUNG wire#powerrail
      { S7_Templates := "SrcType := Int" } EQ_Contact(in1 := "MODE SELECTION DB"."UF PLC_1 MODE BUFF", in2 := 1)
      { S7_Templates := "SrcType := Int" } EQ_Contact(in1 := "MODE SELECTION DB"."UF PLC_1 PROCESS BUFF", in2 := 35)
      Move(in := 40, out1 => "MODE SELECTION DB"."UF PLC_1 PROCESS BUFF")
   END_RUNG
   // the same network as SCL:
   IF ("MODE SELECTION DB"."UF PLC_1 MODE BUFF" = 1) AND ("MODE SELECTION DB"."UF PLC_1 PROCESS BUFF" = 35) THEN
       "MODE SELECTION DB"."UF PLC_1 PROCESS BUFF" := 40;
   END_IF;
END_REGION

REGION Network 9: 45
   RUNG wire#powerrail
      { S7_Templates := "SrcType := Int" } EQ_Contact(in1 := "MODE SELECTION DB"."UF PLC_1 MODE BUFF", in2 := 1)
      { S7_Templates := "SrcType := Int" } EQ_Contact(in1 := "MODE SELECTION DB"."UF PLC_1 PROCESS BUFF", in2 := 40)
      Move(in := 45, out1 => "MODE SELECTION DB"."UF PLC_1 PROCESS BUFF")
   END_RUNG
   // the same network as SCL:
   IF ("MODE SELECTION DB"."UF PLC_1 MODE BUFF" = 1) AND ("MODE SELECTION DB"."UF PLC_1 PROCESS BUFF" = 40) THEN
       "MODE SELECTION DB"."UF PLC_1 PROCESS BUFF" := 45;
   END_IF;
END_REGION

REGION Network 11: ABFV-201 OPEN F/B
   RUNG wire#powerrail
      { S7_Templates := "SrcType := Int" } EQ_Contact(in1 := "MODE SELECTION DB"."UF PLC_1 MODE BUFF", in2 := 1)
      { S7_Templates := "SrcType := Int" } EQ_Contact(in1 := "MODE SELECTION DB"."UF PLC_1 PROCESS BUFF", in2 := 45)
      Contact( "INPUT MAPPING DB"."ABFV 201 FEED BACK OPEN" )
      Move(in := 50, out1 => "MODE SELECTION DB"."UF PLC_1 PROCESS BUFF")
   END_RUNG
   // the same network as SCL:
   IF ("MODE SELECTION DB"."UF PLC_1 MODE BUFF" = 1) AND ("MODE SELECTION DB"."UF PLC_1 PROCESS BUFF" = 45) AND "INPUT MAPPING DB"."ABFV 201 FEED BACK OPEN" THEN
       "MODE SELECTION DB"."UF PLC_1 PROCESS BUFF" := 50;
   END_IF;
END_REGION

REGION Network 12: ABFV-205 OPEN F/B
   RUNG wire#powerrail
      { S7_Templates := "SrcType := Int" } EQ_Contact(in1 := "MODE SELECTION DB"."UF PLC_1 MODE BUFF", in2 := 1)
      { S7_Templates := "SrcType := Int" } EQ_Contact(in1 := "MODE SELECTION DB"."UF PLC_1 PROCESS BUFF", in2 := 50)
      Contact( "INPUT MAPPING DB"."ABFV 205 FEED BACK OPEN" )
      { S7_Templates := "time_type := Time" } "IEC_Timer_0_DB_42".TON(pt := T#10S, et =>)
      Move(in := 55, out1 => "MODE SELECTION DB"."UF PLC_1 PROCESS BUFF")
   END_RUNG
   // the same network as SCL:
   "IEC_Timer_0_DB_42".TON(IN := ("MODE SELECTION DB"."UF PLC_1 MODE BUFF" = 1) AND ("MODE SELECTION DB"."UF PLC_1 PROCESS BUFF" = 50) AND "INPUT MAPPING DB"."ABFV 205 FEED BACK OPEN",
                           PT := T#10S);
   IF "IEC_Timer_0_DB_42".Q THEN "MODE SELECTION DB"."UF PLC_1 PROCESS BUFF" := 55; END_IF;
END_REGION

REGION Network 13: FILTRATION MODE
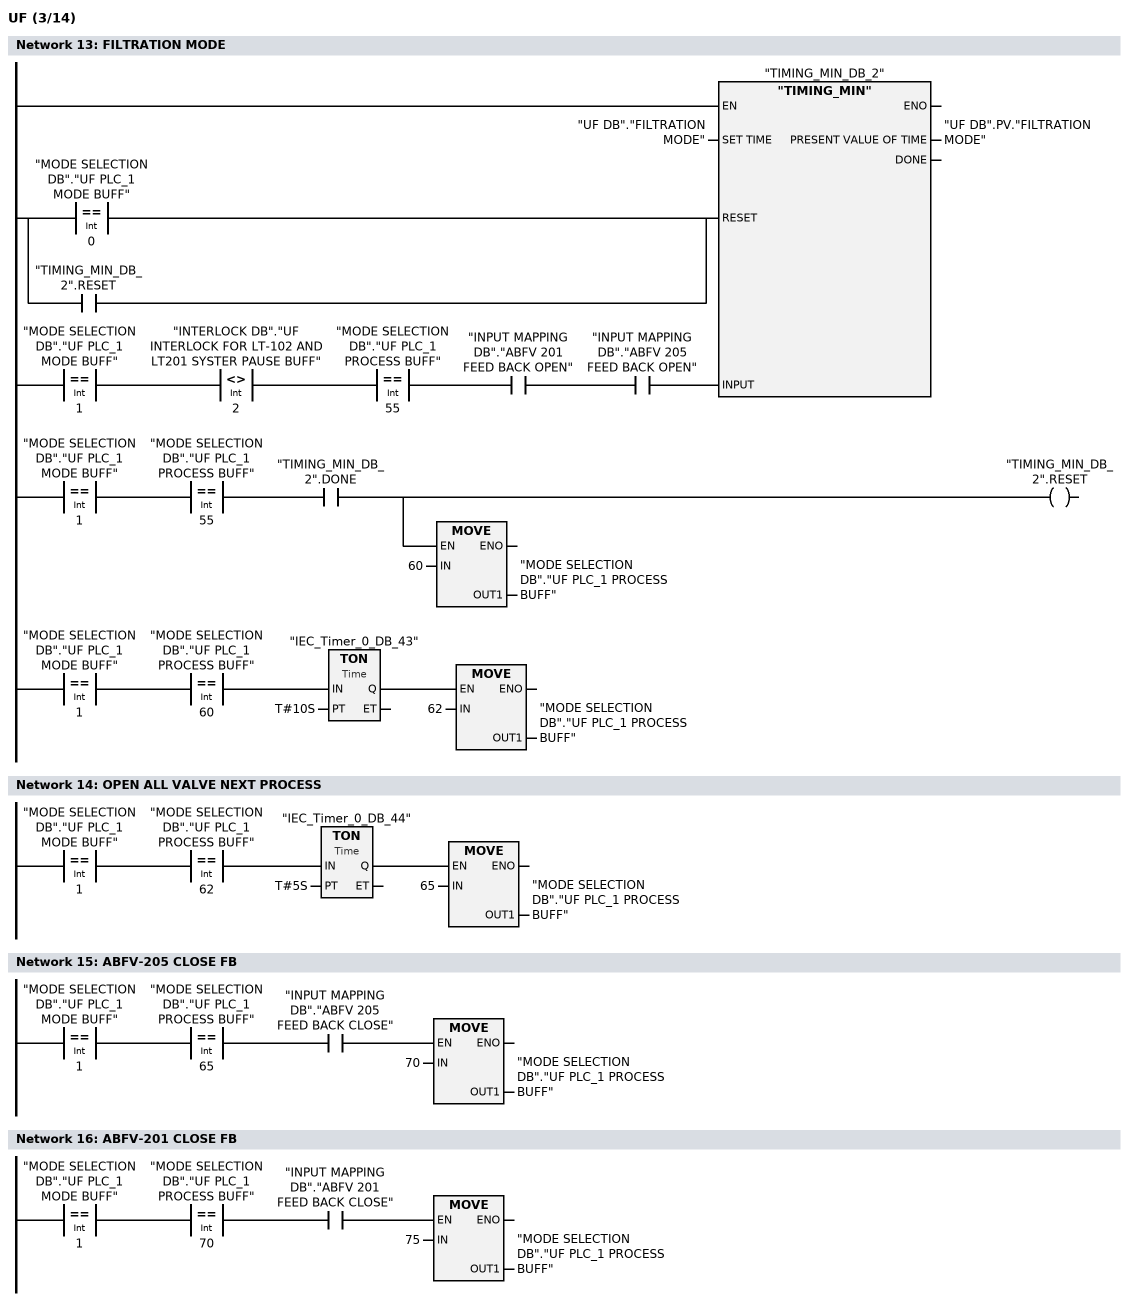
   RUNG wire#powerrail
      "TIMING_MIN_DB_2"(RESET := wire#w1, INPUT := wire#w2, "SET TIME" := "UF DB"."FILTRATION MODE", "PRESENT VALUE OF TIME" => "UF DB".PV."FILTRATION MODE", DONE =>)
   END_RUNG
   RUNG wire#powerrail
      { S7_Templates := "SrcType := Int" } EQ_Contact(in1 := "MODE SELECTION DB"."UF PLC_1 MODE BUFF", in2 := 0)
   END_RUNG wire#w1
   RUNG wire#powerrail
      Contact( "TIMING_MIN_DB_2".RESET )
   END_RUNG wire#w1
   RUNG wire#powerrail
      { S7_Templates := "SrcType := Int" } EQ_Contact(in1 := "MODE SELECTION DB"."UF PLC_1 MODE BUFF", in2 := 1)
      { S7_Templates := "SrcType := Int" } NE_Contact(in1 := "INTERLOCK DB"."UF INTERLOCK FOR LT-102 AND LT201 SYSTER PAUSE BUFF", in2 := 2)
      { S7_Templates := "SrcType := Int" } EQ_Contact(in1 := "MODE SELECTION DB"."UF PLC_1 PROCESS BUFF", in2 := 55)
      Contact( "INPUT MAPPING DB"."ABFV 201 FEED BACK OPEN" )
      Contact( "INPUT MAPPING DB"."ABFV 205 FEED BACK OPEN" )
   END_RUNG wire#w2
   RUNG wire#powerrail
      { S7_Templates := "SrcType := Int" } EQ_Contact(in1 := "MODE SELECTION DB"."UF PLC_1 MODE BUFF", in2 := 1)
      { S7_Templates := "SrcType := Int" } EQ_Contact(in1 := "MODE SELECTION DB"."UF PLC_1 PROCESS BUFF", in2 := 55)
      Contact( "TIMING_MIN_DB_2".DONE )
      wire#w3
      Coil( "TIMING_MIN_DB_2".RESET )
   END_RUNG
   RUNG wire#w3
      Move(in := 60, out1 => "MODE SELECTION DB"."UF PLC_1 PROCESS BUFF")
   END_RUNG
   RUNG wire#powerrail
      { S7_Templates := "SrcType := Int" } EQ_Contact(in1 := "MODE SELECTION DB"."UF PLC_1 MODE BUFF", in2 := 1)
      { S7_Templates := "SrcType := Int" } EQ_Contact(in1 := "MODE SELECTION DB"."UF PLC_1 PROCESS BUFF", in2 := 60)
      { S7_Templates := "time_type := Time" } "IEC_Timer_0_DB_43".TON(pt := T#10S, et =>)
      Move(in := 62, out1 => "MODE SELECTION DB"."UF PLC_1 PROCESS BUFF")
   END_RUNG
   // the same network as SCL:
   "TIMING_MIN_DB_2"("SET TIME" := "UF DB"."FILTRATION MODE",   // "TIMING_MIN"
                     RESET := ("MODE SELECTION DB"."UF PLC_1 MODE BUFF" = 0) OR "TIMING_MIN_DB_2".RESET,
                     INPUT := ("MODE SELECTION DB"."UF PLC_1 MODE BUFF" = 1) AND ("INTERLOCK DB"."UF INTERLOCK FOR LT-102 AND LT201 SYSTER PAUSE BUFF" <> 2) AND ("MODE SELECTION DB"."UF PLC_1 PROCESS BUFF" = 55) AND "INPUT MAPPING DB"."ABFV 201 FEED BACK OPEN" AND "INPUT MAPPING DB"."ABFV 205 FEED BACK OPEN",
                     "PRESENT VALUE OF TIME" => "UF DB".PV."FILTRATION MODE");
   "TIMING_MIN_DB_2".RESET := ("MODE SELECTION DB"."UF PLC_1 MODE BUFF" = 1) AND ("MODE SELECTION DB"."UF PLC_1 PROCESS BUFF" = 55) AND "TIMING_MIN_DB_2".DONE;
   IF "TIMING_MIN_DB_2".RESET THEN "MODE SELECTION DB"."UF PLC_1 PROCESS BUFF" := 60; END_IF;
   "IEC_Timer_0_DB_43".TON(IN := ("MODE SELECTION DB"."UF PLC_1 MODE BUFF" = 1) AND ("MODE SELECTION DB"."UF PLC_1 PROCESS BUFF" = 60),
                           PT := T#10S);
   IF "IEC_Timer_0_DB_43".Q THEN "MODE SELECTION DB"."UF PLC_1 PROCESS BUFF" := 62; END_IF;
END_REGION

REGION Network 14: OPEN ALL VALVE NEXT PROCESS
   RUNG wire#powerrail
      { S7_Templates := "SrcType := Int" } EQ_Contact(in1 := "MODE SELECTION DB"."UF PLC_1 MODE BUFF", in2 := 1)
      { S7_Templates := "SrcType := Int" } EQ_Contact(in1 := "MODE SELECTION DB"."UF PLC_1 PROCESS BUFF", in2 := 62)
      { S7_Templates := "time_type := Time" } "IEC_Timer_0_DB_44".TON(pt := T#5S, et =>)
      Move(in := 65, out1 => "MODE SELECTION DB"."UF PLC_1 PROCESS BUFF")
   END_RUNG
   // the same network as SCL:
   "IEC_Timer_0_DB_44".TON(IN := ("MODE SELECTION DB"."UF PLC_1 MODE BUFF" = 1) AND ("MODE SELECTION DB"."UF PLC_1 PROCESS BUFF" = 62),
                           PT := T#5S);
   IF "IEC_Timer_0_DB_44".Q THEN "MODE SELECTION DB"."UF PLC_1 PROCESS BUFF" := 65; END_IF;
END_REGION

REGION Network 15: ABFV-205 CLOSE FB
   RUNG wire#powerrail
      { S7_Templates := "SrcType := Int" } EQ_Contact(in1 := "MODE SELECTION DB"."UF PLC_1 MODE BUFF", in2 := 1)
      { S7_Templates := "SrcType := Int" } EQ_Contact(in1 := "MODE SELECTION DB"."UF PLC_1 PROCESS BUFF", in2 := 65)
      Contact( "INPUT MAPPING DB"."ABFV 205 FEED BACK CLOSE" )
      Move(in := 70, out1 => "MODE SELECTION DB"."UF PLC_1 PROCESS BUFF")
   END_RUNG
   // the same network as SCL:
   IF ("MODE SELECTION DB"."UF PLC_1 MODE BUFF" = 1) AND ("MODE SELECTION DB"."UF PLC_1 PROCESS BUFF" = 65) AND "INPUT MAPPING DB"."ABFV 205 FEED BACK CLOSE" THEN
       "MODE SELECTION DB"."UF PLC_1 PROCESS BUFF" := 70;
   END_IF;
END_REGION

REGION Network 16: ABFV-201 CLOSE FB
   RUNG wire#powerrail
      { S7_Templates := "SrcType := Int" } EQ_Contact(in1 := "MODE SELECTION DB"."UF PLC_1 MODE BUFF", in2 := 1)
      { S7_Templates := "SrcType := Int" } EQ_Contact(in1 := "MODE SELECTION DB"."UF PLC_1 PROCESS BUFF", in2 := 70)
      Contact( "INPUT MAPPING DB"."ABFV 201 FEED BACK CLOSE" )
      Move(in := 75, out1 => "MODE SELECTION DB"."UF PLC_1 PROCESS BUFF")
   END_RUNG
   // the same network as SCL:
   IF ("MODE SELECTION DB"."UF PLC_1 MODE BUFF" = 1) AND ("MODE SELECTION DB"."UF PLC_1 PROCESS BUFF" = 70) AND "INPUT MAPPING DB"."ABFV 201 FEED BACK CLOSE" THEN
       "MODE SELECTION DB"."UF PLC_1 PROCESS BUFF" := 75;
   END_IF;
END_REGION

REGION Network 17: 80
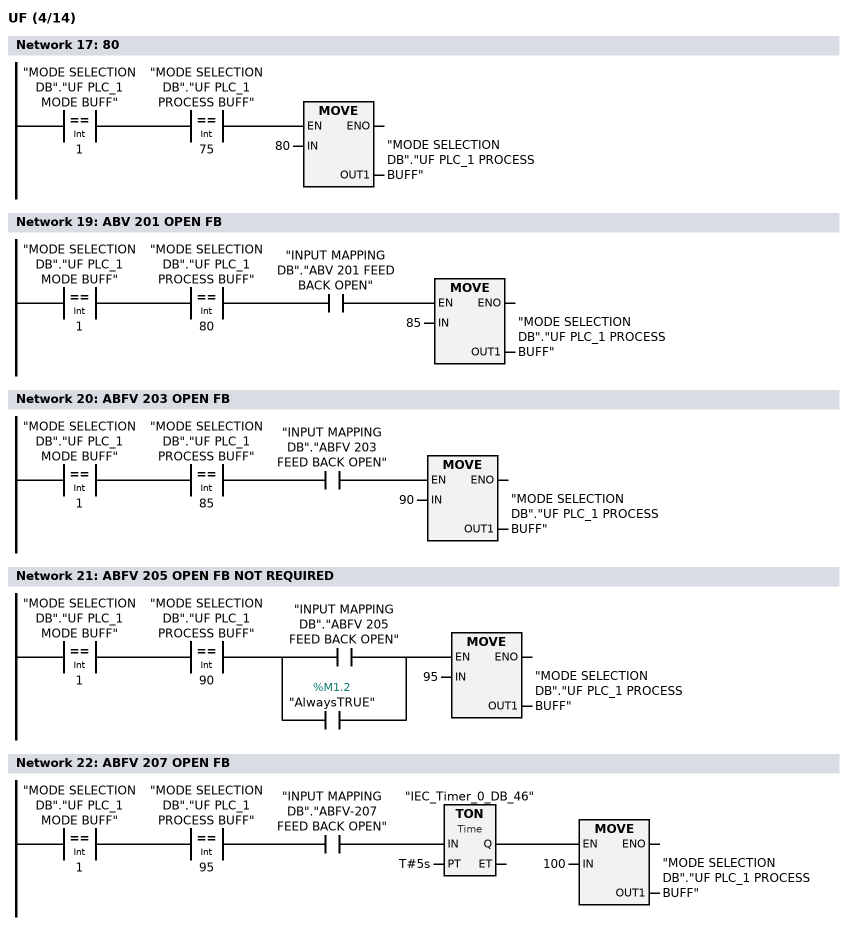
   RUNG wire#powerrail
      { S7_Templates := "SrcType := Int" } EQ_Contact(in1 := "MODE SELECTION DB"."UF PLC_1 MODE BUFF", in2 := 1)
      { S7_Templates := "SrcType := Int" } EQ_Contact(in1 := "MODE SELECTION DB"."UF PLC_1 PROCESS BUFF", in2 := 75)
      Move(in := 80, out1 => "MODE SELECTION DB"."UF PLC_1 PROCESS BUFF")
   END_RUNG
   // the same network as SCL:
   IF ("MODE SELECTION DB"."UF PLC_1 MODE BUFF" = 1) AND ("MODE SELECTION DB"."UF PLC_1 PROCESS BUFF" = 75) THEN
       "MODE SELECTION DB"."UF PLC_1 PROCESS BUFF" := 80;
   END_IF;
END_REGION

REGION Network 19: ABV 201 OPEN FB
   RUNG wire#powerrail
      { S7_Templates := "SrcType := Int" } EQ_Contact(in1 := "MODE SELECTION DB"."UF PLC_1 MODE BUFF", in2 := 1)
      { S7_Templates := "SrcType := Int" } EQ_Contact(in1 := "MODE SELECTION DB"."UF PLC_1 PROCESS BUFF", in2 := 80)
      Contact( "INPUT MAPPING DB"."ABV 201 FEED BACK OPEN" )
      Move(in := 85, out1 => "MODE SELECTION DB"."UF PLC_1 PROCESS BUFF")
   END_RUNG
   // the same network as SCL:
   IF ("MODE SELECTION DB"."UF PLC_1 MODE BUFF" = 1) AND ("MODE SELECTION DB"."UF PLC_1 PROCESS BUFF" = 80) AND "INPUT MAPPING DB"."ABV 201 FEED BACK OPEN" THEN
       "MODE SELECTION DB"."UF PLC_1 PROCESS BUFF" := 85;
   END_IF;
END_REGION

REGION Network 20: ABFV 203 OPEN FB
   RUNG wire#powerrail
      { S7_Templates := "SrcType := Int" } EQ_Contact(in1 := "MODE SELECTION DB"."UF PLC_1 MODE BUFF", in2 := 1)
      { S7_Templates := "SrcType := Int" } EQ_Contact(in1 := "MODE SELECTION DB"."UF PLC_1 PROCESS BUFF", in2 := 85)
      Contact( "INPUT MAPPING DB"."ABFV 203 FEED BACK OPEN" )
      Move(in := 90, out1 => "MODE SELECTION DB"."UF PLC_1 PROCESS BUFF")
   END_RUNG
   // the same network as SCL:
   IF ("MODE SELECTION DB"."UF PLC_1 MODE BUFF" = 1) AND ("MODE SELECTION DB"."UF PLC_1 PROCESS BUFF" = 85) AND "INPUT MAPPING DB"."ABFV 203 FEED BACK OPEN" THEN
       "MODE SELECTION DB"."UF PLC_1 PROCESS BUFF" := 90;
   END_IF;
END_REGION

REGION Network 21: ABFV 205 OPEN FB NOT REQUIRED
   RUNG wire#powerrail
      { S7_Templates := "SrcType := Int" } EQ_Contact(in1 := "MODE SELECTION DB"."UF PLC_1 MODE BUFF", in2 := 1)
      { S7_Templates := "SrcType := Int" } EQ_Contact(in1 := "MODE SELECTION DB"."UF PLC_1 PROCESS BUFF", in2 := 90)
      wire#w1
      Contact( "INPUT MAPPING DB"."ABFV 205 FEED BACK OPEN" )
      wire#w2
      Move(in := 95, out1 => "MODE SELECTION DB"."UF PLC_1 PROCESS BUFF")
   END_RUNG
   RUNG wire#w1
      Contact( "AlwaysTRUE" )
   END_RUNG wire#w2
   // the same network as SCL:
   IF ("MODE SELECTION DB"."UF PLC_1 MODE BUFF" = 1) AND ("MODE SELECTION DB"."UF PLC_1 PROCESS BUFF" = 90) AND ("INPUT MAPPING DB"."ABFV 205 FEED BACK OPEN" OR "AlwaysTRUE") THEN
       "MODE SELECTION DB"."UF PLC_1 PROCESS BUFF" := 95;
   END_IF;
END_REGION

REGION Network 22: ABFV 207 OPEN FB
   RUNG wire#powerrail
      { S7_Templates := "SrcType := Int" } EQ_Contact(in1 := "MODE SELECTION DB"."UF PLC_1 MODE BUFF", in2 := 1)
      { S7_Templates := "SrcType := Int" } EQ_Contact(in1 := "MODE SELECTION DB"."UF PLC_1 PROCESS BUFF", in2 := 95)
      Contact( "INPUT MAPPING DB"."ABFV-207 FEED BACK OPEN" )
      { S7_Templates := "time_type := Time" } "IEC_Timer_0_DB_46".TON(pt := T#5s, et =>)
      Move(in := 100, out1 => "MODE SELECTION DB"."UF PLC_1 PROCESS BUFF")
   END_RUNG
   // the same network as SCL:
   "IEC_Timer_0_DB_46".TON(IN := ("MODE SELECTION DB"."UF PLC_1 MODE BUFF" = 1) AND ("MODE SELECTION DB"."UF PLC_1 PROCESS BUFF" = 95) AND "INPUT MAPPING DB"."ABFV-207 FEED BACK OPEN",
                           PT := T#5s);
   IF "IEC_Timer_0_DB_46".Q THEN "MODE SELECTION DB"."UF PLC_1 PROCESS BUFF" := 100; END_IF;
END_REGION

REGION Network 23: AIR INLET
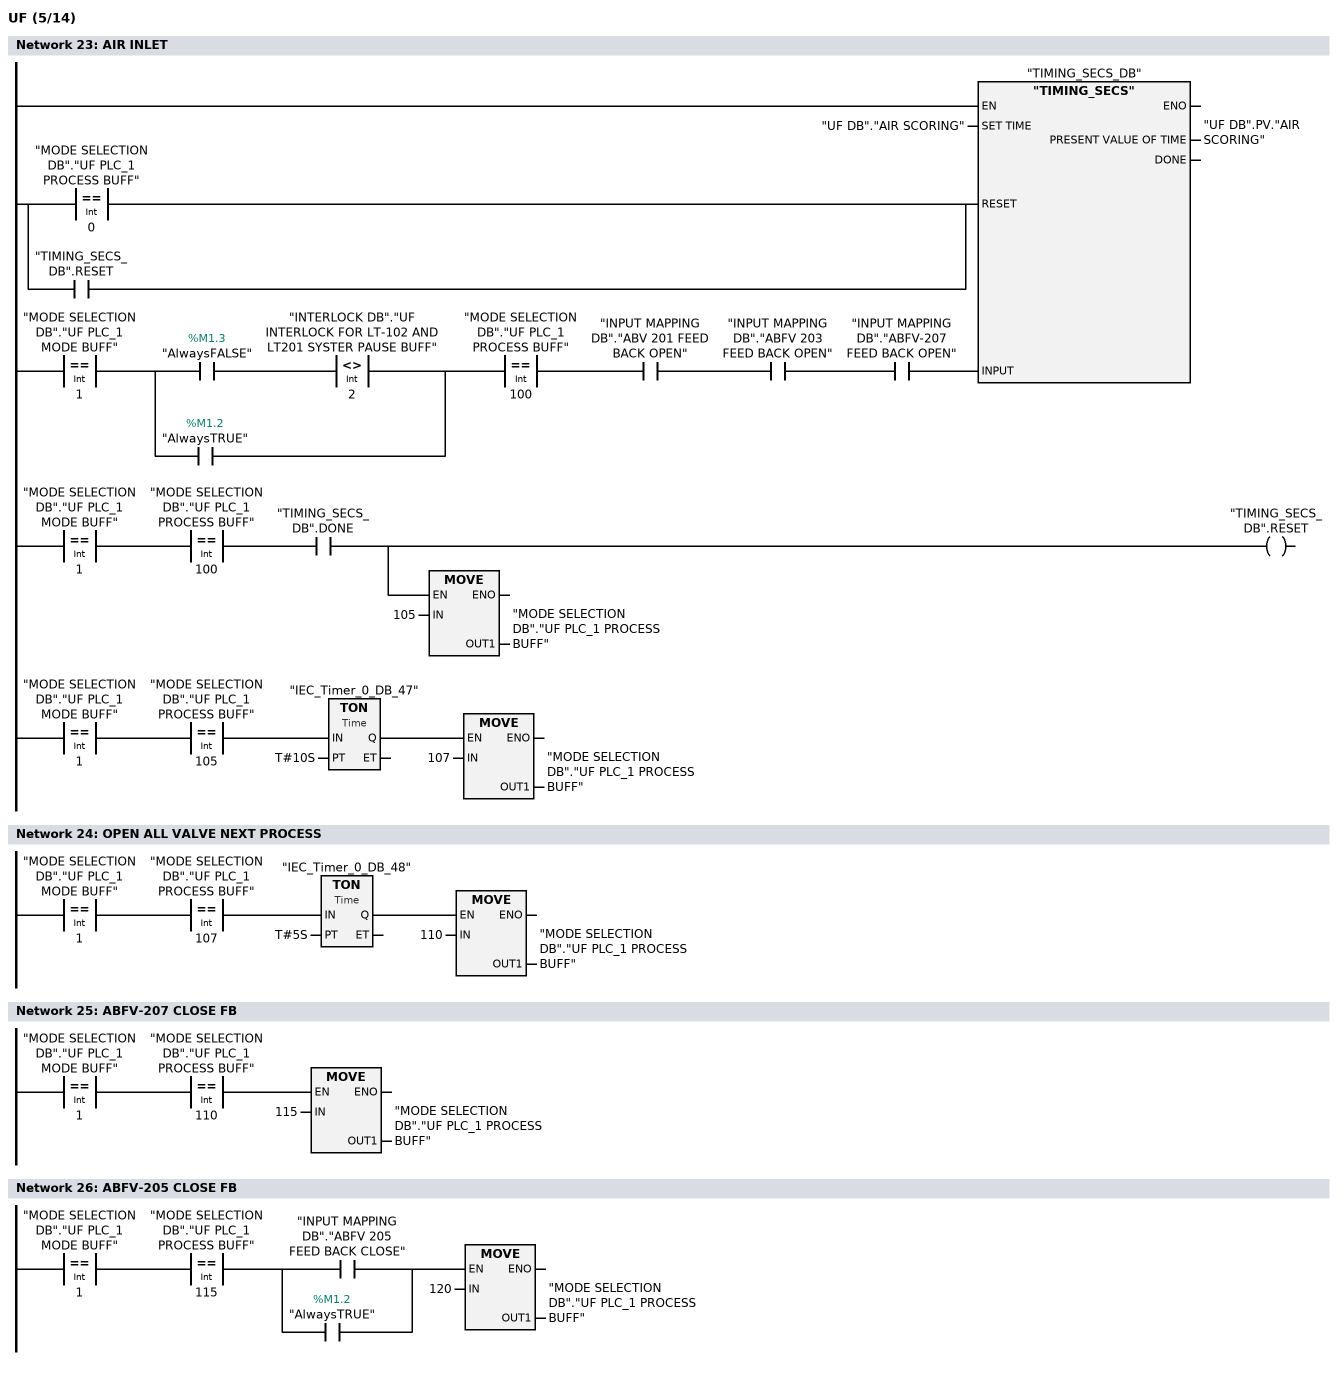
   RUNG wire#powerrail
      "TIMING_SECS_DB"(RESET := wire#w1, INPUT := wire#w4, "SET TIME" := "UF DB"."AIR SCORING", "PRESENT VALUE OF TIME" => "UF DB".PV."AIR SCORING", DONE =>)
   END_RUNG
   RUNG wire#powerrail
      { S7_Templates := "SrcType := Int" } EQ_Contact(in1 := "MODE SELECTION DB"."UF PLC_1 PROCESS BUFF", in2 := 0)
   END_RUNG wire#w1
   RUNG wire#powerrail
      Contact( "TIMING_SECS_DB".RESET )
   END_RUNG wire#w1
   RUNG wire#powerrail
      { S7_Templates := "SrcType := Int" } EQ_Contact(in1 := "MODE SELECTION DB"."UF PLC_1 MODE BUFF", in2 := 1)
      wire#w2
      Contact( "AlwaysFALSE" )
      { S7_Templates := "SrcType := Int" } NE_Contact(in1 := "INTERLOCK DB"."UF INTERLOCK FOR LT-102 AND LT201 SYSTER PAUSE BUFF", in2 := 2)
      wire#w3
      { S7_Templates := "SrcType := Int" } EQ_Contact(in1 := "MODE SELECTION DB"."UF PLC_1 PROCESS BUFF", in2 := 100)
      Contact( "INPUT MAPPING DB"."ABV 201 FEED BACK OPEN" )
      Contact( "INPUT MAPPING DB"."ABFV 203 FEED BACK OPEN" )
      Contact( "INPUT MAPPING DB"."ABFV-207 FEED BACK OPEN" )
   END_RUNG wire#w4
   RUNG wire#w2
      Contact( "AlwaysTRUE" )
   END_RUNG wire#w3
   RUNG wire#powerrail
      { S7_Templates := "SrcType := Int" } EQ_Contact(in1 := "MODE SELECTION DB"."UF PLC_1 MODE BUFF", in2 := 1)
      { S7_Templates := "SrcType := Int" } EQ_Contact(in1 := "MODE SELECTION DB"."UF PLC_1 PROCESS BUFF", in2 := 100)
      Contact( "TIMING_SECS_DB".DONE )
      wire#w5
      Coil( "TIMING_SECS_DB".RESET )
   END_RUNG
   RUNG wire#w5
      Move(in := 105, out1 => "MODE SELECTION DB"."UF PLC_1 PROCESS BUFF")
   END_RUNG
   RUNG wire#powerrail
      { S7_Templates := "SrcType := Int" } EQ_Contact(in1 := "MODE SELECTION DB"."UF PLC_1 MODE BUFF", in2 := 1)
      { S7_Templates := "SrcType := Int" } EQ_Contact(in1 := "MODE SELECTION DB"."UF PLC_1 PROCESS BUFF", in2 := 105)
      { S7_Templates := "time_type := Time" } "IEC_Timer_0_DB_47".TON(pt := T#10S, et =>)
      Move(in := 107, out1 => "MODE SELECTION DB"."UF PLC_1 PROCESS BUFF")
   END_RUNG
   // the same network as SCL:
   "TIMING_SECS_DB"("SET TIME" := "UF DB"."AIR SCORING",   // "TIMING_SECS"
                    RESET := ("MODE SELECTION DB"."UF PLC_1 PROCESS BUFF" = 0) OR "TIMING_SECS_DB".RESET,
                    INPUT := ("MODE SELECTION DB"."UF PLC_1 MODE BUFF" = 1) AND (("AlwaysFALSE" AND ("INTERLOCK DB"."UF INTERLOCK FOR LT-102 AND LT201 SYSTER PAUSE BUFF" <> 2)) OR "AlwaysTRUE") AND ("MODE SELECTION DB"."UF PLC_1 PROCESS BUFF" = 100) AND "INPUT MAPPING DB"."ABV 201 FEED BACK OPEN" AND "INPUT MAPPING DB"."ABFV 203 FEED BACK OPEN" AND "INPUT MAPPING DB"."ABFV-207 FEED BACK OPEN",
                    "PRESENT VALUE OF TIME" => "UF DB".PV."AIR SCORING");
   "TIMING_SECS_DB".RESET := ("MODE SELECTION DB"."UF PLC_1 MODE BUFF" = 1) AND ("MODE SELECTION DB"."UF PLC_1 PROCESS BUFF" = 100) AND "TIMING_SECS_DB".DONE;
   IF "TIMING_SECS_DB".RESET THEN "MODE SELECTION DB"."UF PLC_1 PROCESS BUFF" := 105; END_IF;
   "IEC_Timer_0_DB_47".TON(IN := ("MODE SELECTION DB"."UF PLC_1 MODE BUFF" = 1) AND ("MODE SELECTION DB"."UF PLC_1 PROCESS BUFF" = 105),
                           PT := T#10S);
   IF "IEC_Timer_0_DB_47".Q THEN "MODE SELECTION DB"."UF PLC_1 PROCESS BUFF" := 107; END_IF;
END_REGION

REGION Network 24: OPEN ALL VALVE NEXT PROCESS
   RUNG wire#powerrail
      { S7_Templates := "SrcType := Int" } EQ_Contact(in1 := "MODE SELECTION DB"."UF PLC_1 MODE BUFF", in2 := 1)
      { S7_Templates := "SrcType := Int" } EQ_Contact(in1 := "MODE SELECTION DB"."UF PLC_1 PROCESS BUFF", in2 := 107)
      { S7_Templates := "time_type := Time" } "IEC_Timer_0_DB_48".TON(pt := T#5S, et =>)
      Move(in := 110, out1 => "MODE SELECTION DB"."UF PLC_1 PROCESS BUFF")
   END_RUNG
   // the same network as SCL:
   "IEC_Timer_0_DB_48".TON(IN := ("MODE SELECTION DB"."UF PLC_1 MODE BUFF" = 1) AND ("MODE SELECTION DB"."UF PLC_1 PROCESS BUFF" = 107),
                           PT := T#5S);
   IF "IEC_Timer_0_DB_48".Q THEN "MODE SELECTION DB"."UF PLC_1 PROCESS BUFF" := 110; END_IF;
END_REGION

REGION Network 25: ABFV-207 CLOSE FB
   RUNG wire#powerrail
      { S7_Templates := "SrcType := Int" } EQ_Contact(in1 := "MODE SELECTION DB"."UF PLC_1 MODE BUFF", in2 := 1)
      { S7_Templates := "SrcType := Int" } EQ_Contact(in1 := "MODE SELECTION DB"."UF PLC_1 PROCESS BUFF", in2 := 110)
      Move(in := 115, out1 => "MODE SELECTION DB"."UF PLC_1 PROCESS BUFF")
   END_RUNG
   // the same network as SCL:
   IF ("MODE SELECTION DB"."UF PLC_1 MODE BUFF" = 1) AND ("MODE SELECTION DB"."UF PLC_1 PROCESS BUFF" = 110) THEN
       "MODE SELECTION DB"."UF PLC_1 PROCESS BUFF" := 115;
   END_IF;
END_REGION

REGION Network 26: ABFV-205 CLOSE FB
   RUNG wire#powerrail
      { S7_Templates := "SrcType := Int" } EQ_Contact(in1 := "MODE SELECTION DB"."UF PLC_1 MODE BUFF", in2 := 1)
      { S7_Templates := "SrcType := Int" } EQ_Contact(in1 := "MODE SELECTION DB"."UF PLC_1 PROCESS BUFF", in2 := 115)
      wire#w1
      Contact( "INPUT MAPPING DB"."ABFV 205 FEED BACK CLOSE" )
      wire#w2
      Move(in := 120, out1 => "MODE SELECTION DB"."UF PLC_1 PROCESS BUFF")
   END_RUNG
   RUNG wire#w1
      Contact( "AlwaysTRUE" )
   END_RUNG wire#w2
   // the same network as SCL:
   IF ("MODE SELECTION DB"."UF PLC_1 MODE BUFF" = 1) AND ("MODE SELECTION DB"."UF PLC_1 PROCESS BUFF" = 115) AND ("INPUT MAPPING DB"."ABFV 205 FEED BACK CLOSE" OR "AlwaysTRUE") THEN
       "MODE SELECTION DB"."UF PLC_1 PROCESS BUFF" := 120;
   END_IF;
END_REGION

REGION Network 27: ABFV-203 CLOSE FB
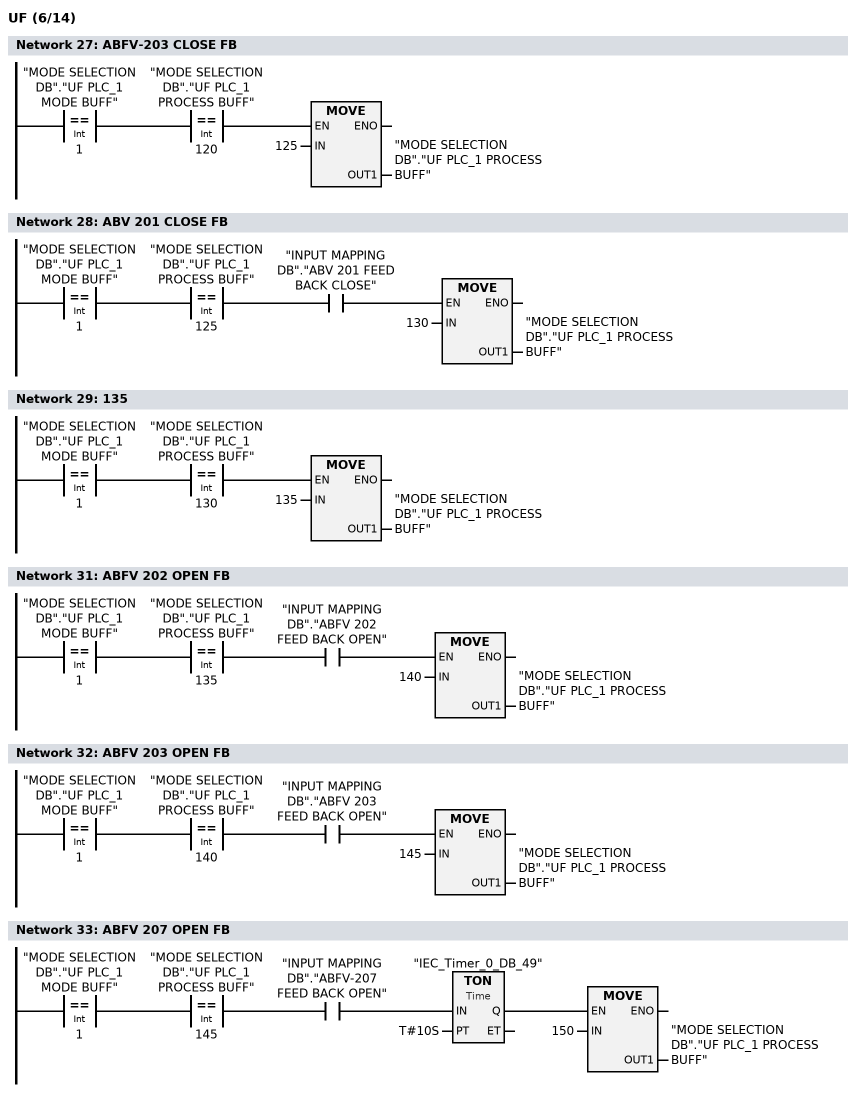
   RUNG wire#powerrail
      { S7_Templates := "SrcType := Int" } EQ_Contact(in1 := "MODE SELECTION DB"."UF PLC_1 MODE BUFF", in2 := 1)
      { S7_Templates := "SrcType := Int" } EQ_Contact(in1 := "MODE SELECTION DB"."UF PLC_1 PROCESS BUFF", in2 := 120)
      Move(in := 125, out1 => "MODE SELECTION DB"."UF PLC_1 PROCESS BUFF")
   END_RUNG
   // the same network as SCL:
   IF ("MODE SELECTION DB"."UF PLC_1 MODE BUFF" = 1) AND ("MODE SELECTION DB"."UF PLC_1 PROCESS BUFF" = 120) THEN
       "MODE SELECTION DB"."UF PLC_1 PROCESS BUFF" := 125;
   END_IF;
END_REGION

REGION Network 28: ABV 201 CLOSE FB
   RUNG wire#powerrail
      { S7_Templates := "SrcType := Int" } EQ_Contact(in1 := "MODE SELECTION DB"."UF PLC_1 MODE BUFF", in2 := 1)
      { S7_Templates := "SrcType := Int" } EQ_Contact(in1 := "MODE SELECTION DB"."UF PLC_1 PROCESS BUFF", in2 := 125)
      Contact( "INPUT MAPPING DB"."ABV 201 FEED BACK CLOSE" )
      Move(in := 130, out1 => "MODE SELECTION DB"."UF PLC_1 PROCESS BUFF")
   END_RUNG
   // the same network as SCL:
   IF ("MODE SELECTION DB"."UF PLC_1 MODE BUFF" = 1) AND ("MODE SELECTION DB"."UF PLC_1 PROCESS BUFF" = 125) AND "INPUT MAPPING DB"."ABV 201 FEED BACK CLOSE" THEN
       "MODE SELECTION DB"."UF PLC_1 PROCESS BUFF" := 130;
   END_IF;
END_REGION

REGION Network 29: 135
   RUNG wire#powerrail
      { S7_Templates := "SrcType := Int" } EQ_Contact(in1 := "MODE SELECTION DB"."UF PLC_1 MODE BUFF", in2 := 1)
      { S7_Templates := "SrcType := Int" } EQ_Contact(in1 := "MODE SELECTION DB"."UF PLC_1 PROCESS BUFF", in2 := 130)
      Move(in := 135, out1 => "MODE SELECTION DB"."UF PLC_1 PROCESS BUFF")
   END_RUNG
   // the same network as SCL:
   IF ("MODE SELECTION DB"."UF PLC_1 MODE BUFF" = 1) AND ("MODE SELECTION DB"."UF PLC_1 PROCESS BUFF" = 130) THEN
       "MODE SELECTION DB"."UF PLC_1 PROCESS BUFF" := 135;
   END_IF;
END_REGION

REGION Network 31: ABFV 202 OPEN FB
   RUNG wire#powerrail
      { S7_Templates := "SrcType := Int" } EQ_Contact(in1 := "MODE SELECTION DB"."UF PLC_1 MODE BUFF", in2 := 1)
      { S7_Templates := "SrcType := Int" } EQ_Contact(in1 := "MODE SELECTION DB"."UF PLC_1 PROCESS BUFF", in2 := 135)
      Contact( "INPUT MAPPING DB"."ABFV 202 FEED BACK OPEN" )
      Move(in := 140, out1 => "MODE SELECTION DB"."UF PLC_1 PROCESS BUFF")
   END_RUNG
   // the same network as SCL:
   IF ("MODE SELECTION DB"."UF PLC_1 MODE BUFF" = 1) AND ("MODE SELECTION DB"."UF PLC_1 PROCESS BUFF" = 135) AND "INPUT MAPPING DB"."ABFV 202 FEED BACK OPEN" THEN
       "MODE SELECTION DB"."UF PLC_1 PROCESS BUFF" := 140;
   END_IF;
END_REGION

REGION Network 32: ABFV 203 OPEN FB
   RUNG wire#powerrail
      { S7_Templates := "SrcType := Int" } EQ_Contact(in1 := "MODE SELECTION DB"."UF PLC_1 MODE BUFF", in2 := 1)
      { S7_Templates := "SrcType := Int" } EQ_Contact(in1 := "MODE SELECTION DB"."UF PLC_1 PROCESS BUFF", in2 := 140)
      Contact( "INPUT MAPPING DB"."ABFV 203 FEED BACK OPEN" )
      Move(in := 145, out1 => "MODE SELECTION DB"."UF PLC_1 PROCESS BUFF")
   END_RUNG
   // the same network as SCL:
   IF ("MODE SELECTION DB"."UF PLC_1 MODE BUFF" = 1) AND ("MODE SELECTION DB"."UF PLC_1 PROCESS BUFF" = 140) AND "INPUT MAPPING DB"."ABFV 203 FEED BACK OPEN" THEN
       "MODE SELECTION DB"."UF PLC_1 PROCESS BUFF" := 145;
   END_IF;
END_REGION

REGION Network 33: ABFV 207 OPEN FB
   RUNG wire#powerrail
      { S7_Templates := "SrcType := Int" } EQ_Contact(in1 := "MODE SELECTION DB"."UF PLC_1 MODE BUFF", in2 := 1)
      { S7_Templates := "SrcType := Int" } EQ_Contact(in1 := "MODE SELECTION DB"."UF PLC_1 PROCESS BUFF", in2 := 145)
      Contact( "INPUT MAPPING DB"."ABFV-207 FEED BACK OPEN" )
      { S7_Templates := "time_type := Time" } "IEC_Timer_0_DB_49".TON(pt := T#10S, et =>)
      Move(in := 150, out1 => "MODE SELECTION DB"."UF PLC_1 PROCESS BUFF")
   END_RUNG
   // the same network as SCL:
   "IEC_Timer_0_DB_49".TON(IN := ("MODE SELECTION DB"."UF PLC_1 MODE BUFF" = 1) AND ("MODE SELECTION DB"."UF PLC_1 PROCESS BUFF" = 145) AND "INPUT MAPPING DB"."ABFV-207 FEED BACK OPEN",
                           PT := T#10S);
   IF "IEC_Timer_0_DB_49".Q THEN "MODE SELECTION DB"."UF PLC_1 PROCESS BUFF" := 150; END_IF;
END_REGION

REGION Network 34: DAIN
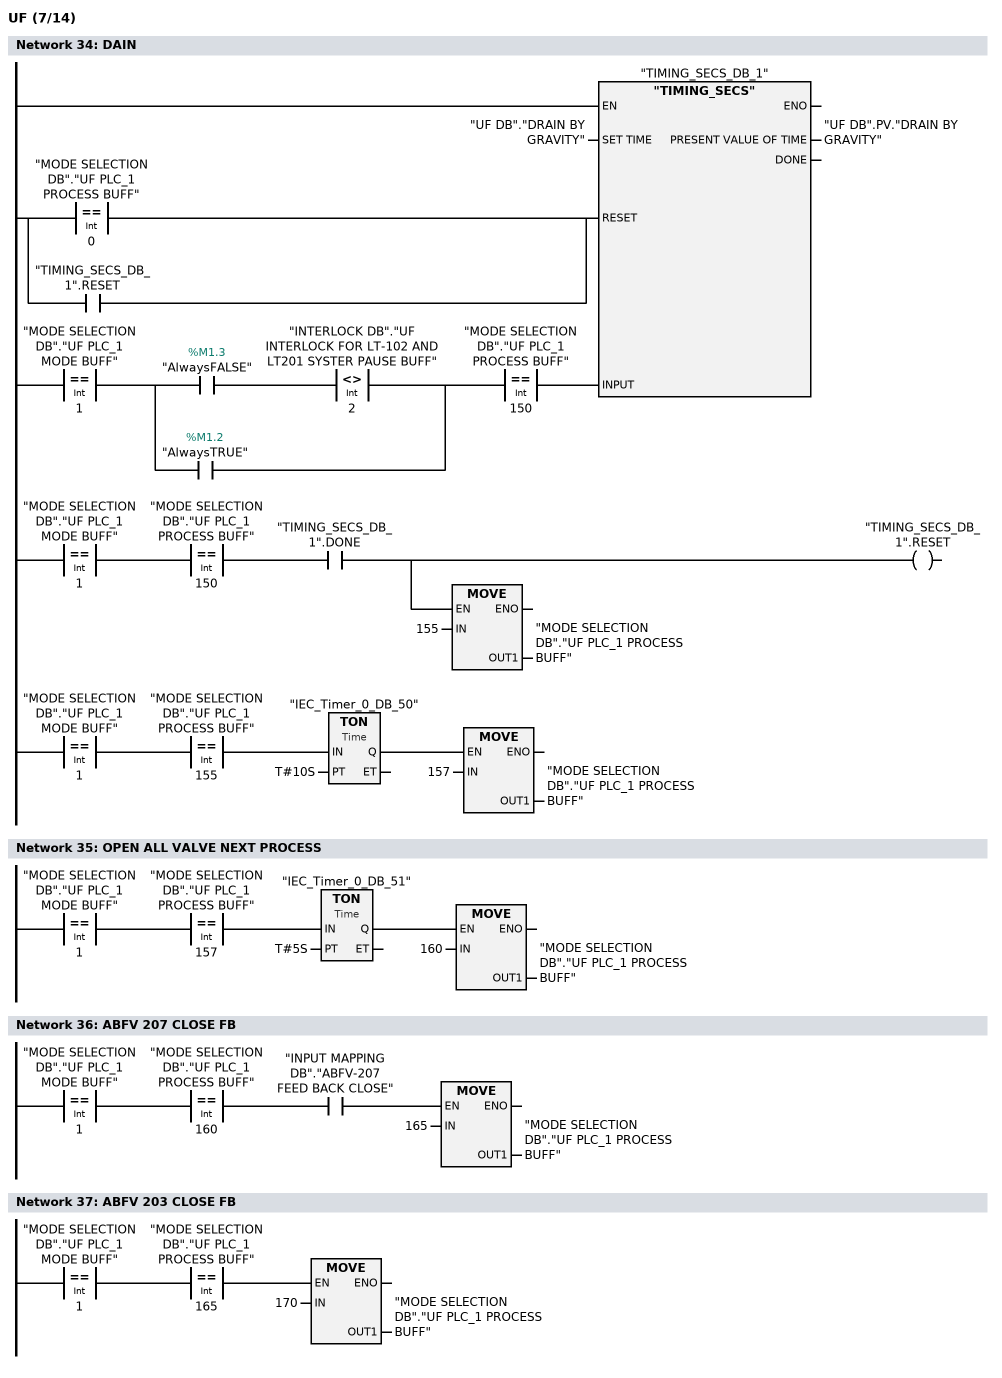
   RUNG wire#powerrail
      "TIMING_SECS_DB_1"(RESET := wire#w1, INPUT := wire#w4, "SET TIME" := "UF DB"."DRAIN BY GRAVITY", "PRESENT VALUE OF TIME" => "UF DB".PV."DRAIN BY GRAVITY", DONE =>)
   END_RUNG
   RUNG wire#powerrail
      { S7_Templates := "SrcType := Int" } EQ_Contact(in1 := "MODE SELECTION DB"."UF PLC_1 PROCESS BUFF", in2 := 0)
   END_RUNG wire#w1
   RUNG wire#powerrail
      Contact( "TIMING_SECS_DB_1".RESET )
   END_RUNG wire#w1
   RUNG wire#powerrail
      { S7_Templates := "SrcType := Int" } EQ_Contact(in1 := "MODE SELECTION DB"."UF PLC_1 MODE BUFF", in2 := 1)
      wire#w2
      Contact( "AlwaysFALSE" )
      { S7_Templates := "SrcType := Int" } NE_Contact(in1 := "INTERLOCK DB"."UF INTERLOCK FOR LT-102 AND LT201 SYSTER PAUSE BUFF", in2 := 2)
      wire#w3
      { S7_Templates := "SrcType := Int" } EQ_Contact(in1 := "MODE SELECTION DB"."UF PLC_1 PROCESS BUFF", in2 := 150)
   END_RUNG wire#w4
   RUNG wire#w2
      Contact( "AlwaysTRUE" )
   END_RUNG wire#w3
   RUNG wire#powerrail
      { S7_Templates := "SrcType := Int" } EQ_Contact(in1 := "MODE SELECTION DB"."UF PLC_1 MODE BUFF", in2 := 1)
      { S7_Templates := "SrcType := Int" } EQ_Contact(in1 := "MODE SELECTION DB"."UF PLC_1 PROCESS BUFF", in2 := 150)
      Contact( "TIMING_SECS_DB_1".DONE )
      wire#w5
      Coil( "TIMING_SECS_DB_1".RESET )
   END_RUNG
   RUNG wire#w5
      Move(in := 155, out1 => "MODE SELECTION DB"."UF PLC_1 PROCESS BUFF")
   END_RUNG
   RUNG wire#powerrail
      { S7_Templates := "SrcType := Int" } EQ_Contact(in1 := "MODE SELECTION DB"."UF PLC_1 MODE BUFF", in2 := 1)
      { S7_Templates := "SrcType := Int" } EQ_Contact(in1 := "MODE SELECTION DB"."UF PLC_1 PROCESS BUFF", in2 := 155)
      { S7_Templates := "time_type := Time" } "IEC_Timer_0_DB_50".TON(pt := T#10S, et =>)
      Move(in := 157, out1 => "MODE SELECTION DB"."UF PLC_1 PROCESS BUFF")
   END_RUNG
   // the same network as SCL:
   "TIMING_SECS_DB_1"("SET TIME" := "UF DB"."DRAIN BY GRAVITY",   // "TIMING_SECS"
                      RESET := ("MODE SELECTION DB"."UF PLC_1 PROCESS BUFF" = 0) OR "TIMING_SECS_DB_1".RESET,
                      INPUT := ("MODE SELECTION DB"."UF PLC_1 MODE BUFF" = 1) AND (("AlwaysFALSE" AND ("INTERLOCK DB"."UF INTERLOCK FOR LT-102 AND LT201 SYSTER PAUSE BUFF" <> 2)) OR "AlwaysTRUE") AND ("MODE SELECTION DB"."UF PLC_1 PROCESS BUFF" = 150),
                      "PRESENT VALUE OF TIME" => "UF DB".PV."DRAIN BY GRAVITY");
   "TIMING_SECS_DB_1".RESET := ("MODE SELECTION DB"."UF PLC_1 MODE BUFF" = 1) AND ("MODE SELECTION DB"."UF PLC_1 PROCESS BUFF" = 150) AND "TIMING_SECS_DB_1".DONE;
   IF "TIMING_SECS_DB_1".RESET THEN "MODE SELECTION DB"."UF PLC_1 PROCESS BUFF" := 155; END_IF;
   "IEC_Timer_0_DB_50".TON(IN := ("MODE SELECTION DB"."UF PLC_1 MODE BUFF" = 1) AND ("MODE SELECTION DB"."UF PLC_1 PROCESS BUFF" = 155),
                           PT := T#10S);
   IF "IEC_Timer_0_DB_50".Q THEN "MODE SELECTION DB"."UF PLC_1 PROCESS BUFF" := 157; END_IF;
END_REGION

REGION Network 35: OPEN ALL VALVE NEXT PROCESS
   RUNG wire#powerrail
      { S7_Templates := "SrcType := Int" } EQ_Contact(in1 := "MODE SELECTION DB"."UF PLC_1 MODE BUFF", in2 := 1)
      { S7_Templates := "SrcType := Int" } EQ_Contact(in1 := "MODE SELECTION DB"."UF PLC_1 PROCESS BUFF", in2 := 157)
      { S7_Templates := "time_type := Time" } "IEC_Timer_0_DB_51".TON(pt := T#5S, et =>)
      Move(in := 160, out1 => "MODE SELECTION DB"."UF PLC_1 PROCESS BUFF")
   END_RUNG
   // the same network as SCL:
   "IEC_Timer_0_DB_51".TON(IN := ("MODE SELECTION DB"."UF PLC_1 MODE BUFF" = 1) AND ("MODE SELECTION DB"."UF PLC_1 PROCESS BUFF" = 157),
                           PT := T#5S);
   IF "IEC_Timer_0_DB_51".Q THEN "MODE SELECTION DB"."UF PLC_1 PROCESS BUFF" := 160; END_IF;
END_REGION

REGION Network 36: ABFV 207 CLOSE FB
   RUNG wire#powerrail
      { S7_Templates := "SrcType := Int" } EQ_Contact(in1 := "MODE SELECTION DB"."UF PLC_1 MODE BUFF", in2 := 1)
      { S7_Templates := "SrcType := Int" } EQ_Contact(in1 := "MODE SELECTION DB"."UF PLC_1 PROCESS BUFF", in2 := 160)
      Contact( "INPUT MAPPING DB"."ABFV-207 FEED BACK CLOSE" )
      Move(in := 165, out1 => "MODE SELECTION DB"."UF PLC_1 PROCESS BUFF")
   END_RUNG
   // the same network as SCL:
   IF ("MODE SELECTION DB"."UF PLC_1 MODE BUFF" = 1) AND ("MODE SELECTION DB"."UF PLC_1 PROCESS BUFF" = 160) AND "INPUT MAPPING DB"."ABFV-207 FEED BACK CLOSE" THEN
       "MODE SELECTION DB"."UF PLC_1 PROCESS BUFF" := 165;
   END_IF;
END_REGION

REGION Network 37: ABFV 203 CLOSE FB
   RUNG wire#powerrail
      { S7_Templates := "SrcType := Int" } EQ_Contact(in1 := "MODE SELECTION DB"."UF PLC_1 MODE BUFF", in2 := 1)
      { S7_Templates := "SrcType := Int" } EQ_Contact(in1 := "MODE SELECTION DB"."UF PLC_1 PROCESS BUFF", in2 := 165)
      Move(in := 170, out1 => "MODE SELECTION DB"."UF PLC_1 PROCESS BUFF")
   END_RUNG
   // the same network as SCL:
   IF ("MODE SELECTION DB"."UF PLC_1 MODE BUFF" = 1) AND ("MODE SELECTION DB"."UF PLC_1 PROCESS BUFF" = 165) THEN
       "MODE SELECTION DB"."UF PLC_1 PROCESS BUFF" := 170;
   END_IF;
END_REGION

REGION Network 38: ABFV 202 CLOSE FB
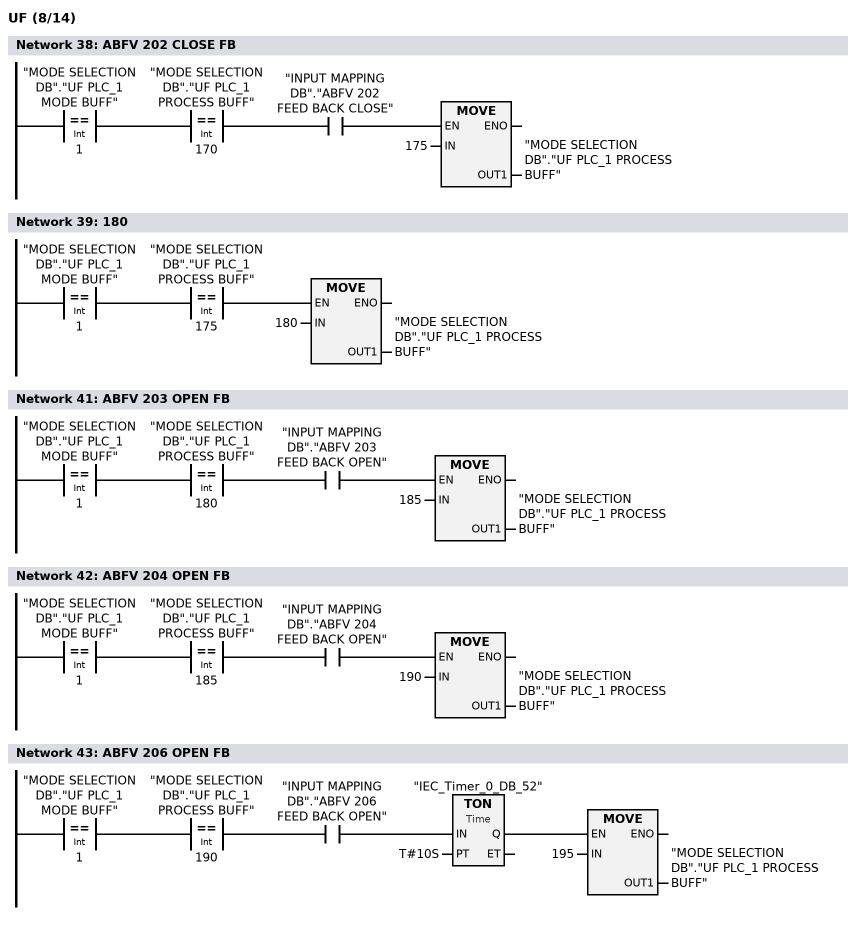
   RUNG wire#powerrail
      { S7_Templates := "SrcType := Int" } EQ_Contact(in1 := "MODE SELECTION DB"."UF PLC_1 MODE BUFF", in2 := 1)
      { S7_Templates := "SrcType := Int" } EQ_Contact(in1 := "MODE SELECTION DB"."UF PLC_1 PROCESS BUFF", in2 := 170)
      Contact( "INPUT MAPPING DB"."ABFV 202 FEED BACK CLOSE" )
      Move(in := 175, out1 => "MODE SELECTION DB"."UF PLC_1 PROCESS BUFF")
   END_RUNG
   // the same network as SCL:
   IF ("MODE SELECTION DB"."UF PLC_1 MODE BUFF" = 1) AND ("MODE SELECTION DB"."UF PLC_1 PROCESS BUFF" = 170) AND "INPUT MAPPING DB"."ABFV 202 FEED BACK CLOSE" THEN
       "MODE SELECTION DB"."UF PLC_1 PROCESS BUFF" := 175;
   END_IF;
END_REGION

REGION Network 39: 180
   RUNG wire#powerrail
      { S7_Templates := "SrcType := Int" } EQ_Contact(in1 := "MODE SELECTION DB"."UF PLC_1 MODE BUFF", in2 := 1)
      { S7_Templates := "SrcType := Int" } EQ_Contact(in1 := "MODE SELECTION DB"."UF PLC_1 PROCESS BUFF", in2 := 175)
      Move(in := 180, out1 => "MODE SELECTION DB"."UF PLC_1 PROCESS BUFF")
   END_RUNG
   // the same network as SCL:
   IF ("MODE SELECTION DB"."UF PLC_1 MODE BUFF" = 1) AND ("MODE SELECTION DB"."UF PLC_1 PROCESS BUFF" = 175) THEN
       "MODE SELECTION DB"."UF PLC_1 PROCESS BUFF" := 180;
   END_IF;
END_REGION

REGION Network 41: ABFV 203 OPEN FB
   RUNG wire#powerrail
      { S7_Templates := "SrcType := Int" } EQ_Contact(in1 := "MODE SELECTION DB"."UF PLC_1 MODE BUFF", in2 := 1)
      { S7_Templates := "SrcType := Int" } EQ_Contact(in1 := "MODE SELECTION DB"."UF PLC_1 PROCESS BUFF", in2 := 180)
      Contact( "INPUT MAPPING DB"."ABFV 203 FEED BACK OPEN" )
      Move(in := 185, out1 => "MODE SELECTION DB"."UF PLC_1 PROCESS BUFF")
   END_RUNG
   // the same network as SCL:
   IF ("MODE SELECTION DB"."UF PLC_1 MODE BUFF" = 1) AND ("MODE SELECTION DB"."UF PLC_1 PROCESS BUFF" = 180) AND "INPUT MAPPING DB"."ABFV 203 FEED BACK OPEN" THEN
       "MODE SELECTION DB"."UF PLC_1 PROCESS BUFF" := 185;
   END_IF;
END_REGION

REGION Network 42: ABFV 204 OPEN FB
   RUNG wire#powerrail
      { S7_Templates := "SrcType := Int" } EQ_Contact(in1 := "MODE SELECTION DB"."UF PLC_1 MODE BUFF", in2 := 1)
      { S7_Templates := "SrcType := Int" } EQ_Contact(in1 := "MODE SELECTION DB"."UF PLC_1 PROCESS BUFF", in2 := 185)
      Contact( "INPUT MAPPING DB"."ABFV 204 FEED BACK OPEN" )
      Move(in := 190, out1 => "MODE SELECTION DB"."UF PLC_1 PROCESS BUFF")
   END_RUNG
   // the same network as SCL:
   IF ("MODE SELECTION DB"."UF PLC_1 MODE BUFF" = 1) AND ("MODE SELECTION DB"."UF PLC_1 PROCESS BUFF" = 185) AND "INPUT MAPPING DB"."ABFV 204 FEED BACK OPEN" THEN
       "MODE SELECTION DB"."UF PLC_1 PROCESS BUFF" := 190;
   END_IF;
END_REGION

REGION Network 43: ABFV 206 OPEN FB
   RUNG wire#powerrail
      { S7_Templates := "SrcType := Int" } EQ_Contact(in1 := "MODE SELECTION DB"."UF PLC_1 MODE BUFF", in2 := 1)
      { S7_Templates := "SrcType := Int" } EQ_Contact(in1 := "MODE SELECTION DB"."UF PLC_1 PROCESS BUFF", in2 := 190)
      Contact( "INPUT MAPPING DB"."ABFV 206 FEED BACK OPEN" )
      { S7_Templates := "time_type := Time" } "IEC_Timer_0_DB_52".TON(pt := T#10S, et =>)
      Move(in := 195, out1 => "MODE SELECTION DB"."UF PLC_1 PROCESS BUFF")
   END_RUNG
   // the same network as SCL:
   "IEC_Timer_0_DB_52".TON(IN := ("MODE SELECTION DB"."UF PLC_1 MODE BUFF" = 1) AND ("MODE SELECTION DB"."UF PLC_1 PROCESS BUFF" = 190) AND "INPUT MAPPING DB"."ABFV 206 FEED BACK OPEN",
                           PT := T#10S);
   IF "IEC_Timer_0_DB_52".Q THEN "MODE SELECTION DB"."UF PLC_1 PROCESS BUFF" := 195; END_IF;
END_REGION

REGION Network 44: BACKWASH-1
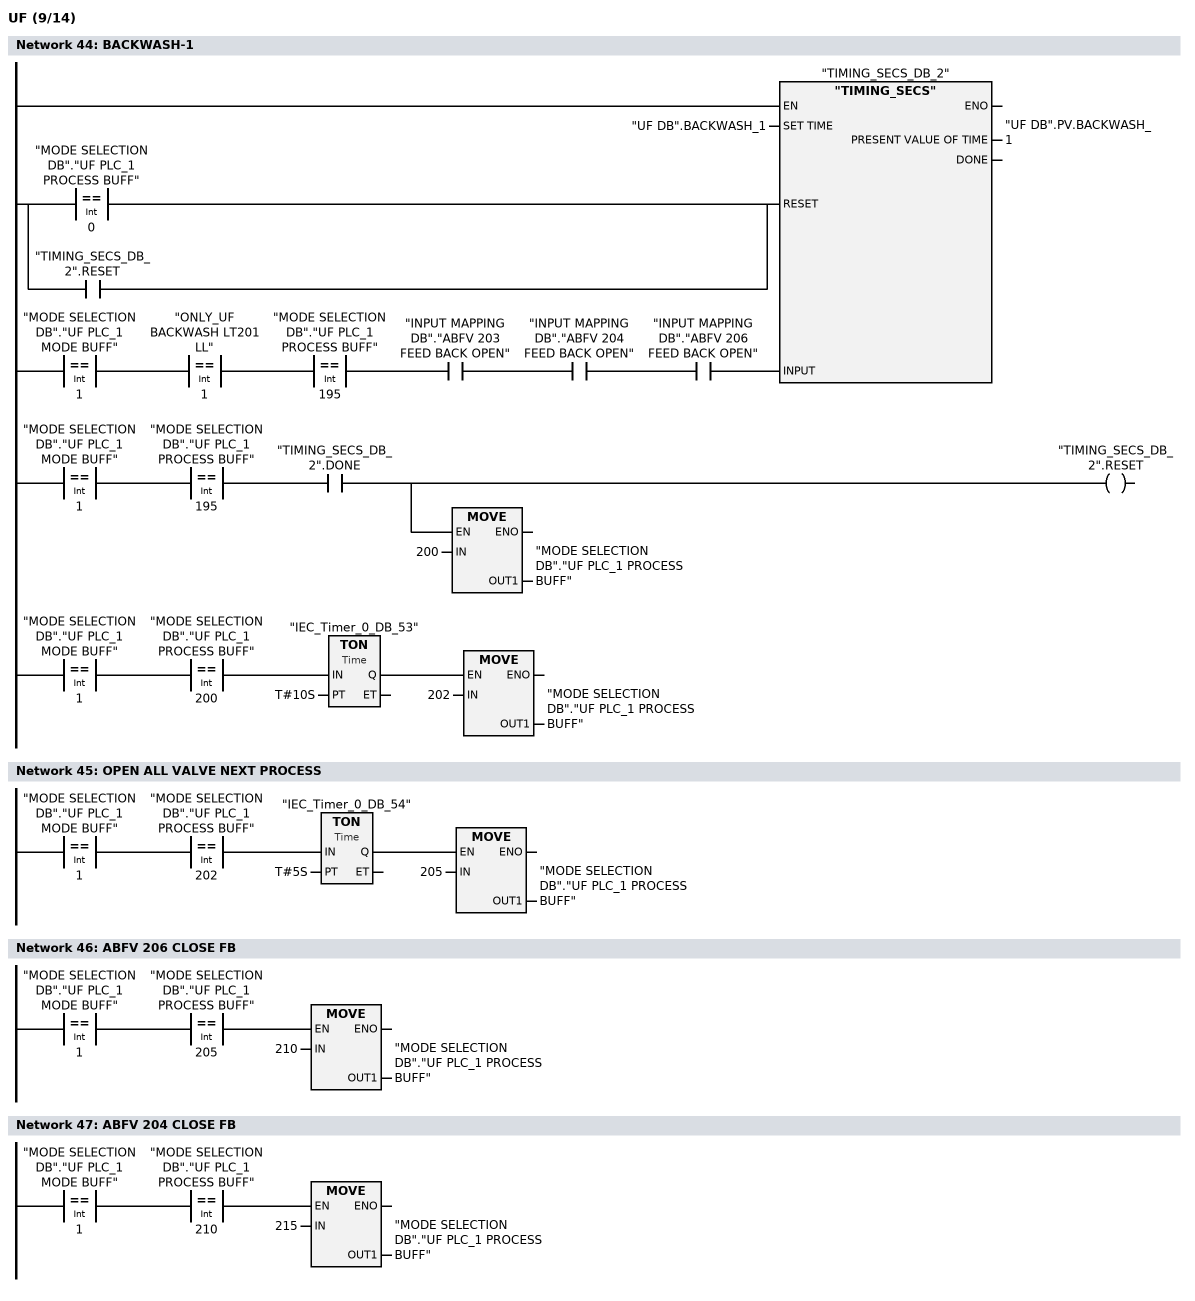
   RUNG wire#powerrail
      "TIMING_SECS_DB_2"(RESET := wire#w1, INPUT := wire#w2, "SET TIME" := "UF DB".BACKWASH_1, "PRESENT VALUE OF TIME" => "UF DB".PV.BACKWASH_1, DONE =>)
   END_RUNG
   RUNG wire#powerrail
      { S7_Templates := "SrcType := Int" } EQ_Contact(in1 := "MODE SELECTION DB"."UF PLC_1 PROCESS BUFF", in2 := 0)
   END_RUNG wire#w1
   RUNG wire#powerrail
      Contact( "TIMING_SECS_DB_2".RESET )
   END_RUNG wire#w1
   RUNG wire#powerrail
      { S7_Templates := "SrcType := Int" } EQ_Contact(in1 := "MODE SELECTION DB"."UF PLC_1 MODE BUFF", in2 := 1)
      { S7_Templates := "SrcType := Int" } EQ_Contact(in1 := "ONLY_UF BACKWASH LT201 LL", in2 := 1)
      { S7_Templates := "SrcType := Int" } EQ_Contact(in1 := "MODE SELECTION DB"."UF PLC_1 PROCESS BUFF", in2 := 195)
      Contact( "INPUT MAPPING DB"."ABFV 203 FEED BACK OPEN" )
      Contact( "INPUT MAPPING DB"."ABFV 204 FEED BACK OPEN" )
      Contact( "INPUT MAPPING DB"."ABFV 206 FEED BACK OPEN" )
   END_RUNG wire#w2
   RUNG wire#powerrail
      { S7_Templates := "SrcType := Int" } EQ_Contact(in1 := "MODE SELECTION DB"."UF PLC_1 MODE BUFF", in2 := 1)
      { S7_Templates := "SrcType := Int" } EQ_Contact(in1 := "MODE SELECTION DB"."UF PLC_1 PROCESS BUFF", in2 := 195)
      Contact( "TIMING_SECS_DB_2".DONE )
      wire#w3
      Coil( "TIMING_SECS_DB_2".RESET )
   END_RUNG
   RUNG wire#w3
      Move(in := 200, out1 => "MODE SELECTION DB"."UF PLC_1 PROCESS BUFF")
   END_RUNG
   RUNG wire#powerrail
      { S7_Templates := "SrcType := Int" } EQ_Contact(in1 := "MODE SELECTION DB"."UF PLC_1 MODE BUFF", in2 := 1)
      { S7_Templates := "SrcType := Int" } EQ_Contact(in1 := "MODE SELECTION DB"."UF PLC_1 PROCESS BUFF", in2 := 200)
      { S7_Templates := "time_type := Time" } "IEC_Timer_0_DB_53".TON(pt := T#10S, et =>)
      Move(in := 202, out1 => "MODE SELECTION DB"."UF PLC_1 PROCESS BUFF")
   END_RUNG
   // the same network as SCL:
   "TIMING_SECS_DB_2"("SET TIME" := "UF DB".BACKWASH_1,   // "TIMING_SECS"
                      RESET := ("MODE SELECTION DB"."UF PLC_1 PROCESS BUFF" = 0) OR "TIMING_SECS_DB_2".RESET,
                      INPUT := ("MODE SELECTION DB"."UF PLC_1 MODE BUFF" = 1) AND ("ONLY_UF BACKWASH LT201 LL" = 1) AND ("MODE SELECTION DB"."UF PLC_1 PROCESS BUFF" = 195) AND "INPUT MAPPING DB"."ABFV 203 FEED BACK OPEN" AND "INPUT MAPPING DB"."ABFV 204 FEED BACK OPEN" AND "INPUT MAPPING DB"."ABFV 206 FEED BACK OPEN",
                      "PRESENT VALUE OF TIME" => "UF DB".PV.BACKWASH_1);
   "TIMING_SECS_DB_2".RESET := ("MODE SELECTION DB"."UF PLC_1 MODE BUFF" = 1) AND ("MODE SELECTION DB"."UF PLC_1 PROCESS BUFF" = 195) AND "TIMING_SECS_DB_2".DONE;
   IF "TIMING_SECS_DB_2".RESET THEN "MODE SELECTION DB"."UF PLC_1 PROCESS BUFF" := 200; END_IF;
   "IEC_Timer_0_DB_53".TON(IN := ("MODE SELECTION DB"."UF PLC_1 MODE BUFF" = 1) AND ("MODE SELECTION DB"."UF PLC_1 PROCESS BUFF" = 200),
                           PT := T#10S);
   IF "IEC_Timer_0_DB_53".Q THEN "MODE SELECTION DB"."UF PLC_1 PROCESS BUFF" := 202; END_IF;
END_REGION

REGION Network 45: OPEN ALL VALVE NEXT PROCESS
   RUNG wire#powerrail
      { S7_Templates := "SrcType := Int" } EQ_Contact(in1 := "MODE SELECTION DB"."UF PLC_1 MODE BUFF", in2 := 1)
      { S7_Templates := "SrcType := Int" } EQ_Contact(in1 := "MODE SELECTION DB"."UF PLC_1 PROCESS BUFF", in2 := 202)
      { S7_Templates := "time_type := Time" } "IEC_Timer_0_DB_54".TON(pt := T#5S, et =>)
      Move(in := 205, out1 => "MODE SELECTION DB"."UF PLC_1 PROCESS BUFF")
   END_RUNG
   // the same network as SCL:
   "IEC_Timer_0_DB_54".TON(IN := ("MODE SELECTION DB"."UF PLC_1 MODE BUFF" = 1) AND ("MODE SELECTION DB"."UF PLC_1 PROCESS BUFF" = 202),
                           PT := T#5S);
   IF "IEC_Timer_0_DB_54".Q THEN "MODE SELECTION DB"."UF PLC_1 PROCESS BUFF" := 205; END_IF;
END_REGION

REGION Network 46: ABFV 206 CLOSE FB
   RUNG wire#powerrail
      { S7_Templates := "SrcType := Int" } EQ_Contact(in1 := "MODE SELECTION DB"."UF PLC_1 MODE BUFF", in2 := 1)
      { S7_Templates := "SrcType := Int" } EQ_Contact(in1 := "MODE SELECTION DB"."UF PLC_1 PROCESS BUFF", in2 := 205)
      Move(in := 210, out1 => "MODE SELECTION DB"."UF PLC_1 PROCESS BUFF")
   END_RUNG
   // the same network as SCL:
   IF ("MODE SELECTION DB"."UF PLC_1 MODE BUFF" = 1) AND ("MODE SELECTION DB"."UF PLC_1 PROCESS BUFF" = 205) THEN
       "MODE SELECTION DB"."UF PLC_1 PROCESS BUFF" := 210;
   END_IF;
END_REGION

REGION Network 47: ABFV 204 CLOSE FB
   RUNG wire#powerrail
      { S7_Templates := "SrcType := Int" } EQ_Contact(in1 := "MODE SELECTION DB"."UF PLC_1 MODE BUFF", in2 := 1)
      { S7_Templates := "SrcType := Int" } EQ_Contact(in1 := "MODE SELECTION DB"."UF PLC_1 PROCESS BUFF", in2 := 210)
      Move(in := 215, out1 => "MODE SELECTION DB"."UF PLC_1 PROCESS BUFF")
   END_RUNG
   // the same network as SCL:
   IF ("MODE SELECTION DB"."UF PLC_1 MODE BUFF" = 1) AND ("MODE SELECTION DB"."UF PLC_1 PROCESS BUFF" = 210) THEN
       "MODE SELECTION DB"."UF PLC_1 PROCESS BUFF" := 215;
   END_IF;
END_REGION

REGION Network 48: ABFV 203 CLOSE FB
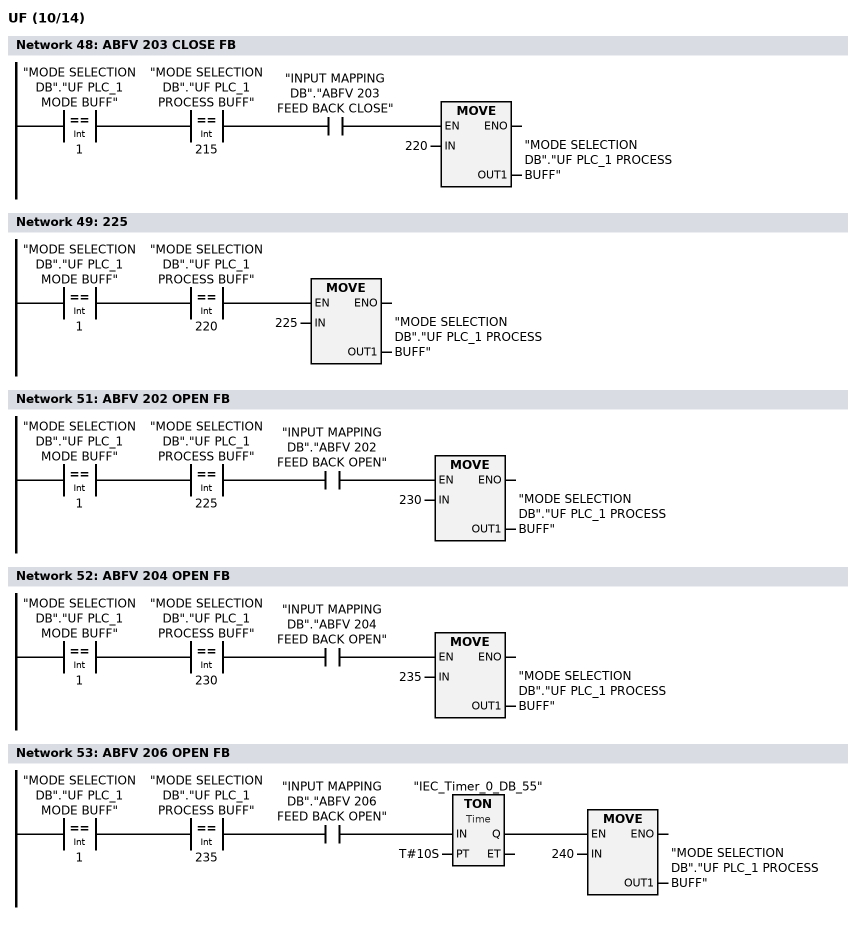
   RUNG wire#powerrail
      { S7_Templates := "SrcType := Int" } EQ_Contact(in1 := "MODE SELECTION DB"."UF PLC_1 MODE BUFF", in2 := 1)
      { S7_Templates := "SrcType := Int" } EQ_Contact(in1 := "MODE SELECTION DB"."UF PLC_1 PROCESS BUFF", in2 := 215)
      Contact( "INPUT MAPPING DB"."ABFV 203 FEED BACK CLOSE" )
      Move(in := 220, out1 => "MODE SELECTION DB"."UF PLC_1 PROCESS BUFF")
   END_RUNG
   // the same network as SCL:
   IF ("MODE SELECTION DB"."UF PLC_1 MODE BUFF" = 1) AND ("MODE SELECTION DB"."UF PLC_1 PROCESS BUFF" = 215) AND "INPUT MAPPING DB"."ABFV 203 FEED BACK CLOSE" THEN
       "MODE SELECTION DB"."UF PLC_1 PROCESS BUFF" := 220;
   END_IF;
END_REGION

REGION Network 49: 225
   RUNG wire#powerrail
      { S7_Templates := "SrcType := Int" } EQ_Contact(in1 := "MODE SELECTION DB"."UF PLC_1 MODE BUFF", in2 := 1)
      { S7_Templates := "SrcType := Int" } EQ_Contact(in1 := "MODE SELECTION DB"."UF PLC_1 PROCESS BUFF", in2 := 220)
      Move(in := 225, out1 => "MODE SELECTION DB"."UF PLC_1 PROCESS BUFF")
   END_RUNG
   // the same network as SCL:
   IF ("MODE SELECTION DB"."UF PLC_1 MODE BUFF" = 1) AND ("MODE SELECTION DB"."UF PLC_1 PROCESS BUFF" = 220) THEN
       "MODE SELECTION DB"."UF PLC_1 PROCESS BUFF" := 225;
   END_IF;
END_REGION

REGION Network 51: ABFV 202 OPEN FB
   RUNG wire#powerrail
      { S7_Templates := "SrcType := Int" } EQ_Contact(in1 := "MODE SELECTION DB"."UF PLC_1 MODE BUFF", in2 := 1)
      { S7_Templates := "SrcType := Int" } EQ_Contact(in1 := "MODE SELECTION DB"."UF PLC_1 PROCESS BUFF", in2 := 225)
      Contact( "INPUT MAPPING DB"."ABFV 202 FEED BACK OPEN" )
      Move(in := 230, out1 => "MODE SELECTION DB"."UF PLC_1 PROCESS BUFF")
   END_RUNG
   // the same network as SCL:
   IF ("MODE SELECTION DB"."UF PLC_1 MODE BUFF" = 1) AND ("MODE SELECTION DB"."UF PLC_1 PROCESS BUFF" = 225) AND "INPUT MAPPING DB"."ABFV 202 FEED BACK OPEN" THEN
       "MODE SELECTION DB"."UF PLC_1 PROCESS BUFF" := 230;
   END_IF;
END_REGION

REGION Network 52: ABFV 204 OPEN FB
   RUNG wire#powerrail
      { S7_Templates := "SrcType := Int" } EQ_Contact(in1 := "MODE SELECTION DB"."UF PLC_1 MODE BUFF", in2 := 1)
      { S7_Templates := "SrcType := Int" } EQ_Contact(in1 := "MODE SELECTION DB"."UF PLC_1 PROCESS BUFF", in2 := 230)
      Contact( "INPUT MAPPING DB"."ABFV 204 FEED BACK OPEN" )
      Move(in := 235, out1 => "MODE SELECTION DB"."UF PLC_1 PROCESS BUFF")
   END_RUNG
   // the same network as SCL:
   IF ("MODE SELECTION DB"."UF PLC_1 MODE BUFF" = 1) AND ("MODE SELECTION DB"."UF PLC_1 PROCESS BUFF" = 230) AND "INPUT MAPPING DB"."ABFV 204 FEED BACK OPEN" THEN
       "MODE SELECTION DB"."UF PLC_1 PROCESS BUFF" := 235;
   END_IF;
END_REGION

REGION Network 53: ABFV 206 OPEN FB
   RUNG wire#powerrail
      { S7_Templates := "SrcType := Int" } EQ_Contact(in1 := "MODE SELECTION DB"."UF PLC_1 MODE BUFF", in2 := 1)
      { S7_Templates := "SrcType := Int" } EQ_Contact(in1 := "MODE SELECTION DB"."UF PLC_1 PROCESS BUFF", in2 := 235)
      Contact( "INPUT MAPPING DB"."ABFV 206 FEED BACK OPEN" )
      { S7_Templates := "time_type := Time" } "IEC_Timer_0_DB_55".TON(pt := T#10S, et =>)
      Move(in := 240, out1 => "MODE SELECTION DB"."UF PLC_1 PROCESS BUFF")
   END_RUNG
   // the same network as SCL:
   "IEC_Timer_0_DB_55".TON(IN := ("MODE SELECTION DB"."UF PLC_1 MODE BUFF" = 1) AND ("MODE SELECTION DB"."UF PLC_1 PROCESS BUFF" = 235) AND "INPUT MAPPING DB"."ABFV 206 FEED BACK OPEN",
                           PT := T#10S);
   IF "IEC_Timer_0_DB_55".Q THEN "MODE SELECTION DB"."UF PLC_1 PROCESS BUFF" := 240; END_IF;
END_REGION

REGION Network 54: BACKWASH-2
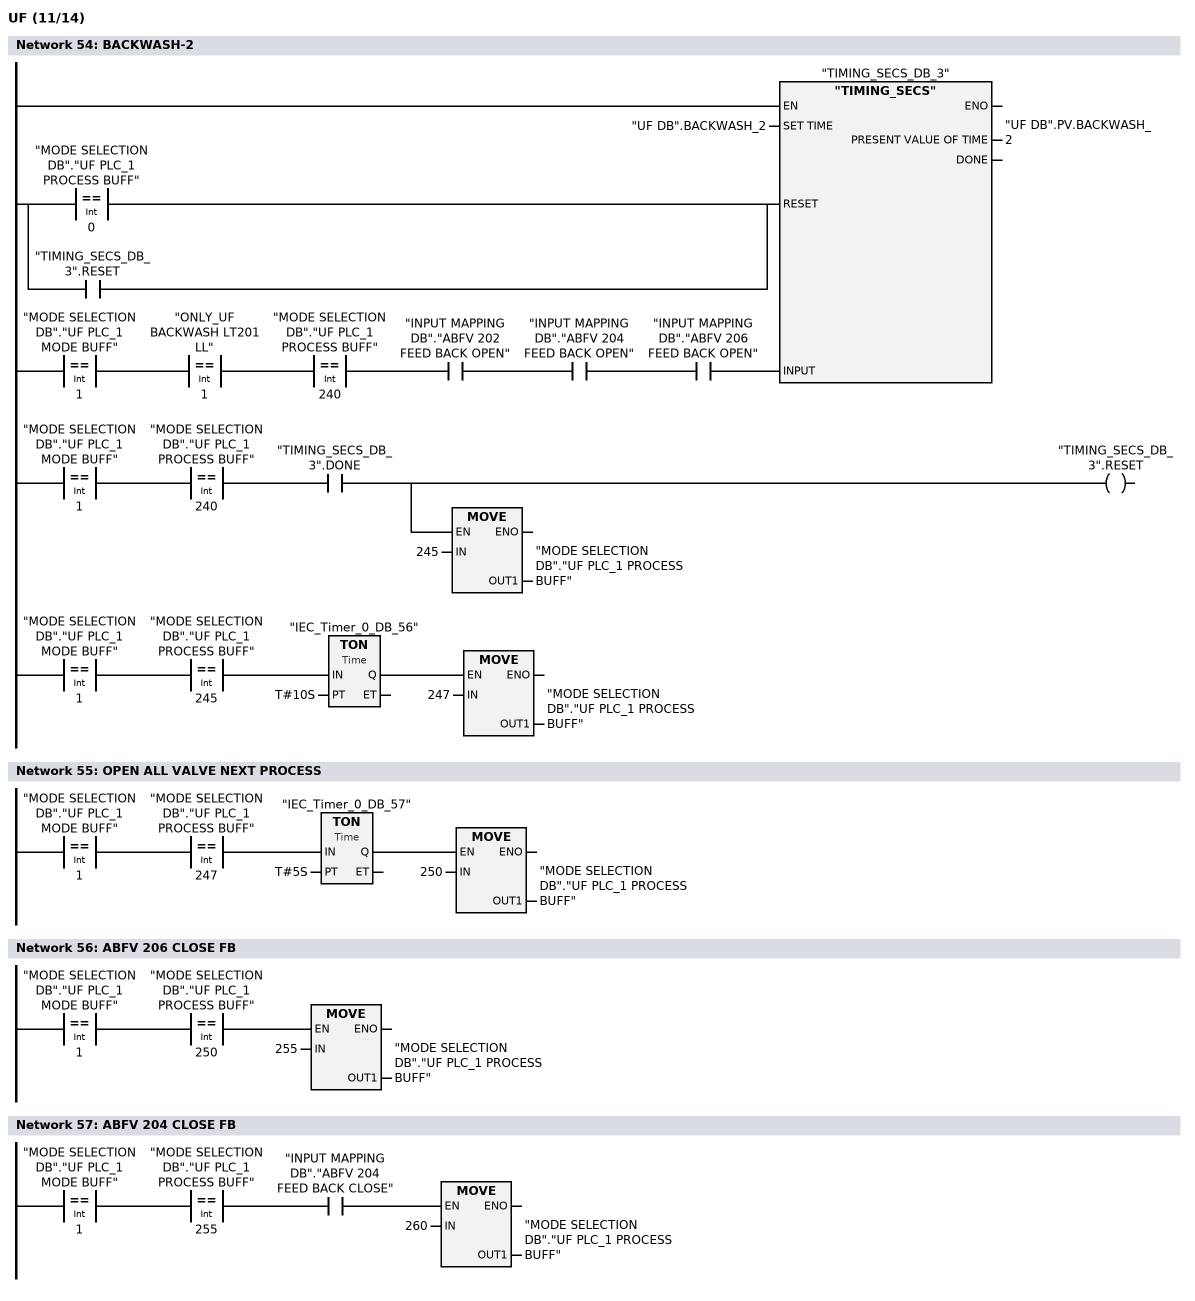
   RUNG wire#powerrail
      "TIMING_SECS_DB_3"(RESET := wire#w1, INPUT := wire#w2, "SET TIME" := "UF DB".BACKWASH_2, "PRESENT VALUE OF TIME" => "UF DB".PV.BACKWASH_2, DONE =>)
   END_RUNG
   RUNG wire#powerrail
      { S7_Templates := "SrcType := Int" } EQ_Contact(in1 := "MODE SELECTION DB"."UF PLC_1 PROCESS BUFF", in2 := 0)
   END_RUNG wire#w1
   RUNG wire#powerrail
      Contact( "TIMING_SECS_DB_3".RESET )
   END_RUNG wire#w1
   RUNG wire#powerrail
      { S7_Templates := "SrcType := Int" } EQ_Contact(in1 := "MODE SELECTION DB"."UF PLC_1 MODE BUFF", in2 := 1)
      { S7_Templates := "SrcType := Int" } EQ_Contact(in1 := "ONLY_UF BACKWASH LT201 LL", in2 := 1)
      { S7_Templates := "SrcType := Int" } EQ_Contact(in1 := "MODE SELECTION DB"."UF PLC_1 PROCESS BUFF", in2 := 240)
      Contact( "INPUT MAPPING DB"."ABFV 202 FEED BACK OPEN" )
      Contact( "INPUT MAPPING DB"."ABFV 204 FEED BACK OPEN" )
      Contact( "INPUT MAPPING DB"."ABFV 206 FEED BACK OPEN" )
   END_RUNG wire#w2
   RUNG wire#powerrail
      { S7_Templates := "SrcType := Int" } EQ_Contact(in1 := "MODE SELECTION DB"."UF PLC_1 MODE BUFF", in2 := 1)
      { S7_Templates := "SrcType := Int" } EQ_Contact(in1 := "MODE SELECTION DB"."UF PLC_1 PROCESS BUFF", in2 := 240)
      Contact( "TIMING_SECS_DB_3".DONE )
      wire#w3
      Coil( "TIMING_SECS_DB_3".RESET )
   END_RUNG
   RUNG wire#w3
      Move(in := 245, out1 => "MODE SELECTION DB"."UF PLC_1 PROCESS BUFF")
   END_RUNG
   RUNG wire#powerrail
      { S7_Templates := "SrcType := Int" } EQ_Contact(in1 := "MODE SELECTION DB"."UF PLC_1 MODE BUFF", in2 := 1)
      { S7_Templates := "SrcType := Int" } EQ_Contact(in1 := "MODE SELECTION DB"."UF PLC_1 PROCESS BUFF", in2 := 245)
      { S7_Templates := "time_type := Time" } "IEC_Timer_0_DB_56".TON(pt := T#10S, et =>)
      Move(in := 247, out1 => "MODE SELECTION DB"."UF PLC_1 PROCESS BUFF")
   END_RUNG
   // the same network as SCL:
   "TIMING_SECS_DB_3"("SET TIME" := "UF DB".BACKWASH_2,   // "TIMING_SECS"
                      RESET := ("MODE SELECTION DB"."UF PLC_1 PROCESS BUFF" = 0) OR "TIMING_SECS_DB_3".RESET,
                      INPUT := ("MODE SELECTION DB"."UF PLC_1 MODE BUFF" = 1) AND ("ONLY_UF BACKWASH LT201 LL" = 1) AND ("MODE SELECTION DB"."UF PLC_1 PROCESS BUFF" = 240) AND "INPUT MAPPING DB"."ABFV 202 FEED BACK OPEN" AND "INPUT MAPPING DB"."ABFV 204 FEED BACK OPEN" AND "INPUT MAPPING DB"."ABFV 206 FEED BACK OPEN",
                      "PRESENT VALUE OF TIME" => "UF DB".PV.BACKWASH_2);
   "TIMING_SECS_DB_3".RESET := ("MODE SELECTION DB"."UF PLC_1 MODE BUFF" = 1) AND ("MODE SELECTION DB"."UF PLC_1 PROCESS BUFF" = 240) AND "TIMING_SECS_DB_3".DONE;
   IF "TIMING_SECS_DB_3".RESET THEN "MODE SELECTION DB"."UF PLC_1 PROCESS BUFF" := 245; END_IF;
   "IEC_Timer_0_DB_56".TON(IN := ("MODE SELECTION DB"."UF PLC_1 MODE BUFF" = 1) AND ("MODE SELECTION DB"."UF PLC_1 PROCESS BUFF" = 245),
                           PT := T#10S);
   IF "IEC_Timer_0_DB_56".Q THEN "MODE SELECTION DB"."UF PLC_1 PROCESS BUFF" := 247; END_IF;
END_REGION

REGION Network 55: OPEN ALL VALVE NEXT PROCESS
   RUNG wire#powerrail
      { S7_Templates := "SrcType := Int" } EQ_Contact(in1 := "MODE SELECTION DB"."UF PLC_1 MODE BUFF", in2 := 1)
      { S7_Templates := "SrcType := Int" } EQ_Contact(in1 := "MODE SELECTION DB"."UF PLC_1 PROCESS BUFF", in2 := 247)
      { S7_Templates := "time_type := Time" } "IEC_Timer_0_DB_57".TON(pt := T#5S, et =>)
      Move(in := 250, out1 => "MODE SELECTION DB"."UF PLC_1 PROCESS BUFF")
   END_RUNG
   // the same network as SCL:
   "IEC_Timer_0_DB_57".TON(IN := ("MODE SELECTION DB"."UF PLC_1 MODE BUFF" = 1) AND ("MODE SELECTION DB"."UF PLC_1 PROCESS BUFF" = 247),
                           PT := T#5S);
   IF "IEC_Timer_0_DB_57".Q THEN "MODE SELECTION DB"."UF PLC_1 PROCESS BUFF" := 250; END_IF;
END_REGION

REGION Network 56: ABFV 206 CLOSE FB
   RUNG wire#powerrail
      { S7_Templates := "SrcType := Int" } EQ_Contact(in1 := "MODE SELECTION DB"."UF PLC_1 MODE BUFF", in2 := 1)
      { S7_Templates := "SrcType := Int" } EQ_Contact(in1 := "MODE SELECTION DB"."UF PLC_1 PROCESS BUFF", in2 := 250)
      Move(in := 255, out1 => "MODE SELECTION DB"."UF PLC_1 PROCESS BUFF")
   END_RUNG
   // the same network as SCL:
   IF ("MODE SELECTION DB"."UF PLC_1 MODE BUFF" = 1) AND ("MODE SELECTION DB"."UF PLC_1 PROCESS BUFF" = 250) THEN
       "MODE SELECTION DB"."UF PLC_1 PROCESS BUFF" := 255;
   END_IF;
END_REGION

